2095.08 BOOL  ; RK_07 U8_Z 铝壳上料移载Y轴CW极限输入信号
2095.09 BOOL  ; RK_07 U8_Z 铝壳上料移载Y轴CCW极限输入信号
2095.10 BOOL  ; RK_07 U8_Z 铝壳上料移载Y轴原点接近输入信号
2095.11 BOOL  ; RK_07 U8_Z 铝壳上料移载Y轴原点输入信号
2095.12 BOOL  ; RK_07 U8_Z 铝壳上料移载Y轴中断输入信号
2095.13 BOOL  ; RK_07 U8_Z 铝壳上料移载Y轴紧急停止输入信号
2095.14 BOOL  ; RK_07 U8_Z 铝壳上料移载Y轴定位完成信号
2095.15 BOOL  ; $?St$Bk?_#[5047] / RK_07 U8_Z 铝壳上料移载Y轴偏差计数器复位输出 / 原点调整命令输出$?St$Bk?_#[5047]
2096 CHANNEL  ; RK_07 U8_Z 铝壳上料移载Y轴错误代码
2096.00 BOOL  ; RK_07 U8_Z 铝壳上料移载Y轴错误代码
2096.01 BOOL  ; RK_07 U8_Z 铝壳上料移载Y轴错误代码
2096.02 BOOL  ; RK_07 U8_Z 铝壳上料移载Y轴错误代码
2096.03 BOOL  ; RK_07 U8_Z 铝壳上料移载Y轴错误代码
2096.04 BOOL  ; RK_07 U8_Z 铝壳上料移载Y轴错误代码
2096.05 BOOL  ; RK_07 U8_Z 铝壳上料移载Y轴错误代码
2096.06 BOOL  ; RK_07 U8_Z 铝壳上料移载Y轴错误代码
2096.07 BOOL  ; RK_07 U8_Z 铝壳上料移载Y轴错误代码
2096.08 BOOL  ; RK_07 U8_Z 铝壳上料移载Y轴错误代码
2096.09 BOOL  ; RK_07 U8_Z 铝壳上料移载Y轴错误代码
2096.10 BOOL  ; RK_07 U8_Z 铝壳上料移载Y轴错误代码
2096.11 BOOL  ; RK_07 U8_Z 铝壳上料移载Y轴错误代码
2096.12 BOOL  ; RK_07 U8_Z 铝壳上料移载Y轴错误代码
2096.13 BOOL  ; RK_07 U8_Z 铝壳上料移载Y轴错误代码
2096.14 BOOL  ; RK_07 U8_Z 铝壳上料移载Y轴错误代码
2096.15 BOOL  ; RK_07 U8_Z 铝壳上料移载Y轴错误代码
2097.00 BOOL  ; RK_10 U8_U 电池除尘上料X轴Not Use
2097.01 BOOL  ; RK_10 U8_U 电池除尘上料X轴Not Use
2097.02 BOOL  ; RK_10 U8_U 电池除尘上料X轴Not Use
2097.03 BOOL  ; RK_10 U8_U 电池除尘上料X轴Not Use
2097.04 BOOL  ; RK_10 U8_U 电池除尘上料X轴等待存储器操作标志位
2097.05 BOOL  ; RK_10 U8_U 电池除尘上料X轴定位结束标志位
2097.06 BOOL  ; RK_10 U8_U 电池除尘上料X轴无原点标志位
2097.07 BOOL  ; RK_10 U8_U 电池除尘上料X轴原点停止标志位
2097.08 BOOL  ; RK_10 U8_U 电池除尘上料X轴区域0监控标志位
2097.09 BOOL  ; RK_10 U8_U 电池除尘上料X轴区域1监控标志位
2097.10 BOOL  ; RK_10 U8_U 电池除尘上料X轴区域2监控标志位
2097.11 BOOL  ; RK_10 U8_U 电池除尘上料X轴示教完成标志位
2097.12 BOOL  ; RK_10 U8_U 电池除尘上料X轴错误标志位
2097.13 BOOL  ; RK_10 U8_U 电池除尘上料X轴忙标志位
2097.14 BOOL  ; RK_10 U8_U 电池除尘上料X轴数据传送标志
2097.15 BOOL  ; RK_10 U8_U 电池除尘上料X轴减速停止执行标志
2098.00 BOOL  ; RK_10 U8_U 电池除尘上料X轴Not Use
2098.01 BOOL  ; RK_10 U8_U 电池除尘上料X轴Not Use
2098.02 BOOL  ; RK_10 U8_U 电池除尘上料X轴Not Use
2098.03 BOOL  ; RK_10 U8_U 电池除尘上料X轴Not Use
2098.04 BOOL  ; RK_10 U8_U 电池除尘上料X轴Not Use
2098.05 BOOL  ; RK_10 U8_U 电池除尘上料X轴Not Use
2098.06 BOOL  ; RK_10 U8_U 电池除尘上料X轴Not Use
2098.07 BOOL  ; RK_10 U8_U 电池除尘上料X轴Not Use
2098.08 BOOL  ; RK_10 U8_U 电池除尘上料X轴CW极限输入信号
2098.09 BOOL  ; RK_10 U8_U 电池除尘上料X轴CCW极限输入信号
2098.10 BOOL  ; RK_10 U8_U 电池除尘上料X轴原点接近输入信号
2098.11 BOOL  ; RK_10 U8_U 电池除尘上料X轴原点输入信号
2098.12 BOOL  ; RK_10 U8_U 电池除尘上料X轴中断输入信号
2098.13 BOOL  ; RK_10 U8_U 电池除尘上料X轴紧急停止输入信号
2098.14 BOOL  ; RK_10 U8_U 电池除尘上料X轴定位完成信号
2098.15 BOOL  ; $?St$Bk?_#[5048] / RK_10 U8_U 电池除尘上料X轴偏差计数器复位输出 / 原点调整命令输出$?St$Bk?_#[5048]
2099 CHANNEL  ; RK_10 U8_U 电池除尘上料X轴错误代码
2099.00 BOOL  ; RK_10 U8_U 电池除尘上料X轴错误代码
2099.01 BOOL  ; RK_10 U8_U 电池除尘上料X轴错误代码
2099.02 BOOL  ; RK_10 U8_U 电池除尘上料X轴错误代码
2099.03 BOOL  ; RK_10 U8_U 电池除尘上料X轴错误代码
2099.04 BOOL  ; RK_10 U8_U 电池除尘上料X轴错误代码
2099.05 BOOL  ; RK_10 U8_U 电池除尘上料X轴错误代码
2099.06 BOOL  ; RK_10 U8_U 电池除尘上料X轴错误代码
2099.07 BOOL  ; RK_10 U8_U 电池除尘上料X轴错误代码
2099.08 BOOL  ; RK_10 U8_U 电池除尘上料X轴错误代码
2099.09 BOOL  ; RK_10 U8_U 电池除尘上料X轴错误代码
2099.10 BOOL  ; RK_10 U8_U 电池除尘上料X轴错误代码
2099.11 BOOL  ; RK_10 U8_U 电池除尘上料X轴错误代码
2099.12 BOOL  ; RK_10 U8_U 电池除尘上料X轴错误代码
2099.13 BOOL  ; RK_10 U8_U 电池除尘上料X轴错误代码
2099.14 BOOL  ; RK_10 U8_U 电池除尘上料X轴错误代码
2099.15 BOOL  ; RK_10 U8_U 电池除尘上料X轴错误代码
2101 CHANNEL  ; RK_05 #1入壳压力采样值
2102 CHANNEL  ; RK_05 #2入壳压力采样值
210.01 BOOL  ; PC系统通讯正常标志
210.02 BOOL  ; 整机机械手归零标志
210.03 BOOL  ; 安全门标志
221.00 BOOL  ; 整机复位（M）
221.01 BOOL  ; RK_01 电芯来料机构整机复位（M）
221.02 BOOL  ; RK_02 电芯进料机构整机复位（M）
221.03 BOOL  ; RK_03 电芯上料机构整机复位（M）
221.04 BOOL  ; RK_04 电芯除尘机构整机复位（M）
221.05 BOOL  ; RK_05 #1入壳机构整机复位（M）
221.06 BOOL  ; RK_05 #2入壳机构整机复位（M）
221.07 BOOL  ; RK_06 电池上下料机构整机复位（M）
221.08 BOOL  ; RK_07 铝壳进料机构整机复位（M）
221.09 BOOL  ; RK_07 铝壳上料移载机构整机复位（M）
221.10 BOOL  ; RK_07 #1铝壳上料升降机构整机复位（M）
221.11 BOOL  ; RK_07 #2铝壳上料升降机构整机复位（M）
221.12 BOOL  ; RK_07 铝壳托盘下料升降机构整机复位（M）
221.13 BOOL  ; RK_08 铝壳除尘机构整机复位（M）
221.14 BOOL  ; RK_09 #1Hipot检测机构整机复位（M）
221.15 BOOL  ; RK_09 #2Hipot检测机构整机复位（M）
222.00 BOOL  ; RK_10 电池除尘上料机构整机复位（M）
222.01 BOOL  ; RK_11 电池除尘机构整机复位（M）
222.02 BOOL  ; RK_12 预焊上下料机构整机复位（M）
222.03 BOOL  ; RK_13 #1移载机构整机复位（M）
222.04 BOOL  ; RK_13 #2移载机构整机复位（M）
222.05 BOOL  ; RK_14 #1压装机构整机复位（M）
222.06 BOOL  ; RK_14 #2压装机构整机复位（M）
222.07 BOOL  ; RK_15 轮廓检测机构整机复位（M）
222.08 BOOL  ; RK_16 焊接机构整机复位（M）
2.00 BOOL  ; RK_01 U0_X 电芯来料Y轴报警信号
2.01 BOOL  ; RK_01 U0_X 电芯来料Y轴准备好了信号
2.02 BOOL  ; RK_02 U0_Y 电芯进料X轴报警信号
2.03 BOOL  ; RK_02 U0_Y 电芯进料X轴准备好了信号
2.04 BOOL  ; RK_02 U0_Z 电芯进料Z轴报警信号
2.05 BOOL  ; RK_02 U0_Z 电芯进料Z轴准备好了信号
2.06 BOOL  ; RK_03 U0_U 电芯上料X轴报警信号
2.07 BOOL  ; RK_03 U0_U 电芯上料X轴准备好了信号
2.08 BOOL  ; RK_05 U2_X #1入壳Y轴报警信号
2.09 BOOL  ; RK_05 U2_X #1入壳Y轴准备好了信号
2.10 BOOL  ; RK_05 U2_Y #2入壳Y轴报警信号
2.11 BOOL  ; RK_05 U2_Y #2入壳Y轴准备好了信号
2.13 BOOL  ; RK_05 #1入壳定位陶瓷棒上#1夹紧气缸伸出位
2.14 BOOL  ; RK_05 #1入壳定位陶瓷棒上#2夹紧气缸伸出位
2.15 BOOL  ; RK_05 #1入壳定位陶瓷棒下#1夹紧气缸伸出位
3000.00 BOOL  ; 前工序安全位模拟
300.00 BOOL  ; RK_02 电芯进料机械手夹爪气缸夹紧[Pls]
300.01 BOOL  ; RK_02 电芯进料机械手夹爪气缸张开[Pls]
300.02 BOOL  ; RK_02 电芯进料机械手压紧气缸伸出[Pls]
300.03 BOOL  ; RK_02 电芯进料机械手压紧气缸缩回[Pls]
300.04 BOOL  ; RK_03 电芯上料机械手夹爪气缸夹紧[Pls]
300.05 BOOL  ; RK_03 电芯上料机械手夹爪气缸张开[Pls]
300.06 BOOL  ; RK_03 电芯上料机械手压紧气缸伸出[Pls]
300.07 BOOL  ; RK_03 电芯上料机械手压紧气缸缩回[Pls]
300.08 BOOL  ; RK_03 电芯上料升降气缸下降[Pls]
300.09 BOOL  ; RK_03 电芯上料升降气缸上升[Pls]
300.10 BOOL  ; RK_04 电芯除尘伸缩气缸缩回[Pls]
300.11 BOOL  ; RK_04 电芯除尘伸缩气缸伸出[Pls]
300.12 BOOL  ; RK_05 #1入壳滚轮夹紧气缸伸出[Pls]
300.13 BOOL  ; RK_05 #1入壳滚轮夹紧气缸缩回[Pls]
300.14 BOOL  ; RK_05 #1入壳铝壳定位平台伸缩气缸缩回[Pls]
300.15 BOOL  ; RK_05 #1入壳铝壳定位平台伸缩气缸伸出[Pls]
301.00 BOOL  ; RK_05 #1入壳铝壳定位平台升降气缸上升[Pls]
301.01 BOOL  ; RK_05 #1入壳铝壳定位平台升降气缸下降[Pls]
301.02 BOOL  ; RK_05 #1入壳铝壳定位伸缩气缸缩回[Pls]
301.03 BOOL  ; RK_05 #1入壳铝壳定位伸缩气缸伸出[Pls]
301.04 BOOL  ; RK_05 #1入壳铝壳定位夹爪气缸夹紧[Pls]
301.05 BOOL  ; RK_05 #1入壳铝壳定位夹爪气缸张开[Pls]
301.06 BOOL  ; RK_05 #2入壳滚轮夹紧气缸伸出[Pls]
301.07 BOOL  ; RK_05 #2入壳滚轮夹紧气缸缩回[Pls]
301.08 BOOL  ; RK_05 #2入壳铝壳定位平台伸缩气缸缩回[Pls]
301.09 BOOL  ; RK_05 #2入壳铝壳定位平台伸缩气缸伸出[Pls]
301.10 BOOL  ; RK_05 #2入壳铝壳定位平台升降气缸上升[Pls]
301.11 BOOL  ; RK_05 #2入壳铝壳定位平台升降气缸下降[Pls]
301.12 BOOL  ; RK_05 #2入壳铝壳定位伸缩气缸缩回[Pls]
301.13 BOOL  ; RK_05 #2入壳铝壳定位伸缩气缸伸出[Pls]
301.14 BOOL  ; RK_05 #2入壳铝壳定位夹爪气缸夹紧[Pls]
301.15 BOOL  ; RK_05 #2入壳铝壳定位夹爪气缸张开[Pls]
302.00 BOOL  ; RK_01 U0_X 电芯来料Y轴报警复位[Pls]
302.01 BOOL  ; RK_01 U0_X 电芯来料Y轴使能[Pls]
302.02 BOOL  ; RK_02 U0_Y 电芯进料X轴报警复位[Pls]
302.03 BOOL  ; RK_02 U0_Y 电芯进料X轴使能[Pls]
302.04 BOOL  ; RK_02 U0_Z 电芯进料Z轴报警复位[Pls]
302.05 BOOL  ; RK_02 U0_Z 电芯进料Z轴使能[Pls]
302.06 BOOL  ; RK_03 U0_U 电芯上料X轴报警复位[Pls]
302.07 BOOL  ; RK_03 U0_U 电芯上料X轴使能[Pls]
302.08 BOOL  ; RK_05 U2_X #1入壳Y轴报警复位[Pls]
302.09 BOOL  ; RK_05 U2_X #1入壳Y轴使能[Pls]
302.10 BOOL  ; RK_05 U2_Y #2入壳Y轴报警复位[Pls]
302.11 BOOL  ; RK_05 U2_Y #2入壳Y轴使能[Pls]
302.12 BOOL  ; RK_02 电芯进料Z轴刹车使能[Pls]
302.13 BOOL  ; RK_05 #1入壳定位陶瓷棒夹紧气缸伸出[Pls]
302.14 BOOL  ; RK_05 #1入壳定位陶瓷棒夹紧气缸缩回[Pls]
302.15 BOOL  ; RK_05 #2入壳定位陶瓷棒夹紧气缸伸出[Pls]
303.00 BOOL  ; RK_05 #2入壳定位陶瓷棒夹紧气缸缩回[Pls]
303.01 BOOL  ; RK_04 电芯除尘吹气阀开[Pls]
303.02 BOOL  ; RK_02 扫码NG拉带启动[Pls]
303.03 BOOL  ; RK_05 #1入壳吸盘立真空[Pls]
303.04 BOOL  ; RK_05 #2入壳吸盘立真空[Pls]
303.05 BOOL  ; RK_05 #1入壳吸盘伸缩气缸伸出[Pls]
303.06 BOOL  ; RK_05 #1入壳吸盘伸缩气缸缩回[Pls]
303.07 BOOL  ; RK_05 #2入壳吸盘伸缩气缸伸出[Pls]
303.08 BOOL  ; RK_05 #2入壳吸盘伸缩气缸缩回[Pls]
303.09 BOOL  ; 前端设备对接输出信号（公共）[Pls]
303.10 BOOL  ; 后端设备对接输出信号（公共）[Pls]
303.11 BOOL  ; RK_05 #1入壳电芯定位夹爪气缸伸出[Pls]
303.12 BOOL  ; RK_05 #1入壳电芯定位夹爪气缸缩回[Pls]
303.13 BOOL  ; RK_05 #2入壳电芯定位夹爪气缸伸出[Pls]
303.14 BOOL  ; RK_05 #2入壳电芯定位夹爪气缸缩回[Pls]
308.00 BOOL  ; RK_11 电池除尘旋转伸缩气缸缩回[Pls]
308.01 BOOL  ; RK_11 电池除尘旋转伸缩气缸伸出[Pls]
308.02 BOOL  ; RK_11 电池除尘伸缩气缸伸出[Pls]
308.03 BOOL  ; RK_11 电池除尘伸缩气缸缩回[Pls]
308.04 BOOL  ; RK_11 电池除尘夹爪气缸夹紧[Pls]
308.05 BOOL  ; RK_11 电池除尘夹爪气缸张开[Pls]
308.06 BOOL  ; RK_12 预焊上料机械手夹爪气缸夹紧[Pls]
308.07 BOOL  ; RK_12 预焊上料机械手夹爪气缸张开[Pls]
308.08 BOOL  ; RK_12 预焊下料机械手夹爪气缸夹紧[Pls]
308.09 BOOL  ; RK_12 预焊下料机械手夹爪气缸张开[Pls]
308.10 BOOL  ; RK_13 #1移载升降气缸上升[Pls]
308.11 BOOL  ; RK_13 #1移载升降气缸下降[Pls]
308.12 BOOL  ; RK_13 #1移载定位#1伸缩气缸缩回[Pls]
308.13 BOOL  ; RK_13 #1移载定位#1伸缩气缸伸出[Pls]
308.14 BOOL  ; RK_13 #1移载定位#2伸缩气缸缩回[Pls]
308.15 BOOL  ; RK_13 #1移载定位#2伸缩气缸伸出[Pls]
309.00 BOOL  ; RK_13 #1移载导向#1伸缩气缸伸出[Pls]
309.01 BOOL  ; RK_13 #1移载导向#1伸缩气缸缩回[Pls]
309.02 BOOL  ; RK_13 #1移载导向#2伸缩气缸伸出[Pls]
309.03 BOOL  ; RK_13 #1移载导向#2伸缩气缸缩回[Pls]
309.04 BOOL  ; RK_13 #1移载左右定位伸缩气缸伸出[Pls]
309.05 BOOL  ; RK_13 #1移载左右定位伸缩气缸缩回[Pls]
309.06 BOOL  ; RK_13 #2移载升降气缸上升[Pls]
309.07 BOOL  ; RK_13 #2移载升降气缸下降[Pls]
309.08 BOOL  ; RK_13 #2移载定位#1伸缩气缸缩回[Pls]
309.09 BOOL  ; RK_13 #2移载定位#1伸缩气缸伸出[Pls]
309.10 BOOL  ; RK_13 #2移载定位#2伸缩气缸缩回[Pls]
309.11 BOOL  ; RK_13 #2移载定位#2伸缩气缸伸出[Pls]
309.12 BOOL  ; RK_13 #2移载导向#1伸缩气缸伸出[Pls]
309.13 BOOL  ; RK_13 #2移载导向#1伸缩气缸缩回[Pls]
309.14 BOOL  ; RK_13 #2移载导向#2伸缩气缸伸出[Pls]
309.15 BOOL  ; RK_13 #2移载导向#2伸缩气缸缩回[Pls]
310.00 BOOL  ; RK_13 #2移载左右定位伸缩气缸伸出[Pls]
310.01 BOOL  ; RK_13 #2移载左右定位伸缩气缸缩回[Pls]
310.02 BOOL  ; RK_14 #1压装升降气缸下降[Pls]
310.03 BOOL  ; RK_14 #1压装升降气缸上升[Pls]
310.04 BOOL  ; RK_14 #1压装#1吸盘升降气缸下降[Pls]
310.05 BOOL  ; RK_14 #1压装#1吸盘升降气缸上升[Pls]
310.06 BOOL  ; RK_14 #1压装#2吸盘升降气缸下降[Pls]
310.07 BOOL  ; RK_14 #1压装#2吸盘升降气缸上升[Pls]
310.08 BOOL  ; RK_14 #2压装升降气缸下降[Pls]
310.09 BOOL  ; RK_14 #2压装升降气缸上升[Pls]
310.10 BOOL  ; RK_14 #2压装#1吸盘升降气缸下降[Pls]
310.11 BOOL  ; RK_14 #2压装#1吸盘升降气缸上升[Pls]
310.12 BOOL  ; RK_14 #2压装#2吸盘升降气缸下降[Pls]
310.13 BOOL  ; RK_14 #2压装#2吸盘升降气缸上升[Pls]
310.14 BOOL  ; RK_15 轮廓检测#1伸缩气缸伸出[Pls]
310.15 BOOL  ; RK_15 轮廓检测#1伸缩气缸缩回[Pls]
311.00 BOOL  ; RK_15 轮廓检测#2伸缩气缸伸出[Pls]
311.01 BOOL  ; RK_15 轮廓检测#2伸缩气缸缩回[Pls]
311.02 BOOL  ; RK_12 轮廓检测NG拨料气缸伸出[Pls]
311.03 BOOL  ; RK_12 轮廓检测NG拨料气缸缩回[Pls]
311.04 BOOL  ; RK_11 电池除尘吹气阀开[Pls]
311.05 BOOL  ; 0[Pls]
311.06 BOOL  ; 0[Pls]
311.07 BOOL  ; RK_16 激光焊接触发[Pls]
311.08 BOOL  ; RK_16 PLC急停输出到激光设备[Pls]
311.09 BOOL  ; RK_16 #1移载激光焊任务选择[Pls]
311.10 BOOL  ; RK_16 #2移载激光焊任务选择[Pls]
311.11 BOOL  ; RK_16 集尘器启动[Pls]
311.12 BOOL  ; 0[Pls]
311.13 BOOL  ; 0[Pls]
311.14 BOOL  ; RK_14 #1压装吸盘立真空[Pls]
311.15 BOOL  ; RK_14 #2压装吸盘立真空[Pls]
312.00 BOOL  ; RK_12 U4_X 预焊上下料X轴报警复位[Pls]
312.01 BOOL  ; RK_12 U4_X 预焊上下料X轴使能[Pls]
312.02 BOOL  ; RK_12 U4_Y 预焊上料Z轴报警复位[Pls]
312.03 BOOL  ; RK_12 U4_Y 预焊上料Z轴使能[Pls]
312.04 BOOL  ; RK_12 U4_Z 预焊下料Z轴报警复位[Pls]
312.05 BOOL  ; RK_12 U4_Z 预焊下料Z轴使能[Pls]
312.06 BOOL  ; RK_13 U4_U #1移载Y轴报警复位[Pls]
312.07 BOOL  ; RK_13 U4_U #1移载Y轴使能[Pls]
312.08 BOOL  ; RK_13 U6_X #2移载Y轴报警复位[Pls]
312.09 BOOL  ; RK_13 U6_X #2移载Y轴使能[Pls]
312.10 BOOL  ; RK_16 U6_Y 激光焊接X轴报警复位[Pls]
312.11 BOOL  ; RK_16 U6_Y 激光焊接X轴使能[Pls]
312.12 BOOL  ; RK_16 U6_Z 激光焊接Z轴报警复位[Pls]
312.13 BOOL  ; RK_16 U6_Z 激光焊接Z轴使能[Pls]
312.14 BOOL  ; RK_12 预焊上料Z轴刹车使能[Pls]
312.15 BOOL  ; RK_12 预焊下料Z轴刹车使能[Pls]
313.00 BOOL  ; RK_16 激光焊接Z轴刹车使能[Pls]
313.01 BOOL  ; 0[Pls]
313.02 BOOL  ; 0[Pls]
313.03 BOOL  ; 0[Pls]
313.04 BOOL  ; 0[Pls]
313.05 BOOL  ; RK_12 OK出料拉带启动[Pls]
313.06 BOOL  ; 0[Pls]
313.07 BOOL  ; 0[Pls]
313.08 BOOL  ; 0[Pls]
313.09 BOOL  ; RK_07 #1铝壳上料电机刹车使能[Pls]
313.10 BOOL  ; RK_07 #2铝壳上料电机刹车使能[Pls]
313.11 BOOL  ; RK_07 #3托盘下料电机刹车使能[Pls]
313.12 BOOL  ; 三色灯_红（公共）[Pls]
313.13 BOOL  ; 三色灯_绿（公共）[Pls]
313.14 BOOL  ; 三色灯_黄（公共）[Pls]
313.15 BOOL  ; 蜂鸣器（公共）[Pls]
314.00 BOOL  ; RK_06 铝壳上料升降气缸下降[Pls]
314.01 BOOL  ; RK_06 铝壳上料升降气缸上升[Pls]
314.02 BOOL  ; RK_06 电池下料升降气缸下降[Pls]
314.03 BOOL  ; RK_06 电池下料升降气缸上升[Pls]
314.04 BOOL  ; RK_06 铝壳上料夹爪气缸夹紧[Pls]
314.05 BOOL  ; RK_06 铝壳上料夹爪气缸张开[Pls]
314.06 BOOL  ; RK_06 电池下料夹爪气缸夹紧[Pls]
314.07 BOOL  ; RK_06 电池下料夹爪气缸张开[Pls]
314.08 BOOL  ; RK_07 #1铝壳上料车定位升降气缸上升[Pls]
314.09 BOOL  ; RK_07 #1铝壳上料车定位升降气缸下降[Pls]
314.10 BOOL  ; RK_07 #2铝壳上料车定位升降气缸上升[Pls]
314.11 BOOL  ; RK_07 #2铝壳上料车定位升降气缸下降[Pls]
314.12 BOOL  ; RK_07 #3托盘下料车定位升降气缸上升[Pls]
314.13 BOOL  ; RK_07 #3托盘下料车定位升降气缸下降[Pls]
314.14 BOOL  ; RK_07 铝壳进料机械手升降气缸下降[Pls]
314.15 BOOL  ; RK_07 铝壳进料机械手升降气缸上升[Pls]
315.00 BOOL  ; RK_08 铝壳除尘旋转伸缩气缸缩回[Pls]
315.01 BOOL  ; RK_08 铝壳除尘旋转伸缩气缸伸出[Pls]
315.02 BOOL  ; RK_08 铝壳除尘伸缩气缸伸出[Pls]
315.03 BOOL  ; RK_08 铝壳除尘伸缩气缸缩回[Pls]
315.04 BOOL  ; RK_08 铝壳除尘夹爪气缸夹紧[Pls]
315.05 BOOL  ; RK_08 铝壳除尘夹爪气缸张开[Pls]
315.06 BOOL  ; RK_09 #1Hipot测试旋转伸缩气缸伸出[Pls]
315.07 BOOL  ; RK_09 #1Hipot测试旋转伸缩气缸缩回[Pls]
315.08 BOOL  ; RK_09 #1Hipot测试平台伸缩气缸缩回[Pls]
315.09 BOOL  ; RK_09 #1Hipot测试平台伸缩气缸伸出[Pls]
315.10 BOOL  ; RK_09 #1Hipot测试伸缩气缸伸出[Pls]
315.11 BOOL  ; RK_09 #1Hipot测试伸缩气缸缩回[Pls]
315.12 BOOL  ; RK_09 #2Hipot测试旋转伸缩气缸伸出[Pls]
315.13 BOOL  ; RK_09 #2Hipot测试旋转伸缩气缸缩回[Pls]
315.14 BOOL  ; RK_09 #2Hipot测试平台伸缩气缸缩回[Pls]
315.15 BOOL  ; RK_09 #2Hipot测试平台伸缩气缸伸出[Pls]
316.00 BOOL  ; RK_09 #2Hipot测试伸缩气缸伸出[Pls]
316.01 BOOL  ; RK_09 #2Hipot测试伸缩气缸缩回[Pls]
316.02 BOOL  ; RK_10 电池除尘上料机械手升降气缸下降[Pls]
316.03 BOOL  ; RK_10 电池除尘上料机械手升降气缸上升[Pls]
316.04 BOOL  ; RK_10 电池除尘上料机械手夹爪气缸夹紧[Pls]
316.05 BOOL  ; RK_10 电池除尘上料机械手夹爪气缸张开[Pls]
316.06 BOOL  ; RK_06 U8_X 电池上下料X轴报警复位[Pls]
316.07 BOOL  ; RK_06 U8_X 电池上下料X轴使能[Pls]
316.08 BOOL  ; RK_07 U8_Y 铝壳进料X轴报警复位[Pls]
316.09 BOOL  ; RK_07 U8_Y 铝壳进料X轴使能[Pls]
316.10 BOOL  ; RK_07 U8_Z 铝壳上料移载Y轴报警复位[Pls]
316.11 BOOL  ; RK_07 U8_Z 铝壳上料移载Y轴使能[Pls]
316.12 BOOL  ; RK_10 U8_U 电池除尘上料X轴报警复位[Pls]
316.13 BOOL  ; RK_10 U8_U 电池除尘上料X轴使能[Pls]
316.14 BOOL  ; RK_09 Hipot测试仪远程使能（取消）[Pls]
316.15 BOOL  ; RK_07 #1铝壳上料启动指示[Pls]
317.00 BOOL  ; RK_07 #2铝壳上料启动指示[Pls]
317.01 BOOL  ; RK_07 #3托盘下料启动指示[Pls]
317.02 BOOL  ; RK_07 铝壳上料移载吸盘立真空[Pls]
317.03 BOOL  ; RK_07 铝壳进料吸盘立真空[Pls]
317.04 BOOL  ; RK_07 #1铝壳上料电机正转[Pls]
317.05 BOOL  ; RK_07 #1铝壳上料电机反转[Pls]
317.06 BOOL  ; RK_10 Hipot检测NG拉带启动[Pls]
317.07 BOOL  ; RK_08 铝壳除尘吹气阀开[Pls]
317.08 BOOL  ; 0[Pls]
317.09 BOOL  ; RK_07 #2铝壳上料电机正转[Pls]
317.10 BOOL  ; RK_07 #2铝壳上料电机反转[Pls]
317.11 BOOL  ; 启动指示_绿（公共）[Pls]
317.12 BOOL  ; 停止指示_红（公共）[Pls]
317.13 BOOL  ; 复位指示_黄（公共）[Pls]
317.14 BOOL  ; RK_07 #3托盘下料电机正转[Pls]
317.15 BOOL  ; RK_07 #3托盘下料电机反转[Pls]
321.04 BOOL  ; RK_11 电池除尘吹气阀关[Pls]
321.14 BOOL  ; RK_14 #1压装吸盘破真空[Pls]
321.15 BOOL  ; RK_14 #2压装吸盘破真空[Pls]
323.01 BOOL  ; RK_04 电芯除尘吹气阀关[Pls]
323.02 BOOL  ; RK_02 扫码NG拉带停止[Pls]
323.03 BOOL  ; RK_05 #1入壳吸盘破真空[Pls]
323.04 BOOL  ; RK_05 #2入壳吸盘破真空[Pls]
323.05 BOOL  ; RK_12 OK出料拉带停止[Pls]
327.02 BOOL  ; RK_07 铝壳上料移载吸盘破真空[Pls]
327.03 BOOL  ; RK_07 铝壳进料吸盘破真空[Pls]
327.04 BOOL  ; RK_07 #1铝壳上料电机停止[Pls]
327.06 BOOL  ; RK_10 Hipot检测NG拉带停止[Pls]
327.07 BOOL  ; RK_08 铝壳除尘吹气阀关[Pls]
327.09 BOOL  ; RK_07 #2铝壳上料电机停止[Pls]
327.14 BOOL  ; RK_07 #3托盘下料电机停止[Pls]
350.00 BOOL  ; RK_01 U0_X 电芯来料Y轴待料位[Pls]
350.01 BOOL  ; RK_01 U0_X 电芯来料Y轴上料位[Pls]
350.02 BOOL  ; RK_01 U0_X 电芯来料Y轴扫码位[Pls]
350.03 BOOL  ; RK_01 U0_X 电芯来料Y轴下料位[Pls]
350.04 BOOL  ; 备用[Pls]
350.05 BOOL  ; 备用[Pls]
350.06 BOOL  ; 备用[Pls]
350.07 BOOL  ; 备用[Pls]
350.08 BOOL  ; 备用[Pls]
350.09 BOOL  ; 备用[Pls]
350.10 BOOL  ; RK_01 U0_X 电芯来料Y轴回原点[Pls]
350.11 BOOL  ; RK_01 U0_X 电芯来料Y轴JOG+[Pls]
350.12 BOOL  ; RK_01 U0_X 电芯来料Y轴JOG-[Pls]
350.13 BOOL  ; RK_01 U0_X 电芯来料Y轴JOG高速[Pls]
350.14 BOOL  ; RK_01 U0_X 电芯来料Y轴JOG低速[Pls]
350.15 BOOL  ; 备用[Pls]
351.00 BOOL  ; RK_02 U0_Y 电芯进料X轴待料位[Pls]
351.01 BOOL  ; RK_02 U0_Y 电芯进料X轴取料位[Pls]
351.02 BOOL  ; RK_02 U0_Y 电芯进料X轴扫码OK放料位[Pls]
351.03 BOOL  ; RK_02 U0_Y 电芯进料X轴扫码NG放料位[Pls]
351.04 BOOL  ; 备用[Pls]
351.05 BOOL  ; 备用[Pls]
351.06 BOOL  ; 备用[Pls]
351.07 BOOL  ; 备用[Pls]
351.08 BOOL  ; 备用[Pls]
351.09 BOOL  ; 备用[Pls]
351.10 BOOL  ; RK_02 U0_Y 电芯进料X轴回原点[Pls]
351.11 BOOL  ; RK_02 U0_Y 电芯进料X轴JOG+[Pls]
351.12 BOOL  ; RK_02 U0_Y 电芯进料X轴JOG-[Pls]
351.13 BOOL  ; RK_02 U0_Y 电芯进料X轴JOG高速[Pls]
351.14 BOOL  ; RK_02 U0_Y 电芯进料X轴JOG低速[Pls]
351.15 BOOL  ; 备用[Pls]
352.00 BOOL  ; RK_02 U0_Z 电芯进料Z轴待料位（扫码）[Pls]
352.01 BOOL  ; RK_02 U0_Z 电芯进料Z轴取料位[Pls]
352.02 BOOL  ; RK_02 U0_Z 电芯进料Z轴扫码OK放料位[Pls]
352.03 BOOL  ; RK_02 U0_Z 电芯进料Z轴扫码NG放料位[Pls]
352.04 BOOL  ; RK_02 U0_Z 电芯进料Z轴扫码位[Pls]
352.05 BOOL  ; 备用[Pls]
352.06 BOOL  ; 备用[Pls]
352.07 BOOL  ; 备用[Pls]
352.08 BOOL  ; 备用[Pls]
352.09 BOOL  ; 备用[Pls]
352.10 BOOL  ; RK_02 U0_Z 电芯进料Z轴回原点[Pls]
352.11 BOOL  ; RK_02 U0_Z 电芯进料Z轴JOG+[Pls]
352.12 BOOL  ; RK_02 U0_Z 电芯进料Z轴JOG-[Pls]
352.13 BOOL  ; RK_02 U0_Z 电芯进料Z轴JOG高速[Pls]
352.14 BOOL  ; RK_02 U0_Z 电芯进料Z轴JOG低速[Pls]
352.15 BOOL  ; 备用[Pls]
353.00 BOOL  ; RK_03 U0_U 电芯上料X轴待料位[Pls]
353.01 BOOL  ; RK_03 U0_U 电芯上料X轴取料位[Pls]
353.02 BOOL  ; RK_03 U0_U 电芯上料X轴#1入壳放料位[Pls]
353.03 BOOL  ; RK_03 U0_U 电芯上料X轴#2入壳放料位[Pls]
353.04 BOOL  ; 备用[Pls]
353.05 BOOL  ; 备用[Pls]
353.06 BOOL  ; 备用[Pls]
353.07 BOOL  ; 备用[Pls]
353.08 BOOL  ; 备用[Pls]
353.09 BOOL  ; 备用[Pls]
353.10 BOOL  ; RK_03 U0_U 电芯上料X轴回原点[Pls]
353.11 BOOL  ; RK_03 U0_U 电芯上料X轴JOG+[Pls]
353.12 BOOL  ; RK_03 U0_U 电芯上料X轴JOG-[Pls]
353.13 BOOL  ; RK_03 U0_U 电芯上料X轴JOG高速[Pls]
353.14 BOOL  ; RK_03 U0_U 电芯上料X轴JOG低速[Pls]
353.15 BOOL  ; 备用[Pls]
354.00 BOOL  ; RK_05 U2_X #1入壳Y轴待料位[Pls]
354.01 BOOL  ; RK_05 U2_X #1入壳Y轴滚轮压紧位[Pls]
354.02 BOOL  ; RK_05 U2_X #1入壳Y轴滚轮松开位[Pls]
354.03 BOOL  ; RK_05 U2_X #1入壳Y轴入壳位[Pls]
354.04 BOOL  ; RK_05 U2_X #1入壳Y轴电芯定位夹爪松开位[Pls]
354.05 BOOL  ; 备用[Pls]
354.06 BOOL  ; 备用[Pls]
354.07 BOOL  ; 备用[Pls]
354.08 BOOL  ; 备用[Pls]
354.09 BOOL  ; 备用[Pls]
354.10 BOOL  ; RK_05 U2_X #1入壳Y轴回原点[Pls]
354.11 BOOL  ; RK_05 U2_X #1入壳Y轴JOG+[Pls]
354.12 BOOL  ; RK_05 U2_X #1入壳Y轴JOG-[Pls]
354.13 BOOL  ; RK_05 U2_X #1入壳Y轴JOG高速[Pls]
354.14 BOOL  ; RK_05 U2_X #1入壳Y轴JOG低速[Pls]
354.15 BOOL  ; 备用[Pls]
355.00 BOOL  ; RK_05 U2_Y #2入壳Y轴待料位[Pls]
355.01 BOOL  ; RK_05 U2_Y #2入壳Y轴滚轮压紧位[Pls]
355.02 BOOL  ; RK_05 U2_Y #2入壳Y轴滚轮松开位[Pls]
355.03 BOOL  ; RK_05 U2_Y #2入壳Y轴入壳位[Pls]
355.04 BOOL  ; RK_05 U2_Y #2入壳Y轴电芯定位夹爪松开位[Pls]
355.05 BOOL  ; 备用[Pls]
355.06 BOOL  ; 备用[Pls]
355.07 BOOL  ; 备用[Pls]
355.08 BOOL  ; 备用[Pls]
355.09 BOOL  ; 备用[Pls]
355.10 BOOL  ; RK_05 U2_Y #2入壳Y轴回原点[Pls]
355.11 BOOL  ; RK_05 U2_Y #2入壳Y轴JOG+[Pls]
355.12 BOOL  ; RK_05 U2_Y #2入壳Y轴JOG-[Pls]
355.13 BOOL  ; RK_05 U2_Y #2入壳Y轴JOG高速[Pls]
355.14 BOOL  ; RK_05 U2_Y #2入壳Y轴JOG低速[Pls]
355.15 BOOL  ; 备用[Pls]
356.00 BOOL  ; RK_12 U4_X 预焊上下料X轴待料位[Pls]
356.01 BOOL  ; RK_12 U4_X 预焊上下料X轴除尘取料位[Pls]
356.02 BOOL  ; RK_12 U4_X 预焊上下料X轴#1移载放料位[Pls]
356.03 BOOL  ; RK_12 U4_X 预焊上下料X轴#2移载放料位[Pls]
356.04 BOOL  ; RK_12 U4_X 预焊上下料X轴#1移载取料位[Pls]
356.05 BOOL  ; RK_12 U4_X 预焊上下料X轴#2移载取料位[Pls]
356.06 BOOL  ; RK_12 U4_X 预焊上下料X轴OK放料位[Pls]
356.07 BOOL  ; RK_12 U4_X 预焊上下料X轴#1NG放料位[Pls]
356.08 BOOL  ; RK_12 U4_X 预焊上下料X轴#2NG放料位[Pls]
356.09 BOOL  ; 备用[Pls]
356.10 BOOL  ; RK_12 U4_X 预焊上下料X轴回原点[Pls]
356.11 BOOL  ; RK_12 U4_X 预焊上下料X轴JOG+[Pls]
356.12 BOOL  ; RK_12 U4_X 预焊上下料X轴JOG-[Pls]
356.13 BOOL  ; RK_12 U4_X 预焊上下料X轴JOG高速[Pls]
356.14 BOOL  ; RK_12 U4_X 预焊上下料X轴JOG低速[Pls]
356.15 BOOL  ; 备用[Pls]
357.00 BOOL  ; RK_12 U4_Y 预焊上料Z轴待料位[Pls]
357.01 BOOL  ; RK_12 U4_Y 预焊上料Z轴除尘取料位[Pls]
357.02 BOOL  ; RK_12 U4_Y 预焊上料Z轴#1移载放料位[Pls]
357.03 BOOL  ; RK_12 U4_Y 预焊上料Z轴#2移载放料位[Pls]
357.04 BOOL  ; 备用[Pls]
357.05 BOOL  ; 备用[Pls]
357.06 BOOL  ; 备用[Pls]
357.07 BOOL  ; 备用[Pls]
357.08 BOOL  ; 备用[Pls]
357.09 BOOL  ; 备用[Pls]
357.10 BOOL  ; RK_12 U4_Y 预焊上料Z轴回原点[Pls]
357.11 BOOL  ; RK_12 U4_Y 预焊上料Z轴JOG+[Pls]
357.12 BOOL  ; RK_12 U4_Y 预焊上料Z轴JOG-[Pls]
357.13 BOOL  ; RK_12 U4_Y 预焊上料Z轴JOG高速[Pls]
357.14 BOOL  ; RK_12 U4_Y 预焊上料Z轴JOG低速[Pls]
357.15 BOOL  ; 备用[Pls]
358.00 BOOL  ; RK_12 U4_Z 预焊下料Z轴待料位[Pls]
358.01 BOOL  ; RK_12 U4_Z 预焊下料Z轴#1移载取料位[Pls]
358.02 BOOL  ; RK_12 U4_Z 预焊下料Z轴#2移载取料位[Pls]
358.03 BOOL  ; RK_12 U4_Z 预焊下料Z轴OK放料位[Pls]
358.04 BOOL  ; RK_12 U4_Z 预焊下料Z轴#1NG放料位[Pls]
358.05 BOOL  ; RK_12 U4_Z 预焊下料Z轴#2NG放料位[Pls]
358.06 BOOL  ; 备用[Pls]
358.07 BOOL  ; 备用[Pls]
358.08 BOOL  ; 备用[Pls]
358.09 BOOL  ; 备用[Pls]
358.10 BOOL  ; RK_12 U4_Z 预焊下料Z轴回原点[Pls]
358.11 BOOL  ; RK_12 U4_Z 预焊下料Z轴JOG+[Pls]
358.12 BOOL  ; RK_12 U4_Z 预焊下料Z轴JOG-[Pls]
358.13 BOOL  ; RK_12 U4_Z 预焊下料Z轴JOG高速[Pls]
358.14 BOOL  ; RK_12 U4_Z 预焊下料Z轴JOG低速[Pls]
358.15 BOOL  ; 备用[Pls]
359.00 BOOL  ; RK_13 U4_U #1移载Y轴待料位[Pls]
359.01 BOOL  ; RK_13 U4_U #1移载Y轴取放料位[Pls]
359.02 BOOL  ; RK_13 U4_U #1移载Y轴压装位[Pls]
359.03 BOOL  ; RK_13 U4_U #1移载Y轴#1轮廓检测位[Pls]
359.04 BOOL  ; RK_13 U4_U #1移载Y轴#2轮廓检测位[Pls]
359.05 BOOL  ; RK_13 U4_U #1移载Y轴激光焊接位[Pls]
359.06 BOOL  ; 备用[Pls]
359.07 BOOL  ; 备用[Pls]
359.08 BOOL  ; 备用[Pls]
359.09 BOOL  ; 备用[Pls]
359.10 BOOL  ; RK_13 U4_U #1移载Y轴回原点[Pls]
359.11 BOOL  ; RK_13 U4_U #1移载Y轴JOG+[Pls]
359.12 BOOL  ; RK_13 U4_U #1移载Y轴JOG-[Pls]
359.13 BOOL  ; RK_13 U4_U #1移载Y轴JOG高速[Pls]
359.14 BOOL  ; RK_13 U4_U #1移载Y轴JOG低速[Pls]
359.15 BOOL  ; 备用[Pls]
360.00 BOOL  ; RK_13 U6_X #2移载Y轴待料位[Pls]
360.01 BOOL  ; RK_13 U6_X #2移载Y轴取放料位[Pls]
360.02 BOOL  ; RK_13 U6_X #2移载Y轴压装位[Pls]
360.03 BOOL  ; RK_13 U6_X #2移载Y轴#1轮廓检测位[Pls]
360.04 BOOL  ; RK_13 U6_X #2移载Y轴#2轮廓检测位[Pls]
360.05 BOOL  ; RK_13 U6_X #2移载Y轴激光焊接位[Pls]
360.06 BOOL  ; 备用[Pls]
360.07 BOOL  ; 备用[Pls]
360.08 BOOL  ; 备用[Pls]
360.09 BOOL  ; 备用[Pls]
360.10 BOOL  ; RK_13 U6_X #2移载Y轴回原点[Pls]
360.11 BOOL  ; RK_13 U6_X #2移载Y轴JOG+[Pls]
360.12 BOOL  ; RK_13 U6_X #2移载Y轴JOG-[Pls]
360.13 BOOL  ; RK_13 U6_X #2移载Y轴JOG高速[Pls]
360.14 BOOL  ; RK_13 U6_X #2移载Y轴JOG低速[Pls]
360.15 BOOL  ; 备用[Pls]
361.00 BOOL  ; RK_16 U6_Y 激光焊接X轴待机位[Pls]
361.01 BOOL  ; RK_16 U6_Y 激光焊接X轴#1移载焊接位[Pls]
361.02 BOOL  ; RK_16 U6_Y 激光焊接X轴#2移载焊接位[Pls]
361.03 BOOL  ; 备用[Pls]
361.04 BOOL  ; 备用[Pls]
361.05 BOOL  ; 备用[Pls]
361.06 BOOL  ; 备用[Pls]
361.07 BOOL  ; 备用[Pls]
361.08 BOOL  ; 备用[Pls]
361.09 BOOL  ; 备用[Pls]
361.10 BOOL  ; RK_16 U6_Y 激光焊接X轴回原点[Pls]
361.11 BOOL  ; RK_16 U6_Y 激光焊接X轴JOG+[Pls]
361.12 BOOL  ; RK_16 U6_Y 激光焊接X轴JOG-[Pls]
361.13 BOOL  ; RK_16 U6_Y 激光焊接X轴JOG高速[Pls]
361.14 BOOL  ; RK_16 U6_Y 激光焊接X轴JOG低速[Pls]
361.15 BOOL  ; 备用[Pls]
362.00 BOOL  ; RK_16 U6_Z 激光焊接Z轴待机位[Pls]
362.01 BOOL  ; RK_16 U6_Z 激光焊接Z轴#1移载焊接位[Pls]
362.02 BOOL  ; RK_16 U6_Z 激光焊接Z轴#2移载焊接位[Pls]
362.03 BOOL  ; 备用[Pls]
362.04 BOOL  ; 备用[Pls]
362.05 BOOL  ; 备用[Pls]
362.06 BOOL  ; 备用[Pls]
362.07 BOOL  ; 备用[Pls]
362.08 BOOL  ; 备用[Pls]
362.09 BOOL  ; 备用[Pls]
362.10 BOOL  ; RK_16 U6_Z 激光焊接Z轴回原点[Pls]
362.11 BOOL  ; RK_16 U6_Z 激光焊接Z轴JOG+[Pls]
362.12 BOOL  ; RK_16 U6_Z 激光焊接Z轴JOG-[Pls]
362.13 BOOL  ; RK_16 U6_Z 激光焊接Z轴JOG高速[Pls]
362.14 BOOL  ; RK_16 U6_Z 激光焊接Z轴JOG低速[Pls]
362.15 BOOL  ; 备用[Pls]
363.00 BOOL  ; RK_06 U8_X 电池上下料X轴待机位[Pls]
363.01 BOOL  ; RK_06 U8_X 电池上下料X轴铝壳除尘取料位[Pls]
363.02 BOOL  ; RK_06 U8_X 电池上下料X轴#1入壳放料位[Pls]
363.03 BOOL  ; RK_06 U8_X 电池上下料X轴#2入壳放料位[Pls]
363.04 BOOL  ; RK_06 U8_X 电池上下料X轴#1入壳取料位[Pls]
363.05 BOOL  ; RK_06 U8_X 电池上下料X轴#2入壳取料位[Pls]
363.06 BOOL  ; RK_06 U8_X 电池上下料X轴#1Hipot检测放料位[Pls]
363.07 BOOL  ; RK_06 U8_X 电池上下料X轴#2Hipot检测放料位[Pls]
363.08 BOOL  ; 备用[Pls]
363.09 BOOL  ; 备用[Pls]
363.10 BOOL  ; RK_06 U8_X 电池上下料X轴回原点[Pls]
363.11 BOOL  ; RK_06 U8_X 电池上下料X轴JOG+[Pls]
363.12 BOOL  ; RK_06 U8_X 电池上下料X轴JOG-[Pls]
363.13 BOOL  ; RK_06 U8_X 电池上下料X轴JOG高速[Pls]
363.14 BOOL  ; RK_06 U8_X 电池上下料X轴JOG低速[Pls]
363.15 BOOL  ; 备用[Pls]
364.00 BOOL  ; RK_07 U8_Y 铝壳进料X轴等待位[Pls]
364.01 BOOL  ; RK_07 U8_Y 铝壳进料X轴取料位[Pls]
364.02 BOOL  ; RK_07 U8_Y 铝壳进料X轴放料位[Pls]
364.03 BOOL  ; 备用[Pls]
364.04 BOOL  ; 备用[Pls]
364.05 BOOL  ; 备用[Pls]
364.06 BOOL  ; 备用[Pls]
364.07 BOOL  ; 备用[Pls]
364.08 BOOL  ; 备用[Pls]
364.09 BOOL  ; 备用[Pls]
364.10 BOOL  ; RK_07 U8_Y 铝壳进料X轴回原点[Pls]
364.11 BOOL  ; RK_07 U8_Y 铝壳进料X轴JOG+[Pls]
364.12 BOOL  ; RK_07 U8_Y 铝壳进料X轴JOG-[Pls]
364.13 BOOL  ; RK_07 U8_Y 铝壳进料X轴JOG高速[Pls]
364.14 BOOL  ; RK_07 U8_Y 铝壳进料X轴JOG低速[Pls]
364.15 BOOL  ; 备用[Pls]
365.00 BOOL  ; RK_07 U8_Z 铝壳上料移载Y轴待料位[Pls]
365.01 BOOL  ; RK_07 U8_Z 铝壳上料移载Y轴#1铝壳上料位[Pls]
365.02 BOOL  ; RK_07 U8_Z 铝壳上料移载Y轴#2铝壳上料位[Pls]
365.03 BOOL  ; RK_07 U8_Z 铝壳上料移载Y轴#3铝壳托盘下料位[Pls]
365.04 BOOL  ; RK_07 U8_Z 铝壳上料移载Y轴铝壳取料位[Pls]
365.05 BOOL  ; 备用[Pls]
365.06 BOOL  ; 备用[Pls]
365.07 BOOL  ; 备用[Pls]
365.08 BOOL  ; 备用[Pls]
365.09 BOOL  ; 备用[Pls]
365.10 BOOL  ; RK_07 U8_Z 铝壳上料移载Y轴回原点[Pls]
365.11 BOOL  ; RK_07 U8_Z 铝壳上料移载Y轴JOG+[Pls]
365.12 BOOL  ; RK_07 U8_Z 铝壳上料移载Y轴JOG-[Pls]
365.13 BOOL  ; RK_07 U8_Z 铝壳上料移载Y轴JOG高速[Pls]
365.14 BOOL  ; RK_07 U8_Z 铝壳上料移载Y轴JOG低速[Pls]
365.15 BOOL  ; 备用[Pls]
366.00 BOOL  ; RK_10 U8_U 电池除尘上料X轴待料位[Pls]
366.01 BOOL  ; RK_10 U8_U 电池除尘上料X轴#1Hipot检测取料位[Pls]
366.02 BOOL  ; RK_10 U8_U 电池除尘上料X轴#2Hipot检测取料位[Pls]
366.03 BOOL  ; RK_10 U8_U 电池除尘上料X轴Hipot OK放料位[Pls]
366.04 BOOL  ; RK_10 U8_U 电池除尘上料X轴Hipot NG放料位[Pls]
366.05 BOOL  ; 备用[Pls]
366.06 BOOL  ; 备用[Pls]
366.07 BOOL  ; 备用[Pls]
366.08 BOOL  ; 备用[Pls]
366.09 BOOL  ; 备用[Pls]
366.10 BOOL  ; RK_10 U8_U 电池除尘上料X轴回原点[Pls]
366.11 BOOL  ; RK_10 U8_U 电池除尘上料X轴JOG+[Pls]
366.12 BOOL  ; RK_10 U8_U 电池除尘上料X轴JOG-[Pls]
366.13 BOOL  ; RK_10 U8_U 电池除尘上料X轴JOG高速[Pls]
366.14 BOOL  ; RK_10 U8_U 电池除尘上料X轴JOG低速[Pls]
366.15 BOOL  ; 备用[Pls]
3.00 BOOL  ; RK_05 #1入壳定位陶瓷棒下#2夹紧气缸伸出位
3.01 BOOL  ; RK_05 #1入壳定位陶瓷棒上#1夹紧气缸缩回位
3.02 BOOL  ; RK_05 #1入壳定位陶瓷棒上#2夹紧气缸缩回位
3.03 BOOL  ; RK_05 #1入壳定位陶瓷棒下#1夹紧气缸缩回位
3.04 BOOL  ; RK_05 #1入壳定位陶瓷棒下#2夹紧气缸缩回位
3.05 BOOL  ; RK_05 #1入壳吸盘上#1伸缩气缸缩回位
3.06 BOOL  ; RK_05 #1入壳吸盘上#2伸缩气缸缩回位
3.07 BOOL  ; RK_05 #1入壳吸盘上#3伸缩气缸缩回位
3.08 BOOL  ; RK_05 #1入壳吸盘下#1伸缩气缸缩回位
3.09 BOOL  ; RK_05 #1入壳吸盘下#2伸缩气缸缩回位
3.10 BOOL  ; RK_05 #1入壳吸盘下#3伸缩气缸缩回位
3.11 BOOL  ; RK_05 #1入壳电芯#1定位夹爪气缸松开位
3.12 BOOL  ; RK_05 #1入壳电芯#2定位夹爪气缸松开位
3.13 BOOL  ; RK_05 #1入壳电芯#1定位夹爪气缸夹紧位
3.14 BOOL  ; RK_05 #1入壳电芯#2定位夹爪气缸夹紧位
3.15 BOOL  ; RK_05 #2入壳定位陶瓷棒上#1夹紧气缸伸出位
400.00 BOOL  ; RK_02 电芯进料机械手夹爪气缸夹紧[M]
400.01 BOOL  ; RK_02 电芯进料机械手夹爪气缸张开[M]
400.02 BOOL  ; RK_02 电芯进料机械手压紧气缸伸出[M]
400.03 BOOL  ; RK_02 电芯进料机械手压紧气缸缩回[M]
400.04 BOOL  ; RK_03 电芯上料机械手夹爪气缸夹紧[M]
400.05 BOOL  ; RK_03 电芯上料机械手夹爪气缸张开[M]
400.06 BOOL  ; RK_03 电芯上料机械手压紧气缸伸出[M]
400.07 BOOL  ; RK_03 电芯上料机械手压紧气缸缩回[M]
400.08 BOOL  ; RK_03 电芯上料升降气缸下降[M]
400.09 BOOL  ; RK_03 电芯上料升降气缸上升[M]
400.10 BOOL  ; RK_04 电芯除尘伸缩气缸缩回[M]
400.11 BOOL  ; RK_04 电芯除尘伸缩气缸伸出[M]
400.12 BOOL  ; RK_05 #1入壳滚轮夹紧气缸伸出[M]
400.13 BOOL  ; RK_05 #1入壳滚轮夹紧气缸缩回[M]
400.14 BOOL  ; RK_05 #1入壳铝壳定位平台伸缩气缸缩回[M]
400.15 BOOL  ; RK_05 #1入壳铝壳定位平台伸缩气缸伸出[M]
401.00 BOOL  ; RK_05 #1入壳铝壳定位平台升降气缸上升[M]
401.01 BOOL  ; RK_05 #1入壳铝壳定位平台升降气缸下降[M]
401.02 BOOL  ; RK_05 #1入壳铝壳定位伸缩气缸缩回[M]
401.03 BOOL  ; RK_05 #1入壳铝壳定位伸缩气缸伸出[M]
401.04 BOOL  ; RK_05 #1入壳铝壳定位夹爪气缸夹紧[M]
401.05 BOOL  ; RK_05 #1入壳铝壳定位夹爪气缸张开[M]
401.06 BOOL  ; RK_05 #2入壳滚轮夹紧气缸伸出[M]
401.07 BOOL  ; RK_05 #2入壳滚轮夹紧气缸缩回[M]
401.08 BOOL  ; RK_05 #2入壳铝壳定位平台伸缩气缸缩回[M]
401.09 BOOL  ; RK_05 #2入壳铝壳定位平台伸缩气缸伸出[M]
401.10 BOOL  ; RK_05 #2入壳铝壳定位平台升降气缸上升[M]
401.11 BOOL  ; RK_05 #2入壳铝壳定位平台升降气缸下降[M]
401.12 BOOL  ; RK_05 #2入壳铝壳定位伸缩气缸缩回[M]
401.13 BOOL  ; RK_05 #2入壳铝壳定位伸缩气缸伸出[M]
401.14 BOOL  ; RK_05 #2入壳铝壳定位夹爪气缸夹紧[M]
401.15 BOOL  ; RK_05 #2入壳铝壳定位夹爪气缸张开[M]
402.00 BOOL  ; RK_01 U0_X 电芯来料Y轴报警复位[M]
402.01 BOOL  ; RK_01 U0_X 电芯来料Y轴使能[M]
402.02 BOOL  ; RK_02 U0_Y 电芯进料X轴报警复位[M]
402.03 BOOL  ; RK_02 U0_Y 电芯进料X轴使能[M]
402.04 BOOL  ; RK_02 U0_Z 电芯进料Z轴报警复位[M]
402.05 BOOL  ; RK_02 U0_Z 电芯进料Z轴使能[M]
402.06 BOOL  ; RK_03 U0_U 电芯上料X轴报警复位[M]
402.07 BOOL  ; RK_03 U0_U 电芯上料X轴使能[M]
402.08 BOOL  ; RK_05 U2_X #1入壳Y轴报警复位[M]
402.09 BOOL  ; RK_05 U2_X #1入壳Y轴使能[M]
402.10 BOOL  ; RK_05 U2_Y #2入壳Y轴报警复位[M]
402.11 BOOL  ; RK_05 U2_Y #2入壳Y轴使能[M]
402.12 BOOL  ; RK_02 电芯进料Z轴刹车使能[M]
402.13 BOOL  ; RK_05 #1入壳定位陶瓷棒夹紧气缸伸出[M]
402.14 BOOL  ; RK_05 #1入壳定位陶瓷棒夹紧气缸缩回[M]
402.15 BOOL  ; RK_05 #2入壳定位陶瓷棒夹紧气缸伸出[M]
403.00 BOOL  ; RK_05 #2入壳定位陶瓷棒夹紧气缸缩回[M]
403.01 BOOL  ; RK_04 电芯除尘吹气阀开[M]
403.02 BOOL  ; RK_02 扫码NG拉带启动[M]
403.03 BOOL  ; RK_05 #1入壳吸盘立真空[M]
403.04 BOOL  ; RK_05 #2入壳吸盘立真空[M]
403.05 BOOL  ; RK_05 #1入壳吸盘伸缩气缸伸出[M]
403.06 BOOL  ; RK_05 #1入壳吸盘伸缩气缸缩回[M]
403.07 BOOL  ; RK_05 #2入壳吸盘伸缩气缸伸出[M]
403.08 BOOL  ; RK_05 #2入壳吸盘伸缩气缸缩回[M]
403.09 BOOL  ; 前端设备对接输出信号（公共）[M]
403.10 BOOL  ; 后端设备对接输出信号（公共）[M]
403.11 BOOL  ; RK_05 #1入壳电芯定位夹爪气缸伸出[M]
403.12 BOOL  ; RK_05 #1入壳电芯定位夹爪气缸缩回[M]
403.13 BOOL  ; RK_05 #2入壳电芯定位夹爪气缸伸出[M]
403.14 BOOL  ; RK_05 #2入壳电芯定位夹爪气缸缩回[M]
408.00 BOOL  ; RK_11 电池除尘旋转伸缩气缸缩回[M]
408.01 BOOL  ; RK_11 电池除尘旋转伸缩气缸伸出[M]
408.02 BOOL  ; RK_11 电池除尘伸缩气缸伸出[M]
408.03 BOOL  ; RK_11 电池除尘伸缩气缸缩回[M]
408.04 BOOL  ; RK_11 电池除尘夹爪气缸夹紧[M]
408.05 BOOL  ; RK_11 电池除尘夹爪气缸张开[M]
408.06 BOOL  ; RK_12 预焊上料机械手夹爪气缸夹紧[M]
408.07 BOOL  ; RK_12 预焊上料机械手夹爪气缸张开[M]
408.08 BOOL  ; RK_12 预焊下料机械手夹爪气缸夹紧[M]
408.09 BOOL  ; RK_12 预焊下料机械手夹爪气缸张开[M]
408.10 BOOL  ; RK_13 #1移载升降气缸上升[M]
408.11 BOOL  ; RK_13 #1移载升降气缸下降[M]
408.12 BOOL  ; RK_13 #1移载定位#1伸缩气缸缩回[M]
408.13 BOOL  ; RK_13 #1移载定位#1伸缩气缸伸出[M]
408.14 BOOL  ; RK_13 #1移载定位#2伸缩气缸缩回[M]
408.15 BOOL  ; RK_13 #1移载定位#2伸缩气缸伸出[M]
409.00 BOOL  ; RK_13 #1移载导向#1伸缩气缸伸出[M]
409.01 BOOL  ; RK_13 #1移载导向#1伸缩气缸缩回[M]
409.02 BOOL  ; RK_13 #1移载导向#2伸缩气缸伸出[M]
409.03 BOOL  ; RK_13 #1移载导向#2伸缩气缸缩回[M]
409.04 BOOL  ; RK_13 #1移载左右定位伸缩气缸伸出[M]
409.05 BOOL  ; RK_13 #1移载左右定位伸缩气缸缩回[M]
409.06 BOOL  ; RK_13 #2移载升降气缸上升[M]
409.07 BOOL  ; RK_13 #2移载升降气缸下降[M]
409.08 BOOL  ; RK_13 #2移载定位#1伸缩气缸缩回[M]
409.09 BOOL  ; RK_13 #2移载定位#1伸缩气缸伸出[M]
409.10 BOOL  ; RK_13 #2移载定位#2伸缩气缸缩回[M]
409.11 BOOL  ; RK_13 #2移载定位#2伸缩气缸伸出[M]
409.12 BOOL  ; RK_13 #2移载导向#1伸缩气缸伸出[M]
409.13 BOOL  ; RK_13 #2移载导向#1伸缩气缸缩回[M]
409.14 BOOL  ; RK_13 #2移载导向#2伸缩气缸伸出[M]
409.15 BOOL  ; RK_13 #2移载导向#2伸缩气缸缩回[M]
410.00 BOOL  ; RK_13 #2移载左右定位伸缩气缸伸出[M]
410.01 BOOL  ; RK_13 #2移载左右定位伸缩气缸缩回[M]
410.02 BOOL  ; RK_14 #1压装升降气缸下降[M]
410.03 BOOL  ; RK_14 #1压装升降气缸上升[M]
410.04 BOOL  ; RK_14 #1压装#1吸盘升降气缸下降[M]
410.05 BOOL  ; RK_14 #1压装#1吸盘升降气缸上升[M]
410.06 BOOL  ; RK_14 #1压装#2吸盘升降气缸下降[M]
410.07 BOOL  ; RK_14 #1压装#2吸盘升降气缸上升[M]
410.08 BOOL  ; RK_14 #2压装升降气缸下降[M]
410.09 BOOL  ; RK_14 #2压装升降气缸上升[M]
410.10 BOOL  ; RK_14 #2压装#1吸盘升降气缸下降[M]
410.11 BOOL  ; RK_14 #2压装#1吸盘升降气缸上升[M]
410.12 BOOL  ; RK_14 #2压装#2吸盘升降气缸下降[M]
410.13 BOOL  ; RK_14 #2压装#2吸盘升降气缸上升[M]
410.14 BOOL  ; RK_15 轮廓检测#1伸缩气缸伸出[M]
410.15 BOOL  ; RK_15 轮廓检测#1伸缩气缸缩回[M]
411.00 BOOL  ; RK_15 轮廓检测#2伸缩气缸伸出[M]
411.01 BOOL  ; RK_15 轮廓检测#2伸缩气缸缩回[M]
411.02 BOOL  ; RK_12 轮廓检测NG拨料气缸伸出[M]
411.03 BOOL  ; RK_12 轮廓检测NG拨料气缸缩回[M]
411.04 BOOL  ; RK_11 电池除尘吹气阀开[M]
411.05 BOOL  ; 0[M]
411.06 BOOL  ; 0[M]
411.07 BOOL  ; RK_16 激光焊接触发[M]
411.08 BOOL  ; RK_16 PLC急停输出到激光设备[M]
411.09 BOOL  ; RK_16 #1移载激光焊任务选择[M]
411.10 BOOL  ; RK_16 #2移载激光焊任务选择[M]
411.11 BOOL  ; RK_16 集尘器启动[M]
411.12 BOOL  ; 0[M]
411.13 BOOL  ; 0[M]
411.14 BOOL  ; RK_14 #1压装吸盘立真空[M]
411.15 BOOL  ; RK_14 #2压装吸盘立真空[M]
412.00 BOOL  ; RK_12 U4_X 预焊上下料X轴报警复位[M]
412.01 BOOL  ; RK_12 U4_X 预焊上下料X轴使能[M]
412.02 BOOL  ; RK_12 U4_Y 预焊上料Z轴报警复位[M]
412.03 BOOL  ; RK_12 U4_Y 预焊上料Z轴使能[M]
412.04 BOOL  ; RK_12 U4_Z 预焊下料Z轴报警复位[M]
412.05 BOOL  ; RK_12 U4_Z 预焊下料Z轴使能[M]
412.06 BOOL  ; RK_13 U4_U #1移载Y轴报警复位[M]
412.07 BOOL  ; RK_13 U4_U #1移载Y轴使能[M]
412.08 BOOL  ; RK_13 U6_X #2移载Y轴报警复位[M]
412.09 BOOL  ; RK_13 U6_X #2移载Y轴使能[M]
412.10 BOOL  ; RK_16 U6_Y 激光焊接X轴报警复位[M]
412.11 BOOL  ; RK_16 U6_Y 激光焊接X轴使能[M]
412.12 BOOL  ; RK_16 U6_Z 激光焊接Z轴报警复位[M]
412.13 BOOL  ; RK_16 U6_Z 激光焊接Z轴使能[M]
412.14 BOOL  ; RK_12 预焊上料Z轴刹车使能[M]
412.15 BOOL  ; RK_12 预焊下料Z轴刹车使能[M]
413.00 BOOL  ; RK_16 激光焊接Z轴刹车使能[M]
413.01 BOOL  ; 0[M]
413.02 BOOL  ; 0[M]
413.03 BOOL  ; 0[M]
413.04 BOOL  ; 0[M]
413.05 BOOL  ; RK_12 OK出料拉带启动[M]
413.06 BOOL  ; 0[M]
413.07 BOOL  ; 0[M]
413.08 BOOL  ; 0[M]
413.09 BOOL  ; RK_07 #1铝壳上料电机刹车使能[M]
413.10 BOOL  ; RK_07 #2铝壳上料电机刹车使能[M]
413.11 BOOL  ; RK_07 #3托盘下料电机刹车使能[M]
413.12 BOOL  ; 三色灯_红（公共）[M]
413.13 BOOL  ; 三色灯_绿（公共）[M]
413.14 BOOL  ; 三色灯_黄（公共）[M]
413.15 BOOL  ; 蜂鸣器（公共）[M]
414.00 BOOL  ; RK_06 铝壳上料升降气缸下降[M]
414.01 BOOL  ; RK_06 铝壳上料升降气缸上升[M]
414.02 BOOL  ; RK_06 电池下料升降气缸下降[M]
414.03 BOOL  ; RK_06 电池下料升降气缸上升[M]
414.04 BOOL  ; RK_06 铝壳上料夹爪气缸夹紧[M]
414.05 BOOL  ; RK_06 铝壳上料夹爪气缸张开[M]
414.06 BOOL  ; RK_06 电池下料夹爪气缸夹紧[M]
414.07 BOOL  ; RK_06 电池下料夹爪气缸张开[M]
414.08 BOOL  ; RK_07 #1铝壳上料车定位升降气缸上升[M]
414.09 BOOL  ; RK_07 #1铝壳上料车定位升降气缸下降[M]
414.10 BOOL  ; RK_07 #2铝壳上料车定位升降气缸上升[M]
414.11 BOOL  ; RK_07 #2铝壳上料车定位升降气缸下降[M]
414.12 BOOL  ; RK_07 #3托盘下料车定位升降气缸上升[M]
414.13 BOOL  ; RK_07 #3托盘下料车定位升降气缸下降[M]
414.14 BOOL  ; RK_07 铝壳进料机械手升降气缸下降[M]
414.15 BOOL  ; RK_07 铝壳进料机械手升降气缸上升[M]
415.00 BOOL  ; RK_08 铝壳除尘旋转伸缩气缸缩回[M]
415.01 BOOL  ; RK_08 铝壳除尘旋转伸缩气缸伸出[M]
415.02 BOOL  ; RK_08 铝壳除尘伸缩气缸伸出[M]
415.03 BOOL  ; RK_08 铝壳除尘伸缩气缸缩回[M]
415.04 BOOL  ; RK_08 铝壳除尘夹爪气缸夹紧[M]
415.05 BOOL  ; RK_08 铝壳除尘夹爪气缸张开[M]
415.06 BOOL  ; RK_09 #1Hipot测试旋转伸缩气缸伸出[M]
415.07 BOOL  ; RK_09 #1Hipot测试旋转伸缩气缸缩回[M]
415.08 BOOL  ; RK_09 #1Hipot测试平台伸缩气缸缩回[M]
415.09 BOOL  ; RK_09 #1Hipot测试平台伸缩气缸伸出[M]
415.10 BOOL  ; RK_09 #1Hipot测试伸缩气缸伸出[M]
415.11 BOOL  ; RK_09 #1Hipot测试伸缩气缸缩回[M]
415.12 BOOL  ; RK_09 #2Hipot测试旋转伸缩气缸伸出[M]
415.13 BOOL  ; RK_09 #2Hipot测试旋转伸缩气缸缩回[M]
415.14 BOOL  ; RK_09 #2Hipot测试平台伸缩气缸缩回[M]
415.15 BOOL  ; RK_09 #2Hipot测试平台伸缩气缸伸出[M]
416.00 BOOL  ; RK_09 #2Hipot测试伸缩气缸伸出[M]
416.01 BOOL  ; RK_09 #2Hipot测试伸缩气缸缩回[M]
416.02 BOOL  ; RK_10 电池除尘上料机械手升降气缸下降[M]
416.03 BOOL  ; RK_10 电池除尘上料机械手升降气缸上升[M]
416.04 BOOL  ; RK_10 电池除尘上料机械手夹爪气缸夹紧[M]
416.05 BOOL  ; RK_10 电池除尘上料机械手夹爪气缸张开[M]
416.06 BOOL  ; RK_06 U8_X 电池上下料X轴报警复位[M]
416.07 BOOL  ; RK_06 U8_X 电池上下料X轴使能[M]
416.08 BOOL  ; RK_07 U8_Y 铝壳进料X轴报警复位[M]
416.09 BOOL  ; RK_07 U8_Y 铝壳进料X轴使能[M]
416.10 BOOL  ; RK_07 U8_Z 铝壳上料移载Y轴报警复位[M]
416.11 BOOL  ; RK_07 U8_Z 铝壳上料移载Y轴使能[M]
416.12 BOOL  ; RK_10 U8_U 电池除尘上料X轴报警复位[M]
416.13 BOOL  ; RK_10 U8_U 电池除尘上料X轴使能[M]
416.14 BOOL  ; RK_09 Hipot测试仪远程使能（取消）[M]
416.15 BOOL  ; RK_07 #1铝壳上料启动指示[M]
417.00 BOOL  ; RK_07 #2铝壳上料启动指示[M]
417.01 BOOL  ; RK_07 #3托盘下料启动指示[M]
417.02 BOOL  ; RK_07 铝壳上料移载吸盘立真空[M]
417.03 BOOL  ; RK_07 铝壳进料吸盘立真空[M]
417.04 BOOL  ; RK_07 #1铝壳上料电机正转[M]
417.05 BOOL  ; RK_07 #1铝壳上料电机反转[M]
417.06 BOOL  ; RK_10 Hipot检测NG拉带启动[M]
417.07 BOOL  ; RK_08 铝壳除尘吹气阀开[M]
417.08 BOOL  ; 0[M]
417.09 BOOL  ; RK_07 #2铝壳上料电机正转[M]
417.10 BOOL  ; RK_07 #2铝壳上料电机反转[M]
417.11 BOOL  ; 启动指示_绿（公共）[M]
417.12 BOOL  ; 停止指示_红（公共）[M]
417.13 BOOL  ; 复位指示_黄（公共）[M]
417.14 BOOL  ; RK_07 #3托盘下料电机正转[M]
417.15 BOOL  ; RK_07 #3托盘下料电机反转[M]
421.04 BOOL  ; RK_11 电池除尘吹气阀关[M]
421.14 BOOL  ; RK_14 #1压装吸盘破真空[M]
421.15 BOOL  ; RK_14 #2压装吸盘破真空[M]
423.01 BOOL  ; RK_04 电芯除尘吹气阀关[M]
423.02 BOOL  ; RK_02 扫码NG拉带停止[M]
423.03 BOOL  ; RK_05 #1入壳吸盘破真空[M]
423.04 BOOL  ; RK_05 #2入壳吸盘破真空[M]
423.05 BOOL  ; RK_12 OK出料拉带停止[M]
427.02 BOOL  ; RK_07 铝壳上料移载吸盘破真空[M]
427.03 BOOL  ; RK_07 铝壳进料吸盘破真空[M]
427.04 BOOL  ; RK_07 #1铝壳上料电机停止[M]
427.06 BOOL  ; RK_10 Hipot检测NG拉带停止[M]
427.07 BOOL  ; RK_08 铝壳除尘吹气阀关[M]
427.09 BOOL  ; RK_07 #2铝壳上料电机停止[M]
427.14 BOOL  ; RK_07 #3托盘下料电机停止[M]
449.00 BOOL  ; RK_02 电芯进料机构扫码测试[M]
449.01 BOOL  ; Hipot测试[M]
449.02 BOOL  ; Hipot检测仪参数查询[M]
449.03 BOOL  ; Hipot检测仪参数写入[M]
449.04 BOOL  ; #1移载轮廓测量参数写入[M]
449.05 BOOL  ; #2移载轮廓测量参数写入[M]
449.06 BOOL  ; #1移载#1/4点测量程序切换[M]
449.07 BOOL  ; #1移载#2/3点测量程序切换[M]
449.08 BOOL  ; #2移载#1/4点测量程序切换[M]
449.09 BOOL  ; #2移载#2/3点测量程序切换[M]
449.10 BOOL  ; #1点轮廓测量[M]
449.11 BOOL  ; #2点轮廓测量[M]
449.12 BOOL  ; #3点轮廓测量[M]
449.13 BOOL  ; #4点轮廓测量[M]
449.15 BOOL  ; Hipot检测放电延时参数写入[M]
450.00 BOOL  ; RK_01 U0_X 电芯来料Y轴待料位[M]
450.01 BOOL  ; RK_01 U0_X 电芯来料Y轴上料位[M]
450.02 BOOL  ; RK_01 U0_X 电芯来料Y轴扫码位[M]
450.03 BOOL  ; RK_01 U0_X 电芯来料Y轴下料位[M]
450.04 BOOL  ; 备用[M]
450.05 BOOL  ; 备用[M]
450.06 BOOL  ; 备用[M]
450.07 BOOL  ; 备用[M]
450.08 BOOL  ; 备用[M]
450.09 BOOL  ; 备用[M]
450.10 BOOL  ; RK_01 U0_X 电芯来料Y轴回原点[M]
450.11 BOOL  ; RK_01 U0_X 电芯来料Y轴JOG+[M]
450.12 BOOL  ; RK_01 U0_X 电芯来料Y轴JOG-[M]
450.13 BOOL  ; RK_01 U0_X 电芯来料Y轴JOG高速[M]
450.14 BOOL  ; RK_01 U0_X 电芯来料Y轴JOG低速[M]
450.15 BOOL  ; 备用[M]
451.00 BOOL  ; RK_02 U0_Y 电芯进料X轴待料位[M]
451.01 BOOL  ; RK_02 U0_Y 电芯进料X轴取料位[M]
451.02 BOOL  ; RK_02 U0_Y 电芯进料X轴扫码OK放料位[M]
451.03 BOOL  ; RK_02 U0_Y 电芯进料X轴扫码NG放料位[M]
451.04 BOOL  ; 备用[M]
451.05 BOOL  ; 备用[M]
451.06 BOOL  ; 备用[M]
451.07 BOOL  ; 备用[M]
451.08 BOOL  ; 备用[M]
451.09 BOOL  ; 备用[M]
451.10 BOOL  ; RK_02 U0_Y 电芯进料X轴回原点[M]
451.11 BOOL  ; RK_02 U0_Y 电芯进料X轴JOG+[M]
451.12 BOOL  ; RK_02 U0_Y 电芯进料X轴JOG-[M]
451.13 BOOL  ; RK_02 U0_Y 电芯进料X轴JOG高速[M]
451.14 BOOL  ; RK_02 U0_Y 电芯进料X轴JOG低速[M]
451.15 BOOL  ; 备用[M]
452.00 BOOL  ; RK_02 U0_Z 电芯进料Z轴待料位（扫码）[M]
452.01 BOOL  ; RK_02 U0_Z 电芯进料Z轴取料位[M]
452.02 BOOL  ; RK_02 U0_Z 电芯进料Z轴扫码OK放料位[M]
452.03 BOOL  ; RK_02 U0_Z 电芯进料Z轴扫码NG放料位[M]
452.04 BOOL  ; RK_02 U0_Z 电芯进料Z轴扫码位[M]
452.05 BOOL  ; 备用[M]
452.06 BOOL  ; 备用[M]
452.07 BOOL  ; 备用[M]
452.08 BOOL  ; 备用[M]
452.09 BOOL  ; 备用[M]
452.10 BOOL  ; RK_02 U0_Z 电芯进料Z轴回原点[M]
452.11 BOOL  ; RK_02 U0_Z 电芯进料Z轴JOG+[M]
452.12 BOOL  ; RK_02 U0_Z 电芯进料Z轴JOG-[M]
452.13 BOOL  ; RK_02 U0_Z 电芯进料Z轴JOG高速[M]
452.14 BOOL  ; RK_02 U0_Z 电芯进料Z轴JOG低速[M]
452.15 BOOL  ; 备用[M]
453.00 BOOL  ; RK_03 U0_U 电芯上料X轴待料位[M]
453.01 BOOL  ; RK_03 U0_U 电芯上料X轴取料位[M]
453.02 BOOL  ; RK_03 U0_U 电芯上料X轴#1入壳放料位[M]
453.03 BOOL  ; RK_03 U0_U 电芯上料X轴#2入壳放料位[M]
453.04 BOOL  ; 备用[M]
453.05 BOOL  ; 备用[M]
453.06 BOOL  ; 备用[M]
453.07 BOOL  ; 备用[M]
453.08 BOOL  ; 备用[M]
453.09 BOOL  ; 备用[M]
453.10 BOOL  ; RK_03 U0_U 电芯上料X轴回原点[M]
453.11 BOOL  ; RK_03 U0_U 电芯上料X轴JOG+[M]
453.12 BOOL  ; RK_03 U0_U 电芯上料X轴JOG-[M]
453.13 BOOL  ; RK_03 U0_U 电芯上料X轴JOG高速[M]
453.14 BOOL  ; RK_03 U0_U 电芯上料X轴JOG低速[M]
453.15 BOOL  ; 备用[M]
454.00 BOOL  ; RK_05 U2_X #1入壳Y轴待料位[M]
454.01 BOOL  ; RK_05 U2_X #1入壳Y轴滚轮压紧位[M]
454.02 BOOL  ; RK_05 U2_X #1入壳Y轴滚轮松开位[M]
454.03 BOOL  ; RK_05 U2_X #1入壳Y轴入壳位[M]
454.04 BOOL  ; RK_05 U2_X #1入壳Y轴电芯定位夹爪松开位[M]
454.05 BOOL  ; 备用[M]
454.06 BOOL  ; 备用[M]
454.07 BOOL  ; 备用[M]
454.08 BOOL  ; 备用[M]
454.09 BOOL  ; 备用[M]
454.10 BOOL  ; RK_05 U2_X #1入壳Y轴回原点[M]
454.11 BOOL  ; RK_05 U2_X #1入壳Y轴JOG+[M]
454.12 BOOL  ; RK_05 U2_X #1入壳Y轴JOG-[M]
454.13 BOOL  ; RK_05 U2_X #1入壳Y轴JOG高速[M]
454.14 BOOL  ; RK_05 U2_X #1入壳Y轴JOG低速[M]
454.15 BOOL  ; 备用[M]
455.00 BOOL  ; RK_05 U2_Y #2入壳Y轴待料位[M]
455.01 BOOL  ; RK_05 U2_Y #2入壳Y轴滚轮压紧位[M]
455.02 BOOL  ; RK_05 U2_Y #2入壳Y轴滚轮松开位[M]
455.03 BOOL  ; RK_05 U2_Y #2入壳Y轴入壳位[M]
455.04 BOOL  ; RK_05 U2_Y #2入壳Y轴电芯定位夹爪松开位[M]
455.05 BOOL  ; 备用[M]
455.06 BOOL  ; 备用[M]
455.07 BOOL  ; 备用[M]
455.08 BOOL  ; 备用[M]
455.09 BOOL  ; 备用[M]
455.10 BOOL  ; RK_05 U2_Y #2入壳Y轴回原点[M]
455.11 BOOL  ; RK_05 U2_Y #2入壳Y轴JOG+[M]
455.12 BOOL  ; RK_05 U2_Y #2入壳Y轴JOG-[M]
455.13 BOOL  ; RK_05 U2_Y #2入壳Y轴JOG高速[M]
455.14 BOOL  ; RK_05 U2_Y #2入壳Y轴JOG低速[M]
455.15 BOOL  ; 备用[M]
456.00 BOOL  ; RK_12 U4_X 预焊上下料X轴待料位[M]
456.01 BOOL  ; RK_12 U4_X 预焊上下料X轴除尘取料位[M]
456.02 BOOL  ; RK_12 U4_X 预焊上下料X轴#1移载放料位[M]
456.03 BOOL  ; RK_12 U4_X 预焊上下料X轴#2移载放料位[M]
456.04 BOOL  ; RK_12 U4_X 预焊上下料X轴#1移载取料位[M]
456.05 BOOL  ; RK_12 U4_X 预焊上下料X轴#2移载取料位[M]
456.06 BOOL  ; RK_12 U4_X 预焊上下料X轴OK放料位[M]
456.07 BOOL  ; RK_12 U4_X 预焊上下料X轴#1NG放料位[M]
456.08 BOOL  ; RK_12 U4_X 预焊上下料X轴#2NG放料位[M]
456.09 BOOL  ; 备用[M]
456.10 BOOL  ; RK_12 U4_X 预焊上下料X轴回原点[M]
456.11 BOOL  ; RK_12 U4_X 预焊上下料X轴JOG+[M]
456.12 BOOL  ; RK_12 U4_X 预焊上下料X轴JOG-[M]
456.13 BOOL  ; RK_12 U4_X 预焊上下料X轴JOG高速[M]
456.14 BOOL  ; RK_12 U4_X 预焊上下料X轴JOG低速[M]
456.15 BOOL  ; 备用[M]
457.00 BOOL  ; RK_12 U4_Y 预焊上料Z轴待料位[M]
457.01 BOOL  ; RK_12 U4_Y 预焊上料Z轴除尘取料位[M]
457.02 BOOL  ; RK_12 U4_Y 预焊上料Z轴#1移载放料位[M]
457.03 BOOL  ; RK_12 U4_Y 预焊上料Z轴#2移载放料位[M]
457.04 BOOL  ; 备用[M]
457.05 BOOL  ; 备用[M]
457.06 BOOL  ; 备用[M]
457.07 BOOL  ; 备用[M]
457.08 BOOL  ; 备用[M]
457.09 BOOL  ; 备用[M]
457.10 BOOL  ; RK_12 U4_Y 预焊上料Z轴回原点[M]
457.11 BOOL  ; RK_12 U4_Y 预焊上料Z轴JOG+[M]
457.12 BOOL  ; RK_12 U4_Y 预焊上料Z轴JOG-[M]
457.13 BOOL  ; RK_12 U4_Y 预焊上料Z轴JOG高速[M]
457.14 BOOL  ; RK_12 U4_Y 预焊上料Z轴JOG低速[M]
457.15 BOOL  ; 备用[M]
458.00 BOOL  ; RK_12 U4_Z 预焊下料Z轴待料位[M]
458.01 BOOL  ; RK_12 U4_Z 预焊下料Z轴#1移载取料位[M]
458.02 BOOL  ; RK_12 U4_Z 预焊下料Z轴#2移载取料位[M]
458.03 BOOL  ; RK_12 U4_Z 预焊下料Z轴OK放料位[M]
458.04 BOOL  ; RK_12 U4_Z 预焊下料Z轴#1NG放料位[M]
458.05 BOOL  ; RK_12 U4_Z 预焊下料Z轴#2NG放料位[M]
458.06 BOOL  ; 备用[M]
458.07 BOOL  ; 备用[M]
458.08 BOOL  ; 备用[M]
458.09 BOOL  ; 备用[M]
458.10 BOOL  ; RK_12 U4_Z 预焊下料Z轴回原点[M]
458.11 BOOL  ; RK_12 U4_Z 预焊下料Z轴JOG+[M]
458.12 BOOL  ; RK_12 U4_Z 预焊下料Z轴JOG-[M]
458.13 BOOL  ; RK_12 U4_Z 预焊下料Z轴JOG高速[M]
458.14 BOOL  ; RK_12 U4_Z 预焊下料Z轴JOG低速[M]
458.15 BOOL  ; 备用[M]
459.00 BOOL  ; RK_13 U4_U #1移载Y轴待料位[M]
459.01 BOOL  ; RK_13 U4_U #1移载Y轴取放料位[M]
459.02 BOOL  ; RK_13 U4_U #1移载Y轴压装位[M]
459.03 BOOL  ; RK_13 U4_U #1移载Y轴#1轮廓检测位[M]
459.04 BOOL  ; RK_13 U4_U #1移载Y轴#2轮廓检测位[M]
459.05 BOOL  ; RK_13 U4_U #1移载Y轴激光焊接位[M]
459.06 BOOL  ; 备用[M]
459.07 BOOL  ; 备用[M]
459.08 BOOL  ; 备用[M]
459.09 BOOL  ; 备用[M]
459.10 BOOL  ; RK_13 U4_U #1移载Y轴回原点[M]
459.11 BOOL  ; RK_13 U4_U #1移载Y轴JOG+[M]
459.12 BOOL  ; RK_13 U4_U #1移载Y轴JOG-[M]
459.13 BOOL  ; RK_13 U4_U #1移载Y轴JOG高速[M]
459.14 BOOL  ; RK_13 U4_U #1移载Y轴JOG低速[M]
459.15 BOOL  ; 备用[M]
460.00 BOOL  ; RK_13 U6_X #2移载Y轴待料位[M]
460.01 BOOL  ; RK_13 U6_X #2移载Y轴取放料位[M]
460.02 BOOL  ; RK_13 U6_X #2移载Y轴压装位[M]
460.03 BOOL  ; $?St$Bk?_#[5049] / RK_13 U6_X #2移载Y轴#1轮廓检测位[M] / $?St$Bk?_#[5049]
460.04 BOOL  ; RK_13 U6_X #2移载Y轴#2轮廓检测位[M]
460.05 BOOL  ; RK_13 U6_X #2移载Y轴激光焊接位[M]
460.06 BOOL  ; 备用[M]
460.07 BOOL  ; 备用[M]
460.08 BOOL  ; 备用[M]
460.09 BOOL  ; 备用[M]
460.10 BOOL  ; RK_13 U6_X #2移载Y轴回原点[M]
460.11 BOOL  ; RK_13 U6_X #2移载Y轴JOG+[M]
460.12 BOOL  ; RK_13 U6_X #2移载Y轴JOG-[M]
460.13 BOOL  ; RK_13 U6_X #2移载Y轴JOG高速[M]
460.14 BOOL  ; RK_13 U6_X #2移载Y轴JOG低速[M]
460.15 BOOL  ; 备用[M]
461.00 BOOL  ; RK_16 U6_Y 激光焊接X轴待机位[M]
461.01 BOOL  ; RK_16 U6_Y 激光焊接X轴#1移载焊接位[M]
461.02 BOOL  ; RK_16 U6_Y 激光焊接X轴#2移载焊接位[M]
461.03 BOOL  ; 备用[M]
461.04 BOOL  ; 备用[M]
461.05 BOOL  ; 备用[M]
461.06 BOOL  ; 备用[M]
461.07 BOOL  ; 备用[M]
461.08 BOOL  ; 备用[M]
461.09 BOOL  ; 备用[M]
461.10 BOOL  ; RK_16 U6_Y 激光焊接X轴回原点[M]
461.11 BOOL  ; RK_16 U6_Y 激光焊接X轴JOG+[M]
461.12 BOOL  ; RK_16 U6_Y 激光焊接X轴JOG-[M]
461.13 BOOL  ; RK_16 U6_Y 激光焊接X轴JOG高速[M]
461.14 BOOL  ; RK_16 U6_Y 激光焊接X轴JOG低速[M]
461.15 BOOL  ; 备用[M]
462.00 BOOL  ; RK_16 U6_Z 激光焊接Z轴待机位[M]
462.01 BOOL  ; RK_16 U6_Z 激光焊接Z轴#1移载焊接位[M]
462.02 BOOL  ; RK_16 U6_Z 激光焊接Z轴#2移载焊接位[M]
462.03 BOOL  ; 备用[M]
462.04 BOOL  ; 备用[M]
462.05 BOOL  ; 备用[M]
462.06 BOOL  ; 备用[M]
462.07 BOOL  ; 备用[M]
462.08 BOOL  ; 备用[M]
462.09 BOOL  ; 备用[M]
462.10 BOOL  ; RK_16 U6_Z 激光焊接Z轴回原点[M]
462.11 BOOL  ; RK_16 U6_Z 激光焊接Z轴JOG+[M]
462.12 BOOL  ; RK_16 U6_Z 激光焊接Z轴JOG-[M]
462.13 BOOL  ; RK_16 U6_Z 激光焊接Z轴JOG高速[M]
462.14 BOOL  ; RK_16 U6_Z 激光焊接Z轴JOG低速[M]
462.15 BOOL  ; 备用[M]
463.00 BOOL  ; RK_06 U8_X 电池上下料X轴待机位[M]
463.01 BOOL  ; RK_06 U8_X 电池上下料X轴铝壳除尘取料位[M]
463.02 BOOL  ; RK_06 U8_X 电池上下料X轴#1入壳放料位[M]
463.03 BOOL  ; RK_06 U8_X 电池上下料X轴#2入壳放料位[M]
463.04 BOOL  ; RK_06 U8_X 电池上下料X轴#1入壳取料位[M]
463.05 BOOL  ; RK_06 U8_X 电池上下料X轴#2入壳取料位[M]
463.06 BOOL  ; RK_06 U8_X 电池上下料X轴#1Hipot检测放料位[M]
463.07 BOOL  ; RK_06 U8_X 电池上下料X轴#2Hipot检测放料位[M]
463.08 BOOL  ; 备用[M]
463.09 BOOL  ; 备用[M]
463.10 BOOL  ; RK_06 U8_X 电池上下料X轴回原点[M]
463.11 BOOL  ; RK_06 U8_X 电池上下料X轴JOG+[M]
463.12 BOOL  ; RK_06 U8_X 电池上下料X轴JOG-[M]
463.13 BOOL  ; RK_06 U8_X 电池上下料X轴JOG高速[M]
463.14 BOOL  ; RK_06 U8_X 电池上下料X轴JOG低速[M]
463.15 BOOL  ; 备用[M]
464.00 BOOL  ; RK_07 U8_Y 铝壳进料X轴等待位[M]
464.01 BOOL  ; RK_07 U8_Y 铝壳进料X轴取料位[M]
464.02 BOOL  ; RK_07 U8_Y 铝壳进料X轴放料位[M]
464.03 BOOL  ; 备用[M]
464.04 BOOL  ; 备用[M]
464.05 BOOL  ; 备用[M]
464.06 BOOL  ; 备用[M]
464.07 BOOL  ; 备用[M]
464.08 BOOL  ; 备用[M]
464.09 BOOL  ; 备用[M]
464.10 BOOL  ; RK_07 U8_Y 铝壳进料X轴回原点[M]
464.11 BOOL  ; RK_07 U8_Y 铝壳进料X轴JOG+[M]
464.12 BOOL  ; RK_07 U8_Y 铝壳进料X轴JOG-[M]
464.13 BOOL  ; RK_07 U8_Y 铝壳进料X轴JOG高速[M]
464.14 BOOL  ; RK_07 U8_Y 铝壳进料X轴JOG低速[M]
464.15 BOOL  ; 备用[M]
465.00 BOOL  ; RK_07 U8_Z 铝壳上料移载Y轴待料位[M]
465.01 BOOL  ; RK_07 U8_Z 铝壳上料移载Y轴#1铝壳上料位[M]
465.02 BOOL  ; RK_07 U8_Z 铝壳上料移载Y轴#2铝壳上料位[M]
465.03 BOOL  ; RK_07 U8_Z 铝壳上料移载Y轴#3铝壳托盘下料位[M]
465.04 BOOL  ; RK_07 U8_Z 铝壳上料移载Y轴铝壳取料位[M]
465.05 BOOL  ; 备用[M]
465.06 BOOL  ; 备用[M]
465.07 BOOL  ; 备用[M]
465.08 BOOL  ; 备用[M]
465.09 BOOL  ; 备用[M]
465.10 BOOL  ; RK_07 U8_Z 铝壳上料移载Y轴回原点[M]
465.11 BOOL  ; RK_07 U8_Z 铝壳上料移载Y轴JOG+[M]
465.12 BOOL  ; RK_07 U8_Z 铝壳上料移载Y轴JOG-[M]
465.13 BOOL  ; RK_07 U8_Z 铝壳上料移载Y轴JOG高速[M]
465.14 BOOL  ; RK_07 U8_Z 铝壳上料移载Y轴JOG低速[M]
465.15 BOOL  ; 备用[M]
466.00 BOOL  ; RK_10 U8_U 电池除尘上料X轴待料位[M]
466.01 BOOL  ; RK_10 U8_U 电池除尘上料X轴#1Hipot检测取料位[M]
466.02 BOOL  ; RK_10 U8_U 电池除尘上料X轴#2Hipot检测取料位[M]
466.03 BOOL  ; RK_10 U8_U 电池除尘上料X轴Hipot OK放料位[M]
466.04 BOOL  ; RK_10 U8_U 电池除尘上料X轴Hipot NG放料位[M]
466.05 BOOL  ; 备用[M]
466.06 BOOL  ; 备用[M]
466.07 BOOL  ; 备用[M]
466.08 BOOL  ; 备用[M]
466.09 BOOL  ; 备用[M]
466.10 BOOL  ; RK_10 U8_U 电池除尘上料X轴回原点[M]
466.11 BOOL  ; RK_10 U8_U 电池除尘上料X轴JOG+[M]
466.12 BOOL  ; RK_10 U8_U 电池除尘上料X轴JOG-[M]
466.13 BOOL  ; RK_10 U8_U 电池除尘上料X轴JOG高速[M]
466.14 BOOL  ; RK_10 U8_U 电池除尘上料X轴JOG低速[M]
466.15 BOOL  ; 备用[M]
4.00 BOOL  ; RK_05 #2入壳定位陶瓷棒上#2夹紧气缸伸出位
4.01 BOOL  ; RK_05 #2入壳定位陶瓷棒下#1夹紧气缸伸出位
4.02 BOOL  ; RK_05 #2入壳定位陶瓷棒下#2夹紧气缸伸出位
4.03 BOOL  ; RK_05 #2入壳定位陶瓷棒上#1夹紧气缸缩回位
4.04 BOOL  ; RK_05 #2入壳定位陶瓷棒上#2夹紧气缸缩回位
4.05 BOOL  ; RK_05 #2入壳定位陶瓷棒下#1夹紧气缸缩回位
4.06 BOOL  ; RK_05 #2入壳定位陶瓷棒下#2夹紧气缸缩回位
4.07 BOOL  ; RK_05 #2入壳吸盘上#1伸缩气缸缩回位
4.08 BOOL  ; RK_05 #2入壳吸盘上#2伸缩气缸缩回位
4.09 BOOL  ; RK_05 #2入壳吸盘上#3伸缩气缸缩回位
4.10 BOOL  ; RK_05 #2入壳吸盘下#1伸缩气缸缩回位
4.11 BOOL  ; RK_05 #2入壳吸盘下#2伸缩气缸缩回位
4.12 BOOL  ; RK_05 #2入壳吸盘下#3伸缩气缸缩回位
4.13 BOOL  ; RK_05 #2入壳电芯#1定位夹爪气缸松开位
4.14 BOOL  ; RK_05 #2入壳电芯#2定位夹爪气缸松开位
4.15 BOOL  ; RK_05 #2入壳电芯#1定位夹爪气缸夹紧位
500.00 BOOL  ; RK_02 电芯进料机械手夹爪气缸夹紧条件
500.01 BOOL  ; RK_02 电芯进料机械手夹爪气缸张开条件
500.02 BOOL  ; RK_02 电芯进料机械手压紧气缸伸出条件
500.03 BOOL  ; RK_02 电芯进料机械手压紧气缸缩回条件
500.04 BOOL  ; RK_03 电芯上料机械手夹爪气缸夹紧条件
500.05 BOOL  ; RK_03 电芯上料机械手夹爪气缸张开条件
500.06 BOOL  ; RK_03 电芯上料机械手压紧气缸伸出条件
500.07 BOOL  ; RK_03 电芯上料机械手压紧气缸缩回条件
500.08 BOOL  ; RK_03 电芯上料升降气缸下降条件
500.09 BOOL  ; RK_03 电芯上料升降气缸上升条件
500.10 BOOL  ; RK_04 电芯除尘伸缩气缸缩回条件
500.11 BOOL  ; RK_04 电芯除尘伸缩气缸伸出条件
500.12 BOOL  ; RK_05 #1入壳滚轮夹紧气缸伸出条件
500.13 BOOL  ; RK_05 #1入壳滚轮夹紧气缸缩回条件
500.14 BOOL  ; RK_05 #1入壳铝壳定位平台伸缩气缸缩回条件
500.15 BOOL  ; RK_05 #1入壳铝壳定位平台伸缩气缸伸出条件
501.00 BOOL  ; RK_05 #1入壳铝壳定位平台升降气缸上升条件
501.01 BOOL  ; RK_05 #1入壳铝壳定位平台升降气缸下降条件
501.02 BOOL  ; RK_05 #1入壳铝壳定位伸缩气缸缩回条件
501.03 BOOL  ; RK_05 #1入壳铝壳定位伸缩气缸伸出条件
501.04 BOOL  ; RK_05 #1入壳铝壳定位夹爪气缸夹紧条件
501.05 BOOL  ; RK_05 #1入壳铝壳定位夹爪气缸张开条件
501.06 BOOL  ; RK_05 #2入壳滚轮夹紧气缸伸出条件
501.07 BOOL  ; RK_05 #2入壳滚轮夹紧气缸缩回条件
501.08 BOOL  ; RK_05 #2入壳铝壳定位平台伸缩气缸缩回条件
501.09 BOOL  ; RK_05 #2入壳铝壳定位平台伸缩气缸伸出条件
501.10 BOOL  ; RK_05 #2入壳铝壳定位平台升降气缸上升条件
501.11 BOOL  ; RK_05 #2入壳铝壳定位平台升降气缸下降条件
501.12 BOOL  ; RK_05 #2入壳铝壳定位伸缩气缸缩回条件
501.13 BOOL  ; RK_05 #2入壳铝壳定位伸缩气缸伸出条件
501.14 BOOL  ; RK_05 #2入壳铝壳定位夹爪气缸夹紧条件
501.15 BOOL  ; RK_05 #2入壳铝壳定位夹爪气缸张开条件
502.00 BOOL  ; RK_01 U0_X 电芯来料Y轴报警复位条件
502.01 BOOL  ; RK_01 U0_X 电芯来料Y轴使能条件
502.02 BOOL  ; RK_02 U0_Y 电芯进料X轴报警复位条件
502.03 BOOL  ; RK_02 U0_Y 电芯进料X轴使能条件
502.04 BOOL  ; RK_02 U0_Z 电芯进料Z轴报警复位条件
502.05 BOOL  ; RK_02 U0_Z 电芯进料Z轴使能条件
502.06 BOOL  ; RK_03 U0_U 电芯上料X轴报警复位条件
502.07 BOOL  ; RK_03 U0_U 电芯上料X轴使能条件
502.08 BOOL  ; RK_05 U2_X #1入壳Y轴报警复位条件
502.09 BOOL  ; RK_05 U2_X #1入壳Y轴使能条件
502.10 BOOL  ; RK_05 U2_Y #2入壳Y轴报警复位条件
502.11 BOOL  ; RK_05 U2_Y #2入壳Y轴使能条件
502.12 BOOL  ; RK_02 电芯进料Z轴刹车使能条件
502.13 BOOL  ; RK_05 #1入壳定位陶瓷棒夹紧气缸伸出条件
502.14 BOOL  ; RK_05 #1入壳定位陶瓷棒夹紧气缸缩回条件
502.15 BOOL  ; RK_05 #2入壳定位陶瓷棒夹紧气缸伸出条件
503.00 BOOL  ; RK_05 #2入壳定位陶瓷棒夹紧气缸缩回条件
503.01 BOOL  ; RK_04 电芯除尘吹气阀开条件
503.02 BOOL  ; RK_02 扫码NG拉带启动条件
503.03 BOOL  ; RK_05 #1入壳吸盘立真空条件
503.04 BOOL  ; RK_05 #2入壳吸盘立真空条件
503.05 BOOL  ; RK_05 #1入壳吸盘伸缩气缸伸出条件
503.06 BOOL  ; RK_05 #1入壳吸盘伸缩气缸缩回条件
503.07 BOOL  ; RK_05 #2入壳吸盘伸缩气缸伸出条件
503.08 BOOL  ; RK_05 #2入壳吸盘伸缩气缸缩回条件
503.09 BOOL  ; 前端设备对接输出信号（公共）条件
503.10 BOOL  ; 后端设备对接输出信号（公共）条件
503.11 BOOL  ; RK_05 #1入壳电芯定位夹爪气缸伸出条件
503.12 BOOL  ; RK_05 #1入壳电芯定位夹爪气缸缩回条件
503.13 BOOL  ; RK_05 #2入壳电芯定位夹爪气缸伸出条件
503.14 BOOL  ; RK_05 #2入壳电芯定位夹爪气缸缩回条件
508.00 BOOL  ; RK_11 电池除尘旋转伸缩气缸缩回条件
508.01 BOOL  ; RK_11 电池除尘旋转伸缩气缸伸出条件
508.02 BOOL  ; RK_11 电池除尘伸缩气缸伸出条件
508.03 BOOL  ; RK_11 电池除尘伸缩气缸缩回条件
508.04 BOOL  ; RK_11 电池除尘夹爪气缸夹紧条件
508.05 BOOL  ; RK_11 电池除尘夹爪气缸张开条件
508.06 BOOL  ; RK_12 预焊上料机械手夹爪气缸夹紧条件
508.07 BOOL  ; RK_12 预焊上料机械手夹爪气缸张开条件
508.08 BOOL  ; RK_12 预焊下料机械手夹爪气缸夹紧条件
508.09 BOOL  ; RK_12 预焊下料机械手夹爪气缸张开条件
508.10 BOOL  ; RK_13 #1移载升降气缸上升条件
508.11 BOOL  ; RK_13 #1移载升降气缸下降条件
508.12 BOOL  ; RK_13 #1移载定位#1伸缩气缸缩回条件
508.13 BOOL  ; RK_13 #1移载定位#1伸缩气缸伸出条件
508.14 BOOL  ; RK_13 #1移载定位#2伸缩气缸缩回条件
508.15 BOOL  ; RK_13 #1移载定位#2伸缩气缸伸出条件
509.00 BOOL  ; RK_13 #1移载导向#1伸缩气缸伸出条件
509.01 BOOL  ; RK_13 #1移载导向#1伸缩气缸缩回条件
509.02 BOOL  ; RK_13 #1移载导向#2伸缩气缸伸出条件
509.03 BOOL  ; RK_13 #1移载导向#2伸缩气缸缩回条件
509.04 BOOL  ; RK_13 #1移载左右定位伸缩气缸伸出条件
509.05 BOOL  ; RK_13 #1移载左右定位伸缩气缸缩回条件
509.06 BOOL  ; RK_13 #2移载升降气缸上升条件
509.07 BOOL  ; RK_13 #2移载升降气缸下降条件
509.08 BOOL  ; RK_13 #2移载定位#1伸缩气缸缩回条件
509.09 BOOL  ; RK_13 #2移载定位#1伸缩气缸伸出条件
509.10 BOOL  ; RK_13 #2移载定位#2伸缩气缸缩回条件
509.11 BOOL  ; RK_13 #2移载定位#2伸缩气缸伸出条件
509.12 BOOL  ; RK_13 #2移载导向#1伸缩气缸伸出条件
509.13 BOOL  ; RK_13 #2移载导向#1伸缩气缸缩回条件
509.14 BOOL  ; RK_13 #2移载导向#2伸缩气缸伸出条件
509.15 BOOL  ; RK_13 #2移载导向#2伸缩气缸缩回条件
50.00 BOOL  ; RK_01 U0_X 电芯来料Y轴待料位
50.01 BOOL  ; RK_01 U0_X 电芯来料Y轴上料位
50.02 BOOL  ; RK_01 U0_X 电芯来料Y轴扫码位
50.03 BOOL  ; RK_01 U0_X 电芯来料Y轴下料位
50.04 BOOL  ; 备用
50.05 BOOL  ; 备用
50.06 BOOL  ; 备用
50.07 BOOL  ; 备用
50.08 BOOL  ; 备用
50.09 BOOL  ; 备用
510.00 BOOL  ; RK_13 #2移载左右定位伸缩气缸伸出条件
510.01 BOOL  ; RK_13 #2移载左右定位伸缩气缸缩回条件
510.02 BOOL  ; RK_14 #1压装升降气缸下降条件
510.03 BOOL  ; RK_14 #1压装升降气缸上升条件
510.04 BOOL  ; RK_14 #1压装#1吸盘升降气缸下降条件
510.05 BOOL  ; RK_14 #1压装#1吸盘升降气缸上升条件
510.06 BOOL  ; RK_14 #1压装#2吸盘升降气缸下降条件
510.07 BOOL  ; RK_14 #1压装#2吸盘升降气缸上升条件
510.08 BOOL  ; RK_14 #2压装升降气缸下降条件
510.09 BOOL  ; RK_14 #2压装升降气缸上升条件
510.10 BOOL  ; RK_14 #2压装#1吸盘升降气缸下降条件
510.11 BOOL  ; RK_14 #2压装#1吸盘升降气缸上升条件
510.12 BOOL  ; RK_14 #2压装#2吸盘升降气缸下降条件
510.13 BOOL  ; RK_14 #2压装#2吸盘升降气缸上升条件
510.14 BOOL  ; RK_15 轮廓检测#1伸缩气缸伸出条件
510.15 BOOL  ; RK_15 轮廓检测#1伸缩气缸缩回条件
511.00 BOOL  ; RK_15 轮廓检测#2伸缩气缸伸出条件
511.01 BOOL  ; RK_15 轮廓检测#2伸缩气缸缩回条件
511.02 BOOL  ; RK_12 轮廓检测NG拨料气缸伸出条件
511.03 BOOL  ; RK_12 轮廓检测NG拨料气缸缩回条件
511.04 BOOL  ; RK_11 电池除尘吹气阀开条件
511.05 BOOL  ; 0条件
511.06 BOOL  ; 0条件
511.07 BOOL  ; RK_16 激光焊接触发条件
511.08 BOOL  ; RK_16 PLC急停输出到激光设备条件
511.09 BOOL  ; RK_16 #1移载激光焊任务选择条件
511.10 BOOL  ; RK_16 #2移载激光焊任务选择条件
511.11 BOOL  ; RK_16 集尘器启动条件
511.12 BOOL  ; 0条件
511.13 BOOL  ; 0条件
511.14 BOOL  ; RK_14 #1压装吸盘立真空条件
511.15 BOOL  ; RK_14 #2压装吸盘立真空条件
512.00 BOOL  ; RK_12 U4_X 预焊上下料X轴报警复位条件
512.01 BOOL  ; RK_12 U4_X 预焊上下料X轴使能条件
512.02 BOOL  ; RK_12 U4_Y 预焊上料Z轴报警复位条件
512.03 BOOL  ; RK_12 U4_Y 预焊上料Z轴使能条件
512.04 BOOL  ; RK_12 U4_Z 预焊下料Z轴报警复位条件
512.05 BOOL  ; RK_12 U4_Z 预焊下料Z轴使能条件
512.06 BOOL  ; RK_13 U4_U #1移载Y轴报警复位条件
512.07 BOOL  ; RK_13 U4_U #1移载Y轴使能条件
512.08 BOOL  ; RK_13 U6_X #2移载Y轴报警复位条件
512.09 BOOL  ; RK_13 U6_X #2移载Y轴使能条件
512.10 BOOL  ; RK_16 U6_Y 激光焊接X轴报警复位条件
512.11 BOOL  ; RK_16 U6_Y 激光焊接X轴使能条件
512.12 BOOL  ; RK_16 U6_Z 激光焊接Z轴报警复位条件
512.13 BOOL  ; RK_16 U6_Z 激光焊接Z轴使能条件
512.14 BOOL  ; RK_12 预焊上料Z轴刹车使能条件
512.15 BOOL  ; RK_12 预焊下料Z轴刹车使能条件
513.00 BOOL  ; RK_16 激光焊接Z轴刹车使能条件
513.01 BOOL  ; 0条件
513.02 BOOL  ; 0条件
513.03 BOOL  ; 0条件
513.04 BOOL  ; 0条件
513.05 BOOL  ; RK_12 OK出料拉带启动条件
513.06 BOOL  ; 0条件
513.07 BOOL  ; 0条件
513.08 BOOL  ; 0条件
513.09 BOOL  ; RK_07 #1铝壳上料电机刹车使能条件
513.10 BOOL  ; RK_07 #2铝壳上料电机刹车使能条件
513.11 BOOL  ; RK_07 #3托盘下料电机刹车使能条件
513.12 BOOL  ; 三色灯_红（公共）条件
513.13 BOOL  ; 三色灯_绿（公共）条件
513.14 BOOL  ; 三色灯_黄（公共）条件
513.15 BOOL  ; 蜂鸣器（公共）条件
514.00 BOOL  ; RK_06 铝壳上料升降气缸下降条件
514.01 BOOL  ; RK_06 铝壳上料升降气缸上升条件
514.02 BOOL  ; RK_06 电池下料升降气缸下降条件
514.03 BOOL  ; RK_06 电池下料升降气缸上升条件
514.04 BOOL  ; RK_06 铝壳上料夹爪气缸夹紧条件
514.05 BOOL  ; RK_06 铝壳上料夹爪气缸张开条件
514.06 BOOL  ; RK_06 电池下料夹爪气缸夹紧条件
514.07 BOOL  ; RK_06 电池下料夹爪气缸张开条件
514.08 BOOL  ; RK_07 #1铝壳上料车定位升降气缸上升条件
514.09 BOOL  ; RK_07 #1铝壳上料车定位升降气缸下降条件
514.10 BOOL  ; RK_07 #2铝壳上料车定位升降气缸上升条件
514.11 BOOL  ; RK_07 #2铝壳上料车定位升降气缸下降条件
514.12 BOOL  ; RK_07 #3托盘下料车定位升降气缸上升条件
514.13 BOOL  ; RK_07 #3托盘下料车定位升降气缸下降条件
514.14 BOOL  ; RK_07 铝壳进料机械手升降气缸下降条件
514.15 BOOL  ; RK_07 铝壳进料机械手升降气缸上升条件
515.00 BOOL  ; RK_08 铝壳除尘旋转伸缩气缸缩回条件
515.01 BOOL  ; RK_08 铝壳除尘旋转伸缩气缸伸出条件
515.02 BOOL  ; RK_08 铝壳除尘伸缩气缸伸出条件
515.03 BOOL  ; RK_08 铝壳除尘伸缩气缸缩回条件
515.04 BOOL  ; RK_08 铝壳除尘夹爪气缸夹紧条件
515.05 BOOL  ; RK_08 铝壳除尘夹爪气缸张开条件
515.06 BOOL  ; RK_09 #1Hipot测试旋转伸缩气缸伸出条件
515.07 BOOL  ; RK_09 #1Hipot测试旋转伸缩气缸缩回条件
515.08 BOOL  ; RK_09 #1Hipot测试平台伸缩气缸缩回条件
515.09 BOOL  ; RK_09 #1Hipot测试平台伸缩气缸伸出条件
515.10 BOOL  ; RK_09 #1Hipot测试伸缩气缸伸出条件
515.11 BOOL  ; RK_09 #1Hipot测试伸缩气缸缩回条件
515.12 BOOL  ; RK_09 #2Hipot测试旋转伸缩气缸伸出条件
515.13 BOOL  ; RK_09 #2Hipot测试旋转伸缩气缸缩回条件
515.14 BOOL  ; RK_09 #2Hipot测试平台伸缩气缸缩回条件
515.15 BOOL  ; RK_09 #2Hipot测试平台伸缩气缸伸出条件
516.00 BOOL  ; RK_09 #2Hipot测试伸缩气缸伸出条件
516.01 BOOL  ; RK_09 #2Hipot测试伸缩气缸缩回条件
516.02 BOOL  ; RK_10 电池除尘上料机械手升降气缸下降条件
516.03 BOOL  ; RK_10 电池除尘上料机械手升降气缸上升条件
516.04 BOOL  ; RK_10 电池除尘上料机械手夹爪气缸夹紧条件
516.05 BOOL  ; RK_10 电池除尘上料机械手夹爪气缸张开条件
516.06 BOOL  ; RK_06 U8_X 电池上下料X轴报警复位条件
516.07 BOOL  ; RK_06 U8_X 电池上下料X轴使能条件
516.08 BOOL  ; RK_07 U8_Y 铝壳进料X轴报警复位条件
516.09 BOOL  ; RK_07 U8_Y 铝壳进料X轴使能条件
516.10 BOOL  ; RK_07 U8_Z 铝壳上料移载Y轴报警复位条件
516.11 BOOL  ; RK_07 U8_Z 铝壳上料移载Y轴使能条件
516.12 BOOL  ; RK_10 U8_U 电池除尘上料X轴报警复位条件
516.13 BOOL  ; RK_10 U8_U 电池除尘上料X轴使能条件
516.14 BOOL  ; RK_09 Hipot测试仪远程使能（取消）条件
516.15 BOOL  ; RK_07 #1铝壳上料启动指示条件
517.00 BOOL  ; RK_07 #2铝壳上料启动指示条件
517.01 BOOL  ; RK_07 #3托盘下料启动指示条件
517.02 BOOL  ; RK_07 铝壳上料移载吸盘立真空条件
517.03 BOOL  ; RK_07 铝壳进料吸盘立真空条件
517.04 BOOL  ; RK_07 #1铝壳上料电机正转条件
517.05 BOOL  ; RK_07 #1铝壳上料电机反转条件
517.06 BOOL  ; RK_10 Hipot检测NG拉带启动条件
517.07 BOOL  ; RK_08 铝壳除尘吹气阀开条件
517.08 BOOL  ; 0条件
517.09 BOOL  ; RK_07 #2铝壳上料电机正转条件
517.10 BOOL  ; RK_07 #2铝壳上料电机反转条件
517.11 BOOL  ; 启动指示_绿（公共）条件
517.12 BOOL  ; 停止指示_红（公共）条件
517.13 BOOL  ; 复位指示_黄（公共）条件
517.14 BOOL  ; RK_07 #3托盘下料电机正转条件
517.15 BOOL  ; RK_07 #3托盘下料电机反转条件
51.00 BOOL  ; RK_02 U0_Y 电芯进料X轴待料位
51.01 BOOL  ; RK_02 U0_Y 电芯进料X轴取料位
51.02 BOOL  ; RK_02 U0_Y 电芯进料X轴扫码OK放料位
51.03 BOOL  ; RK_02 U0_Y 电芯进料X轴扫码NG放料位
51.04 BOOL  ; 备用
51.05 BOOL  ; 备用
51.06 BOOL  ; 备用
51.07 BOOL  ; 备用
51.08 BOOL  ; 备用
51.09 BOOL  ; 备用
521.04 BOOL  ; RK_11 电池除尘吹气阀关条件
521.14 BOOL  ; RK_14 #1压装吸盘破真空条件
521.15 BOOL  ; RK_14 #2压装吸盘破真空条件
523.01 BOOL  ; RK_04 电芯除尘吹气阀关条件
523.02 BOOL  ; RK_02 扫码NG拉带停止条件
523.03 BOOL  ; RK_05 #1入壳吸盘破真空条件
523.04 BOOL  ; RK_05 #2入壳吸盘破真空条件
523.05 BOOL  ; RK_12 OK出料拉带停止条件
527.02 BOOL  ; RK_07 铝壳上料移载吸盘破真空条件
527.03 BOOL  ; RK_07 铝壳进料吸盘破真空条件
527.04 BOOL  ; RK_07 #1铝壳上料电机停止条件
527.06 BOOL  ; RK_10 Hipot检测NG拉带停止条件
527.07 BOOL  ; RK_08 铝壳除尘吹气阀关条件
527.09 BOOL  ; RK_07 #2铝壳上料电机停止条件
527.14 BOOL  ; RK_07 #3托盘下料电机停止条件
52.00 BOOL  ; RK_02 U0_Z 电芯进料Z轴待料位（扫码）
52.01 BOOL  ; RK_02 U0_Z 电芯进料Z轴取料位
52.02 BOOL  ; RK_02 U0_Z 电芯进料Z轴扫码OK放料位
52.03 BOOL  ; RK_02 U0_Z 电芯进料Z轴扫码NG放料位
52.04 BOOL  ; RK_02 U0_Z 电芯进料Z轴扫码位
52.05 BOOL  ; 备用
52.06 BOOL  ; 备用
52.07 BOOL  ; 备用
52.08 BOOL  ; 备用
52.09 BOOL  ; 备用
53.00 BOOL  ; RK_03 U0_U 电芯上料X轴待料位
53.01 BOOL  ; RK_03 U0_U 电芯上料X轴取料位
53.02 BOOL  ; RK_03 U0_U 电芯上料X轴#1入壳放料位
53.03 BOOL  ; RK_03 U0_U 电芯上料X轴#2入壳放料位
53.04 BOOL  ; 备用
53.05 BOOL  ; 备用
53.06 BOOL  ; 备用
53.07 BOOL  ; 备用
53.08 BOOL  ; 备用
53.09 BOOL  ; 备用
54.00 BOOL  ; RK_05 U2_X #1入壳Y轴待料位
54.01 BOOL  ; RK_05 U2_X #1入壳Y轴滚轮压紧位
54.02 BOOL  ; RK_05 U2_X #1入壳Y轴滚轮松开位
54.03 BOOL  ; RK_05 U2_X #1入壳Y轴入壳位
54.04 BOOL  ; RK_05 U2_X #1入壳Y轴电芯定位夹爪松开位
54.05 BOOL  ; 备用
54.06 BOOL  ; 备用
54.07 BOOL  ; 备用
54.08 BOOL  ; 备用
54.09 BOOL  ; 备用
550.00 BOOL  ; RK_01 U0_X 电芯来料Y轴待料位条件
550.01 BOOL  ; RK_01 U0_X 电芯来料Y轴上料位条件
550.02 BOOL  ; RK_01 U0_X 电芯来料Y轴扫码位条件
550.03 BOOL  ; RK_01 U0_X 电芯来料Y轴下料位条件
550.04 BOOL  ; 备用条件
550.05 BOOL  ; 备用条件
550.06 BOOL  ; 备用条件
550.07 BOOL  ; 备用条件
550.08 BOOL  ; 备用条件
550.09 BOOL  ; 备用条件
550.10 BOOL  ; RK_01 U0_X 电芯来料Y轴回原点条件
550.11 BOOL  ; RK_01 U0_X 电芯来料Y轴JOG+条件
550.12 BOOL  ; RK_01 U0_X 电芯来料Y轴JOG-条件
550.13 BOOL  ; RK_01 U0_X 电芯来料Y轴JOG高速条件
550.14 BOOL  ; RK_01 U0_X 电芯来料Y轴JOG低速条件
550.15 BOOL  ; 备用条件
551.00 BOOL  ; RK_02 U0_Y 电芯进料X轴待料位条件
551.01 BOOL  ; RK_02 U0_Y 电芯进料X轴取料位条件
551.02 BOOL  ; RK_02 U0_Y 电芯进料X轴扫码OK放料位条件
551.03 BOOL  ; RK_02 U0_Y 电芯进料X轴扫码NG放料位条件
551.04 BOOL  ; 备用条件
551.05 BOOL  ; 备用条件
551.06 BOOL  ; 备用条件
551.07 BOOL  ; 备用条件
551.08 BOOL  ; 备用条件
551.09 BOOL  ; 备用条件
551.10 BOOL  ; RK_02 U0_Y 电芯进料X轴回原点条件
551.11 BOOL  ; RK_02 U0_Y 电芯进料X轴JOG+条件
551.12 BOOL  ; RK_02 U0_Y 电芯进料X轴JOG-条件
551.13 BOOL  ; RK_02 U0_Y 电芯进料X轴JOG高速条件
551.14 BOOL  ; RK_02 U0_Y 电芯进料X轴JOG低速条件
551.15 BOOL  ; 备用条件
552.00 BOOL  ; RK_02 U0_Z 电芯进料Z轴待料位（扫码）条件
552.01 BOOL  ; RK_02 U0_Z 电芯进料Z轴取料位条件
552.02 BOOL  ; RK_02 U0_Z 电芯进料Z轴扫码OK放料位条件
552.03 BOOL  ; RK_02 U0_Z 电芯进料Z轴扫码NG放料位条件
552.04 BOOL  ; RK_02 U0_Z 电芯进料Z轴扫码位条件
552.05 BOOL  ; 备用条件
552.06 BOOL  ; 备用条件
552.07 BOOL  ; 备用条件
552.08 BOOL  ; 备用条件
552.09 BOOL  ; 备用条件
552.10 BOOL  ; RK_02 U0_Z 电芯进料Z轴回原点条件
552.11 BOOL  ; RK_02 U0_Z 电芯进料Z轴JOG+条件
552.12 BOOL  ; RK_02 U0_Z 电芯进料Z轴JOG-条件
552.13 BOOL  ; RK_02 U0_Z 电芯进料Z轴JOG高速条件
552.14 BOOL  ; RK_02 U0_Z 电芯进料Z轴JOG低速条件
552.15 BOOL  ; 备用条件
553.00 BOOL  ; RK_03 U0_U 电芯上料X轴待料位条件
553.01 BOOL  ; RK_03 U0_U 电芯上料X轴取料位条件
553.02 BOOL  ; RK_03 U0_U 电芯上料X轴#1入壳放料位条件
553.03 BOOL  ; RK_03 U0_U 电芯上料X轴#2入壳放料位条件
553.04 BOOL  ; 备用条件
553.05 BOOL  ; 备用条件
553.06 BOOL  ; 备用条件
553.07 BOOL  ; 备用条件
553.08 BOOL  ; 备用条件
553.09 BOOL  ; 备用条件
553.10 BOOL  ; RK_03 U0_U 电芯上料X轴回原点条件
553.11 BOOL  ; RK_03 U0_U 电芯上料X轴JOG+条件
553.12 BOOL  ; RK_03 U0_U 电芯上料X轴JOG-条件
553.13 BOOL  ; RK_03 U0_U 电芯上料X轴JOG高速条件
553.14 BOOL  ; RK_03 U0_U 电芯上料X轴JOG低速条件
553.15 BOOL  ; 备用条件
554.00 BOOL  ; RK_05 U2_X #1入壳Y轴待料位条件
554.01 BOOL  ; RK_05 U2_X #1入壳Y轴滚轮压紧位条件
554.02 BOOL  ; RK_05 U2_X #1入壳Y轴滚轮松开位条件
554.03 BOOL  ; RK_05 U2_X #1入壳Y轴入壳位条件
554.04 BOOL  ; RK_05 U2_X #1入壳Y轴电芯定位夹爪松开位条件
554.05 BOOL  ; 备用条件
554.06 BOOL  ; 备用条件
554.07 BOOL  ; 备用条件
554.08 BOOL  ; 备用条件
554.09 BOOL  ; 备用条件
554.10 BOOL  ; RK_05 U2_X #1入壳Y轴回原点条件
554.11 BOOL  ; RK_05 U2_X #1入壳Y轴JOG+条件
554.12 BOOL  ; RK_05 U2_X #1入壳Y轴JOG-条件
554.13 BOOL  ; RK_05 U2_X #1入壳Y轴JOG高速条件
554.14 BOOL  ; RK_05 U2_X #1入壳Y轴JOG低速条件
554.15 BOOL  ; 备用条件
555.00 BOOL  ; RK_05 U2_Y #2入壳Y轴待料位条件
555.01 BOOL  ; RK_05 U2_Y #2入壳Y轴滚轮压紧位条件
555.02 BOOL  ; RK_05 U2_Y #2入壳Y轴滚轮松开位条件
555.03 BOOL  ; RK_05 U2_Y #2入壳Y轴入壳位条件
555.04 BOOL  ; RK_05 U2_Y #2入壳Y轴电芯定位夹爪松开位条件
555.05 BOOL  ; 备用条件
555.06 BOOL  ; 备用条件
555.07 BOOL  ; 备用条件
555.08 BOOL  ; 备用条件
555.09 BOOL  ; 备用条件
555.10 BOOL  ; RK_05 U2_Y #2入壳Y轴回原点条件
555.11 BOOL  ; RK_05 U2_Y #2入壳Y轴JOG+条件
555.12 BOOL  ; RK_05 U2_Y #2入壳Y轴JOG-条件
555.13 BOOL  ; RK_05 U2_Y #2入壳Y轴JOG高速条件
555.14 BOOL  ; RK_05 U2_Y #2入壳Y轴JOG低速条件
555.15 BOOL  ; 备用条件
556.00 BOOL  ; RK_12 U4_X 预焊上下料X轴待料位条件
556.01 BOOL  ; RK_12 U4_X 预焊上下料X轴除尘取料位条件
556.02 BOOL  ; RK_12 U4_X 预焊上下料X轴#1移载放料位条件
556.03 BOOL  ; RK_12 U4_X 预焊上下料X轴#2移载放料位条件
556.04 BOOL  ; RK_12 U4_X 预焊上下料X轴#1移载取料位条件
556.05 BOOL  ; RK_12 U4_X 预焊上下料X轴#2移载取料位条件
556.06 BOOL  ; RK_12 U4_X 预焊上下料X轴OK放料位条件
556.07 BOOL  ; RK_12 U4_X 预焊上下料X轴#1NG放料位条件
556.08 BOOL  ; RK_12 U4_X 预焊上下料X轴#2NG放料位条件
556.09 BOOL  ; 备用条件
556.10 BOOL  ; RK_12 U4_X 预焊上下料X轴回原点条件
556.11 BOOL  ; RK_12 U4_X 预焊上下料X轴JOG+条件
556.12 BOOL  ; RK_12 U4_X 预焊上下料X轴JOG-条件
556.13 BOOL  ; RK_12 U4_X 预焊上下料X轴JOG高速条件
556.14 BOOL  ; RK_12 U4_X 预焊上下料X轴JOG低速条件
556.15 BOOL  ; 备用条件
557.00 BOOL  ; RK_12 U4_Y 预焊上料Z轴待料位条件
557.01 BOOL  ; RK_12 U4_Y 预焊上料Z轴除尘取料位条件
557.02 BOOL  ; RK_12 U4_Y 预焊上料Z轴#1移载放料位条件
557.03 BOOL  ; RK_12 U4_Y 预焊上料Z轴#2移载放料位条件
557.04 BOOL  ; 备用条件
557.05 BOOL  ; 备用条件
557.06 BOOL  ; 备用条件
557.07 BOOL  ; 备用条件
557.08 BOOL  ; 备用条件
557.09 BOOL  ; 备用条件
557.10 BOOL  ; RK_12 U4_Y 预焊上料Z轴回原点条件
557.11 BOOL  ; RK_12 U4_Y 预焊上料Z轴JOG+条件
557.12 BOOL  ; RK_12 U4_Y 预焊上料Z轴JOG-条件
557.13 BOOL  ; RK_12 U4_Y 预焊上料Z轴JOG高速条件
557.14 BOOL  ; RK_12 U4_Y 预焊上料Z轴JOG低速条件
557.15 BOOL  ; 备用条件
558.00 BOOL  ; RK_12 U4_Z 预焊下料Z轴待料位条件
558.01 BOOL  ; RK_12 U4_Z 预焊下料Z轴#1移载取料位条件
558.02 BOOL  ; RK_12 U4_Z 预焊下料Z轴#2移载取料位条件
558.03 BOOL  ; RK_12 U4_Z 预焊下料Z轴OK放料位条件
558.04 BOOL  ; RK_12 U4_Z 预焊下料Z轴#1NG放料位条件
558.05 BOOL  ; RK_12 U4_Z 预焊下料Z轴#2NG放料位条件
558.06 BOOL  ; 备用条件
558.07 BOOL  ; 备用条件
558.08 BOOL  ; 备用条件
558.09 BOOL  ; 备用条件
558.10 BOOL  ; RK_12 U4_Z 预焊下料Z轴回原点条件
558.11 BOOL  ; RK_12 U4_Z 预焊下料Z轴JOG+条件
558.12 BOOL  ; RK_12 U4_Z 预焊下料Z轴JOG-条件
558.13 BOOL  ; RK_12 U4_Z 预焊下料Z轴JOG高速条件
558.14 BOOL  ; RK_12 U4_Z 预焊下料Z轴JOG低速条件
558.15 BOOL  ; 备用条件
559.00 BOOL  ; RK_13 U4_U #1移载Y轴待料位条件
559.01 BOOL  ; RK_13 U4_U #1移载Y轴取放料位条件
559.02 BOOL  ; RK_13 U4_U #1移载Y轴压装位条件
559.03 BOOL  ; RK_13 U4_U #1移载Y轴#1轮廓检测位条件
559.04 BOOL  ; RK_13 U4_U #1移载Y轴#2轮廓检测位条件
559.05 BOOL  ; RK_13 U4_U #1移载Y轴激光焊接位条件
559.06 BOOL  ; 备用条件
559.07 BOOL  ; 备用条件
559.08 BOOL  ; 备用条件
559.09 BOOL  ; 备用条件
559.10 BOOL  ; RK_13 U4_U #1移载Y轴回原点条件
559.11 BOOL  ; RK_13 U4_U #1移载Y轴JOG+条件
559.12 BOOL  ; RK_13 U4_U #1移载Y轴JOG-条件
559.13 BOOL  ; RK_13 U4_U #1移载Y轴JOG高速条件
559.14 BOOL  ; RK_13 U4_U #1移载Y轴JOG低速条件
559.15 BOOL  ; 备用条件
55.00 BOOL  ; RK_05 U2_Y #2入壳Y轴待料位
55.01 BOOL  ; RK_05 U2_Y #2入壳Y轴滚轮压紧位
55.02 BOOL  ; RK_05 U2_Y #2入壳Y轴滚轮松开位
55.03 BOOL  ; RK_05 U2_Y #2入壳Y轴入壳位
55.04 BOOL  ; RK_05 U2_Y #2入壳Y轴电芯定位夹爪松开位
55.05 BOOL  ; 备用
55.06 BOOL  ; 备用
55.07 BOOL  ; 备用
55.08 BOOL  ; 备用
55.09 BOOL  ; 备用
560.00 BOOL  ; RK_13 U6_X #2移载Y轴待料位条件
560.01 BOOL  ; RK_13 U6_X #2移载Y轴取放料位条件
560.02 BOOL  ; RK_13 U6_X #2移载Y轴压装位条件
560.03 BOOL  ; RK_13 U6_X #2移载Y轴#1轮廓检测位条件
560.04 BOOL  ; RK_13 U6_X #2移载Y轴#2轮廓检测位条件
560.05 BOOL  ; RK_13 U6_X #2移载Y轴激光焊接位条件
560.06 BOOL  ; 备用条件
560.07 BOOL  ; 备用条件
560.08 BOOL  ; 备用条件
560.09 BOOL  ; 备用条件
560.10 BOOL  ; RK_13 U6_X #2移载Y轴回原点条件
560.11 BOOL  ; RK_13 U6_X #2移载Y轴JOG+条件
560.12 BOOL  ; RK_13 U6_X #2移载Y轴JOG-条件
560.13 BOOL  ; RK_13 U6_X #2移载Y轴JOG高速条件
560.14 BOOL  ; RK_13 U6_X #2移载Y轴JOG低速条件
560.15 BOOL  ; 备用条件
561.00 BOOL  ; RK_16 U6_Y 激光焊接X轴待机位条件
561.01 BOOL  ; RK_16 U6_Y 激光焊接X轴#1移载焊接位条件
561.02 BOOL  ; RK_16 U6_Y 激光焊接X轴#2移载焊接位条件
561.03 BOOL  ; 备用条件
561.04 BOOL  ; 备用条件
561.05 BOOL  ; 备用条件
561.06 BOOL  ; 备用条件
561.07 BOOL  ; 备用条件
561.08 BOOL  ; 备用条件
561.09 BOOL  ; 备用条件
561.10 BOOL  ; RK_16 U6_Y 激光焊接X轴回原点条件
561.11 BOOL  ; RK_16 U6_Y 激光焊接X轴JOG+条件
561.12 BOOL  ; RK_16 U6_Y 激光焊接X轴JOG-条件
561.13 BOOL  ; RK_16 U6_Y 激光焊接X轴JOG高速条件
561.14 BOOL  ; RK_16 U6_Y 激光焊接X轴JOG低速条件
561.15 BOOL  ; 备用条件
562.00 BOOL  ; RK_16 U6_Z 激光焊接Z轴待机位条件
562.01 BOOL  ; RK_16 U6_Z 激光焊接Z轴#1移载焊接位条件
562.02 BOOL  ; RK_16 U6_Z 激光焊接Z轴#2移载焊接位条件
562.03 BOOL  ; 备用条件
562.04 BOOL  ; 备用条件
562.05 BOOL  ; 备用条件
562.06 BOOL  ; 备用条件
562.07 BOOL  ; 备用条件
562.08 BOOL  ; 备用条件
562.09 BOOL  ; 备用条件
562.10 BOOL  ; RK_16 U6_Z 激光焊接Z轴回原点条件
562.11 BOOL  ; RK_16 U6_Z 激光焊接Z轴JOG+条件
562.12 BOOL  ; RK_16 U6_Z 激光焊接Z轴JOG-条件
562.13 BOOL  ; RK_16 U6_Z 激光焊接Z轴JOG高速条件
562.14 BOOL  ; RK_16 U6_Z 激光焊接Z轴JOG低速条件
562.15 BOOL  ; 备用条件
563.00 BOOL  ; RK_06 U8_X 电池上下料X轴待机位条件
563.01 BOOL  ; RK_06 U8_X 电池上下料X轴铝壳除尘取料位条件
563.02 BOOL  ; RK_06 U8_X 电池上下料X轴#1入壳放料位条件
563.03 BOOL  ; RK_06 U8_X 电池上下料X轴#2入壳放料位条件
563.04 BOOL  ; RK_06 U8_X 电池上下料X轴#1入壳取料位条件
563.05 BOOL  ; RK_06 U8_X 电池上下料X轴#2入壳取料位条件
563.06 BOOL  ; RK_06 U8_X 电池上下料X轴#1Hipot检测放料位条件
563.07 BOOL  ; RK_06 U8_X 电池上下料X轴#2Hipot检测放料位条件
563.08 BOOL  ; 备用条件
563.09 BOOL  ; 备用条件
563.10 BOOL  ; RK_06 U8_X 电池上下料X轴回原点条件
563.11 BOOL  ; RK_06 U8_X 电池上下料X轴JOG+条件
563.12 BOOL  ; RK_06 U8_X 电池上下料X轴JOG-条件
563.13 BOOL  ; RK_06 U8_X 电池上下料X轴JOG高速条件
563.14 BOOL  ; RK_06 U8_X 电池上下料X轴JOG低速条件
563.15 BOOL  ; 备用条件
564.00 BOOL  ; RK_07 U8_Y 铝壳进料X轴等待位条件
564.01 BOOL  ; RK_07 U8_Y 铝壳进料X轴取料位条件
564.02 BOOL  ; RK_07 U8_Y 铝壳进料X轴放料位条件
564.03 BOOL  ; 备用条件
564.04 BOOL  ; 备用条件
564.05 BOOL  ; 备用条件
564.06 BOOL  ; 备用条件
564.07 BOOL  ; 备用条件
564.08 BOOL  ; 备用条件
564.09 BOOL  ; 备用条件
564.10 BOOL  ; RK_07 U8_Y 铝壳进料X轴回原点条件
564.11 BOOL  ; RK_07 U8_Y 铝壳进料X轴JOG+条件
564.12 BOOL  ; RK_07 U8_Y 铝壳进料X轴JOG-条件
564.13 BOOL  ; RK_07 U8_Y 铝壳进料X轴JOG高速条件
564.14 BOOL  ; RK_07 U8_Y 铝壳进料X轴JOG低速条件
564.15 BOOL  ; 备用条件
565.00 BOOL  ; RK_07 U8_Z 铝壳上料移载Y轴待料位条件
565.01 BOOL  ; RK_07 U8_Z 铝壳上料移载Y轴#1铝壳上料位条件
565.02 BOOL  ; RK_07 U8_Z 铝壳上料移载Y轴#2铝壳上料位条件
565.03 BOOL  ; RK_07 U8_Z 铝壳上料移载Y轴#3铝壳托盘下料位条件
565.04 BOOL  ; RK_07 U8_Z 铝壳上料移载Y轴铝壳取料位条件
565.05 BOOL  ; 备用条件
565.06 BOOL  ; 备用条件
565.07 BOOL  ; 备用条件
565.08 BOOL  ; 备用条件
565.09 BOOL  ; 备用条件
565.10 BOOL  ; RK_07 U8_Z 铝壳上料移载Y轴回原点条件
565.11 BOOL  ; RK_07 U8_Z 铝壳上料移载Y轴JOG+条件
565.12 BOOL  ; RK_07 U8_Z 铝壳上料移载Y轴JOG-条件
565.13 BOOL  ; RK_07 U8_Z 铝壳上料移载Y轴JOG高速条件
565.14 BOOL  ; RK_07 U8_Z 铝壳上料移载Y轴JOG低速条件
565.15 BOOL  ; 备用条件
566.00 BOOL  ; RK_10 U8_U 电池除尘上料X轴待料位条件
566.01 BOOL  ; RK_10 U8_U 电池除尘上料X轴#1Hipot检测取料位条件
566.02 BOOL  ; RK_10 U8_U 电池除尘上料X轴#2Hipot检测取料位条件
566.03 BOOL  ; RK_10 U8_U 电池除尘上料X轴Hipot OK放料位条件
566.04 BOOL  ; RK_10 U8_U 电池除尘上料X轴Hipot NG放料位条件
566.05 BOOL  ; 备用条件
566.06 BOOL  ; 备用条件
566.07 BOOL  ; 备用条件
566.08 BOOL  ; 备用条件
566.09 BOOL  ; 备用条件
566.10 BOOL  ; RK_10 U8_U 电池除尘上料X轴回原点条件
566.11 BOOL  ; RK_10 U8_U 电池除尘上料X轴JOG+条件
566.12 BOOL  ; RK_10 U8_U 电池除尘上料X轴JOG-条件
566.13 BOOL  ; RK_10 U8_U 电池除尘上料X轴JOG高速条件
566.14 BOOL  ; RK_10 U8_U 电池除尘上料X轴JOG低速条件
566.15 BOOL  ; 备用条件
56.00 BOOL  ; RK_12 U4_X 预焊上下料X轴待料位
56.01 BOOL  ; RK_12 U4_X 预焊上下料X轴除尘取料位
56.02 BOOL  ; RK_12 U4_X 预焊上下料X轴#1移载放料位
56.03 BOOL  ; RK_12 U4_X 预焊上下料X轴#2移载放料位
56.04 BOOL  ; RK_12 U4_X 预焊上下料X轴#1移载取料位
56.05 BOOL  ; RK_12 U4_X 预焊上下料X轴#2移载取料位
56.06 BOOL  ; RK_12 U4_X 预焊上下料X轴OK放料位
56.07 BOOL  ; RK_12 U4_X 预焊上下料X轴#1NG放料位
56.08 BOOL  ; RK_12 U4_X 预焊上下料X轴#2NG放料位
56.09 BOOL  ; 备用
57.00 BOOL  ; RK_12 U4_Y 预焊上料Z轴待料位
57.01 BOOL  ; RK_12 U4_Y 预焊上料Z轴除尘取料位
57.02 BOOL  ; RK_12 U4_Y 预焊上料Z轴#1移载放料位
57.03 BOOL  ; RK_12 U4_Y 预焊上料Z轴#2移载放料位
57.04 BOOL  ; 备用
57.05 BOOL  ; 备用
57.06 BOOL  ; 备用
57.07 BOOL  ; 备用
57.08 BOOL  ; 备用
57.09 BOOL  ; 备用
58.00 BOOL  ; RK_12 U4_Z 预焊下料Z轴待料位
58.01 BOOL  ; RK_12 U4_Z 预焊下料Z轴#1移载取料位
58.02 BOOL  ; RK_12 U4_Z 预焊下料Z轴#2移载取料位
58.03 BOOL  ; RK_12 U4_Z 预焊下料Z轴OK放料位
58.04 BOOL  ; RK_12 U4_Z 预焊下料Z轴#1NG放料位
58.05 BOOL  ; RK_12 U4_Z 预焊下料Z轴#2NG放料位
58.06 BOOL  ; 备用
58.07 BOOL  ; 备用
58.08 BOOL  ; 备用
58.09 BOOL  ; 备用
59.00 BOOL  ; RK_13 U4_U #1移载Y轴待料位
59.01 BOOL  ; RK_13 U4_U #1移载Y轴取放料位
59.02 BOOL  ; RK_13 U4_U #1移载Y轴压装位
59.03 BOOL  ; RK_13 U4_U #1移载Y轴#1轮廓检测位
59.04 BOOL  ; RK_13 U4_U #1移载Y轴#2轮廓检测位
59.05 BOOL  ; RK_13 U4_U #1移载Y轴激光焊接位
59.06 BOOL  ; 备用
59.07 BOOL  ; 备用
59.08 BOOL  ; 备用
59.09 BOOL  ; 备用
5.00 BOOL  ; RK_05 #2入壳电芯#2定位夹爪气缸夹紧位
5.01 BOOL  ; RK_01 电芯来料有料感应
5.02 BOOL  ; RK_02 电芯进料机械手夹爪柔性报警
5.03 BOOL  ; RK_03 电芯上料机械手夹爪柔性报警
5.04 BOOL  ; RK_04 电芯除尘有料感应
5.05 BOOL  ; RK_02 扫码NG拉带有料感应#1
5.06 BOOL  ; RK_02 扫码NG拉带有料感应#2
5.07 BOOL  ; RK_02 扫码NG拉带料满感应
5.08 BOOL  ; RK_05 #1入壳电芯有料感应
5.09 BOOL  ; RK_05 #1入壳铝壳有料感应
5.10 BOOL  ; RK_05 #2入壳电芯有料感应
5.11 BOOL  ; RK_05 #2入壳铝壳有料感应
5.12 BOOL  ; RK_05 #1入壳吸盘真空
5.13 BOOL  ; RK_05 #2入壳吸盘真空
5.14 BOOL  ; 前端设备对接输入信号（公共）
5.15 BOOL  ; 后端设备对接输入信号（公共）
6000.00 BOOL  ; 扫码阻挡#1伸出手动按钮
6000.01 BOOL  ; 扫码阻挡#1缩回手动按钮
6000.02 BOOL  ; 扫码阻挡#2伸出手动按钮
6000.03 BOOL  ; 扫码阻挡#2缩回手动按钮
6000.15 BOOL  ; 出料气缸复位
6001.00 BOOL  ; 扫码阻挡#1伸出手动输出
6001.01 BOOL  ; 扫码阻挡#1缩回手动输出
6001.02 BOOL  ; 扫码阻挡#2伸出手动输出
6001.03 BOOL  ; 扫码阻挡#2缩回手动输出
6002 CHANNEL  ; *出料拉带新增自动段
6002.00 BOOL  ; 流程初始化状态检测
6002.01 BOOL  ; 扫码位物料等待
6002.02 BOOL  ; 扫码阻挡伸出
6002.03 BOOL  ; 等待扫码完成
6002.04 BOOL  ; 扫码位物料可流出判定
6002.05 BOOL  ; 扫码隔离缩回
6002.06 BOOL  ; 物料流出到位等待
6002.07 BOOL  ; 扫码隔离伸出&阻挡缩回
6002.08 BOOL  ; 扫码气缸循环结束
600.00 BOOL  ; RK_02 电芯进料机械手夹爪气缸夹紧[A]
600.01 BOOL  ; RK_02 电芯进料机械手夹爪气缸张开[A]
600.02 BOOL  ; RK_02 电芯进料机械手压紧气缸伸出[A]
600.03 BOOL  ; RK_02 电芯进料机械手压紧气缸缩回[A]
600.04 BOOL  ; RK_03 电芯上料机械手夹爪气缸夹紧[A]
600.05 BOOL  ; RK_03 电芯上料机械手夹爪气缸张开[A]
600.06 BOOL  ; RK_03 电芯上料机械手压紧气缸伸出[A]
600.07 BOOL  ; RK_03 电芯上料机械手压紧气缸缩回[A]
600.08 BOOL  ; RK_03 电芯上料升降气缸下降[A]
600.09 BOOL  ; RK_03 电芯上料升降气缸上升[A]
600.10 BOOL  ; RK_04 电芯除尘伸缩气缸缩回[A]
600.11 BOOL  ; RK_04 电芯除尘伸缩气缸伸出[A]
600.12 BOOL  ; RK_05 #1入壳滚轮夹紧气缸伸出[A]
600.13 BOOL  ; RK_05 #1入壳滚轮夹紧气缸缩回[A]
600.14 BOOL  ; RK_05 #1入壳铝壳定位平台伸缩气缸缩回[A]
600.15 BOOL  ; RK_05 #1入壳铝壳定位平台伸缩气缸伸出[A]
601.00 BOOL  ; RK_05 #1入壳铝壳定位平台升降气缸上升[A]
601.01 BOOL  ; RK_05 #1入壳铝壳定位平台升降气缸下降[A]
601.02 BOOL  ; RK_05 #1入壳铝壳定位伸缩气缸缩回[A]
601.03 BOOL  ; RK_05 #1入壳铝壳定位伸缩气缸伸出[A]
601.04 BOOL  ; RK_05 #1入壳铝壳定位夹爪气缸夹紧[A]
601.05 BOOL  ; RK_05 #1入壳铝壳定位夹爪气缸张开[A]
601.06 BOOL  ; RK_05 #2入壳滚轮夹紧气缸伸出[A]
601.07 BOOL  ; RK_05 #2入壳滚轮夹紧气缸缩回[A]
601.08 BOOL  ; RK_05 #2入壳铝壳定位平台伸缩气缸缩回[A]
601.09 BOOL  ; RK_05 #2入壳铝壳定位平台伸缩气缸伸出[A]
601.10 BOOL  ; RK_05 #2入壳铝壳定位平台升降气缸上升[A]
601.11 BOOL  ; RK_05 #2入壳铝壳定位平台升降气缸下降[A]
601.12 BOOL  ; RK_05 #2入壳铝壳定位伸缩气缸缩回[A]
601.13 BOOL  ; RK_05 #2入壳铝壳定位伸缩气缸伸出[A]
601.14 BOOL  ; RK_05 #2入壳铝壳定位夹爪气缸夹紧[A]
601.15 BOOL  ; RK_05 #2入壳铝壳定位夹爪气缸张开[A]
602.00 BOOL  ; RK_01 U0_X 电芯来料Y轴报警复位[A]
602.01 BOOL  ; RK_01 U0_X 电芯来料Y轴使能[A]
602.02 BOOL  ; RK_02 U0_Y 电芯进料X轴报警复位[A]
602.03 BOOL  ; RK_02 U0_Y 电芯进料X轴使能[A]
602.04 BOOL  ; RK_02 U0_Z 电芯进料Z轴报警复位[A]
602.05 BOOL  ; RK_02 U0_Z 电芯进料Z轴使能[A]
602.06 BOOL  ; RK_03 U0_U 电芯上料X轴报警复位[A]
602.07 BOOL  ; RK_03 U0_U 电芯上料X轴使能[A]
602.08 BOOL  ; RK_05 U2_X #1入壳Y轴报警复位[A]
602.09 BOOL  ; RK_05 U2_X #1入壳Y轴使能[A]
602.10 BOOL  ; RK_05 U2_Y #2入壳Y轴报警复位[A]
602.11 BOOL  ; RK_05 U2_Y #2入壳Y轴使能[A]
602.12 BOOL  ; RK_02 电芯进料Z轴刹车使能[A]
602.13 BOOL  ; RK_05 #1入壳定位陶瓷棒夹紧气缸伸出[A]
602.14 BOOL  ; RK_05 #1入壳定位陶瓷棒夹紧气缸缩回[A]
602.15 BOOL  ; RK_05 #2入壳定位陶瓷棒夹紧气缸伸出[A]
603.00 BOOL  ; RK_05 #2入壳定位陶瓷棒夹紧气缸缩回[A]
603.01 BOOL  ; RK_04 电芯除尘吹气阀开[A]
603.02 BOOL  ; RK_02 扫码NG拉带启动[A]
603.03 BOOL  ; RK_05 #1入壳吸盘立真空[A]
603.04 BOOL  ; RK_05 #2入壳吸盘立真空[A]
603.05 BOOL  ; RK_05 #1入壳吸盘伸缩气缸伸出[A]
603.06 BOOL  ; RK_05 #1入壳吸盘伸缩气缸缩回[A]
603.07 BOOL  ; RK_05 #2入壳吸盘伸缩气缸伸出[A]
603.08 BOOL  ; RK_05 #2入壳吸盘伸缩气缸缩回[A]
603.09 BOOL  ; 前端设备对接输出信号（公共）[A]
603.10 BOOL  ; 后端设备对接输出信号（公共）[A]
603.11 BOOL  ; RK_05 #1入壳电芯定位夹爪气缸伸出[A]
603.12 BOOL  ; RK_05 #1入壳电芯定位夹爪气缸缩回[A]
603.13 BOOL  ; RK_05 #2入壳电芯定位夹爪气缸伸出[A]
603.14 BOOL  ; RK_05 #2入壳电芯定位夹爪气缸缩回[A]
608.00 BOOL  ; RK_11 电池除尘旋转伸缩气缸缩回[A]
608.01 BOOL  ; RK_11 电池除尘旋转伸缩气缸伸出[A]
608.02 BOOL  ; RK_11 电池除尘伸缩气缸伸出[A]
608.03 BOOL  ; RK_11 电池除尘伸缩气缸缩回[A]
608.04 BOOL  ; RK_11 电池除尘夹爪气缸夹紧[A]
608.05 BOOL  ; RK_11 电池除尘夹爪气缸张开[A]
608.06 BOOL  ; RK_12 预焊上料机械手夹爪气缸夹紧[A]
608.07 BOOL  ; RK_12 预焊上料机械手夹爪气缸张开[A]
608.08 BOOL  ; RK_12 预焊下料机械手夹爪气缸夹紧[A]
608.09 BOOL  ; RK_12 预焊下料机械手夹爪气缸张开[A]
608.10 BOOL  ; RK_13 #1移载升降气缸上升[A]
608.11 BOOL  ; RK_13 #1移载升降气缸下降[A]
608.12 BOOL  ; RK_13 #1移载定位#1伸缩气缸缩回[A]
608.13 BOOL  ; RK_13 #1移载定位#1伸缩气缸伸出[A]
608.14 BOOL  ; RK_13 #1移载定位#2伸缩气缸缩回[A]
608.15 BOOL  ; RK_13 #1移载定位#2伸缩气缸伸出[A]
609.00 BOOL  ; RK_13 #1移载导向#1伸缩气缸伸出[A]
609.01 BOOL  ; RK_13 #1移载导向#1伸缩气缸缩回[A]
609.02 BOOL  ; RK_13 #1移载导向#2伸缩气缸伸出[A]
609.03 BOOL  ; RK_13 #1移载导向#2伸缩气缸缩回[A]
609.04 BOOL  ; RK_13 #1移载左右定位伸缩气缸伸出[A]
609.05 BOOL  ; RK_13 #1移载左右定位伸缩气缸缩回[A]
609.06 BOOL  ; RK_13 #2移载升降气缸上升[A]
609.07 BOOL  ; RK_13 #2移载升降气缸下降[A]
609.08 BOOL  ; RK_13 #2移载定位#1伸缩气缸缩回[A]
609.09 BOOL  ; RK_13 #2移载定位#1伸缩气缸伸出[A]
609.10 BOOL  ; RK_13 #2移载定位#2伸缩气缸缩回[A]
609.11 BOOL  ; RK_13 #2移载定位#2伸缩气缸伸出[A]
609.12 BOOL  ; RK_13 #2移载导向#1伸缩气缸伸出[A]
609.13 BOOL  ; RK_13 #2移载导向#1伸缩气缸缩回[A]
609.14 BOOL  ; RK_13 #2移载导向#2伸缩气缸伸出[A]
609.15 BOOL  ; RK_13 #2移载导向#2伸缩气缸缩回[A]
60.00 BOOL  ; RK_13 U6_X #2移载Y轴待料位
60.01 BOOL  ; RK_13 U6_X #2移载Y轴取放料位
60.02 BOOL  ; RK_13 U6_X #2移载Y轴压装位
60.03 BOOL  ; RK_13 U6_X #2移载Y轴#1轮廓检测位
60.04 BOOL  ; RK_13 U6_X #2移载Y轴#2轮廓检测位
60.05 BOOL  ; RK_13 U6_X #2移载Y轴激光焊接位
60.06 BOOL  ; 备用
60.07 BOOL  ; 备用
60.08 BOOL  ; 备用
60.09 BOOL  ; 备用
610.00 BOOL  ; RK_13 #2移载左右定位伸缩气缸伸出[A]
610.01 BOOL  ; RK_13 #2移载左右定位伸缩气缸缩回[A]
610.02 BOOL  ; RK_14 #1压装升降气缸下降[A]
610.03 BOOL  ; RK_14 #1压装升降气缸上升[A]
610.04 BOOL  ; RK_14 #1压装#1吸盘升降气缸下降[A]
610.05 BOOL  ; RK_14 #1压装#1吸盘升降气缸上升[A]
610.06 BOOL  ; RK_14 #1压装#2吸盘升降气缸下降[A]
610.07 BOOL  ; RK_14 #1压装#2吸盘升降气缸上升[A]
610.08 BOOL  ; RK_14 #2压装升降气缸下降[A]
610.09 BOOL  ; RK_14 #2压装升降气缸上升[A]
610.10 BOOL  ; RK_14 #2压装#1吸盘升降气缸下降[A]
610.11 BOOL  ; RK_14 #2压装#1吸盘升降气缸上升[A]
610.12 BOOL  ; RK_14 #2压装#2吸盘升降气缸下降[A]
610.13 BOOL  ; RK_14 #2压装#2吸盘升降气缸上升[A]
610.14 BOOL  ; RK_15 轮廓检测#1伸缩气缸伸出[A]
610.15 BOOL  ; RK_15 轮廓检测#1伸缩气缸缩回[A]
611.00 BOOL  ; RK_15 轮廓检测#2伸缩气缸伸出[A]
611.01 BOOL  ; RK_15 轮廓检测#2伸缩气缸缩回[A]
611.02 BOOL  ; RK_12 轮廓检测NG拨料气缸伸出[A]
611.03 BOOL  ; RK_12 轮廓检测NG拨料气缸缩回[A]
611.04 BOOL  ; RK_11 电池除尘吹气阀开[A]
611.05 BOOL  ; 0[A]
611.06 BOOL  ; 0[A]
611.07 BOOL  ; RK_16 激光焊接触发[A]
611.08 BOOL  ; RK_16 PLC急停输出到激光设备[A]
611.09 BOOL  ; RK_16 #1移载激光焊任务选择[A]
611.10 BOOL  ; RK_16 #2移载激光焊任务选择[A]
611.11 BOOL  ; RK_16 集尘器启动[A]
611.12 BOOL  ; 0[A]
611.13 BOOL  ; 0[A]
611.14 BOOL  ; RK_14 #1压装吸盘立真空[A]
611.15 BOOL  ; RK_14 #2压装吸盘立真空[A]
612.00 BOOL  ; RK_12 U4_X 预焊上下料X轴报警复位[A]
612.01 BOOL  ; RK_12 U4_X 预焊上下料X轴使能[A]
612.02 BOOL  ; RK_12 U4_Y 预焊上料Z轴报警复位[A]
612.03 BOOL  ; RK_12 U4_Y 预焊上料Z轴使能[A]
612.04 BOOL  ; RK_12 U4_Z 预焊下料Z轴报警复位[A]
612.05 BOOL  ; RK_12 U4_Z 预焊下料Z轴使能[A]
612.06 BOOL  ; RK_13 U4_U #1移载Y轴报警复位[A]
612.07 BOOL  ; RK_13 U4_U #1移载Y轴使能[A]
612.08 BOOL  ; RK_13 U6_X #2移载Y轴报警复位[A]
612.09 BOOL  ; RK_13 U6_X #2移载Y轴使能[A]
612.10 BOOL  ; RK_16 U6_Y 激光焊接X轴报警复位[A]
612.11 BOOL  ; RK_16 U6_Y 激光焊接X轴使能[A]
612.12 BOOL  ; RK_16 U6_Z 激光焊接Z轴报警复位[A]
612.13 BOOL  ; RK_16 U6_Z 激光焊接Z轴使能[A]
612.14 BOOL  ; RK_12 预焊上料Z轴刹车使能[A]
612.15 BOOL  ; RK_12 预焊下料Z轴刹车使能[A]
613.00 BOOL  ; RK_16 激光焊接Z轴刹车使能[A]
613.01 BOOL  ; 0[A]
613.02 BOOL  ; 0[A]
613.03 BOOL  ; 0[A]
613.04 BOOL  ; 0[A]
613.05 BOOL  ; RK_12 OK出料拉带启动[A]
613.06 BOOL  ; 0[A]
613.07 BOOL  ; 0[A]
613.08 BOOL  ; 0[A]
613.09 BOOL  ; RK_07 #1铝壳上料电机刹车使能[A]
613.10 BOOL  ; RK_07 #2铝壳上料电机刹车使能[A]
613.11 BOOL  ; RK_07 #3托盘下料电机刹车使能[A]
613.12 BOOL  ; 三色灯_红（公共）[A]
613.13 BOOL  ; 三色灯_绿（公共）[A]
613.14 BOOL  ; 三色灯_黄（公共）[A]
613.15 BOOL  ; 蜂鸣器（公共）[A]
614.00 BOOL  ; RK_06 铝壳上料升降气缸下降[A]
614.01 BOOL  ; RK_06 铝壳上料升降气缸上升[A]
614.02 BOOL  ; RK_06 电池下料升降气缸下降[A]
614.03 BOOL  ; RK_06 电池下料升降气缸上升[A]
614.04 BOOL  ; RK_06 铝壳上料夹爪气缸夹紧[A]
614.05 BOOL  ; RK_06 铝壳上料夹爪气缸张开[A]
614.06 BOOL  ; RK_06 电池下料夹爪气缸夹紧[A]
614.07 BOOL  ; RK_06 电池下料夹爪气缸张开[A]
614.08 BOOL  ; RK_07 #1铝壳上料车定位升降气缸上升[A]
614.09 BOOL  ; RK_07 #1铝壳上料车定位升降气缸下降[A]
614.10 BOOL  ; RK_07 #2铝壳上料车定位升降气缸上升[A]
614.11 BOOL  ; RK_07 #2铝壳上料车定位升降气缸下降[A]
614.12 BOOL  ; RK_07 #3托盘下料车定位升降气缸上升[A]
614.13 BOOL  ; RK_07 #3托盘下料车定位升降气缸下降[A]
614.14 BOOL  ; RK_07 铝壳进料机械手升降气缸下降[A]
614.15 BOOL  ; RK_07 铝壳进料机械手升降气缸上升[A]
615.00 BOOL  ; RK_08 铝壳除尘旋转伸缩气缸缩回[A]
615.01 BOOL  ; RK_08 铝壳除尘旋转伸缩气缸伸出[A]
615.02 BOOL  ; RK_08 铝壳除尘伸缩气缸伸出[A]
615.03 BOOL  ; RK_08 铝壳除尘伸缩气缸缩回[A]
615.04 BOOL  ; RK_08 铝壳除尘夹爪气缸夹紧[A]
615.05 BOOL  ; RK_08 铝壳除尘夹爪气缸张开[A]
615.06 BOOL  ; RK_09 #1Hipot测试旋转伸缩气缸伸出[A]
615.07 BOOL  ; RK_09 #1Hipot测试旋转伸缩气缸缩回[A]
615.08 BOOL  ; RK_09 #1Hipot测试平台伸缩气缸缩回[A]
615.09 BOOL  ; RK_09 #1Hipot测试平台伸缩气缸伸出[A]
615.10 BOOL  ; RK_09 #1Hipot测试伸缩气缸伸出[A]
615.11 BOOL  ; RK_09 #1Hipot测试伸缩气缸缩回[A]
615.12 BOOL  ; RK_09 #2Hipot测试旋转伸缩气缸伸出[A]
615.13 BOOL  ; RK_09 #2Hipot测试旋转伸缩气缸缩回[A]
615.14 BOOL  ; RK_09 #2Hipot测试平台伸缩气缸缩回[A]
615.15 BOOL  ; RK_09 #2Hipot测试平台伸缩气缸伸出[A]
616.00 BOOL  ; RK_09 #2Hipot测试伸缩气缸伸出[A]
616.01 BOOL  ; RK_09 #2Hipot测试伸缩气缸缩回[A]
616.02 BOOL  ; RK_10 电池除尘上料机械手升降气缸下降[A]
616.03 BOOL  ; RK_10 电池除尘上料机械手升降气缸上升[A]
616.04 BOOL  ; RK_10 电池除尘上料机械手夹爪气缸夹紧[A]
616.05 BOOL  ; RK_10 电池除尘上料机械手夹爪气缸张开[A]
616.06 BOOL  ; RK_06 U8_X 电池上下料X轴报警复位[A]
616.07 BOOL  ; RK_06 U8_X 电池上下料X轴使能[A]
616.08 BOOL  ; RK_07 U8_Y 铝壳进料X轴报警复位[A]
616.09 BOOL  ; RK_07 U8_Y 铝壳进料X轴使能[A]
616.10 BOOL  ; RK_07 U8_Z 铝壳上料移载Y轴报警复位[A]
616.11 BOOL  ; RK_07 U8_Z 铝壳上料移载Y轴使能[A]
616.12 BOOL  ; RK_10 U8_U 电池除尘上料X轴报警复位[A]
616.13 BOOL  ; RK_10 U8_U 电池除尘上料X轴使能[A]
616.14 BOOL  ; RK_09 Hipot测试仪远程使能（取消）[A]
616.15 BOOL  ; RK_07 #1铝壳上料启动指示[A]
617.00 BOOL  ; RK_07 #2铝壳上料启动指示[A]
617.01 BOOL  ; RK_07 #3托盘下料启动指示[A]
617.02 BOOL  ; RK_07 铝壳上料移载吸盘立真空[A]
617.03 BOOL  ; RK_07 铝壳进料吸盘立真空[A]
617.04 BOOL  ; RK_07 #1铝壳上料电机正转[A]
617.05 BOOL  ; RK_07 #1铝壳上料电机反传[A]
617.06 BOOL  ; RK_10 Hipot检测NG拉带启动[A]
617.07 BOOL  ; RK_08 铝壳除尘吹气阀开[A]
617.08 BOOL  ; 0[A]
617.09 BOOL  ; RK_07 #2铝壳上料电机正传[A]
617.10 BOOL  ; RK_07 #2铝壳上料电机反传[A]
617.11 BOOL  ; 启动指示_绿（公共）[A]
617.12 BOOL  ; 停止指示_红（公共）[A]
617.13 BOOL  ; 复位指示_黄（公共）[A]
617.14 BOOL  ; RK_07 #3托盘下料电机正转[A]
617.15 BOOL  ; RK_07 #3托盘下料电机反传[A]
61.00 BOOL  ; RK_16 U6_Y 激光焊接X轴待机位
61.01 BOOL  ; RK_16 U6_Y 激光焊接X轴#1移载焊接位
61.02 BOOL  ; RK_16 U6_Y 激光焊接X轴#2移载焊接位
61.03 BOOL  ; 备用
61.04 BOOL  ; 备用
61.05 BOOL  ; 备用
61.06 BOOL  ; 备用
61.07 BOOL  ; 备用
61.08 BOOL  ; 备用
61.09 BOOL  ; 备用
621.04 BOOL  ; RK_11 电池除尘吹气阀关[A]
621.14 BOOL  ; RK_14 #1压装吸盘破真空[A]
621.15 BOOL  ; RK_14 #2压装吸盘破真空[A]
623.01 BOOL  ; RK_04 电芯除尘吹气阀关[A]
623.02 BOOL  ; RK_02 扫码NG拉带停止[A]
623.03 BOOL  ; RK_05 #1入壳吸盘破真空[A]
623.04 BOOL  ; RK_05 #2入壳吸盘破真空[A]
623.05 BOOL  ; RK_12 OK出料拉带停止[A]
627.02 BOOL  ; RK_07 铝壳上料移载吸盘破真空[A]
627.03 BOOL  ; RK_07 铝壳进料吸盘破真空[A]
627.04 BOOL  ; RK_07 #1铝壳上料电机停止[A]
627.06 BOOL  ; RK_10 Hipot检测NG拉带停止[A]
627.07 BOOL  ; RK_08 铝壳除尘吹气阀关[A]
627.09 BOOL  ; RK_07 #2铝壳上料电机停止[A]
627.14 BOOL  ; RK_07 #3托盘下料电机停止[A]
62.00 BOOL  ; RK_16 U6_Z 激光焊接Z轴待机位
62.01 BOOL  ; RK_16 U6_Z 激光焊接Z轴#1移载焊接位
62.02 BOOL  ; RK_16 U6_Z 激光焊接Z轴#2移载焊接位
62.03 BOOL  ; 备用
62.04 BOOL  ; 备用
62.05 BOOL  ; 备用
62.06 BOOL  ; 备用
62.07 BOOL  ; 备用
62.08 BOOL  ; 备用
62.09 BOOL  ; 备用
63.00 BOOL  ; RK_06 U8_X 电池上下料X轴待机位
63.01 BOOL  ; RK_06 U8_X 电池上下料X轴铝壳除尘取料位
63.02 BOOL  ; RK_06 U8_X 电池上下料X轴#1入壳放料位
63.03 BOOL  ; RK_06 U8_X 电池上下料X轴#2入壳放料位
63.04 BOOL  ; RK_06 U8_X 电池上下料X轴#1入壳取料位
63.05 BOOL  ; RK_06 U8_X 电池上下料X轴#2入壳取料位
63.06 BOOL  ; RK_06 U8_X 电池上下料X轴#1Hipot检测放料位
63.07 BOOL  ; RK_06 U8_X 电池上下料X轴#2Hipot检测放料位
63.08 BOOL  ; 备用
63.09 BOOL  ; 备用
64.00 BOOL  ; RK_07 U8_Y 铝壳进料X轴等待位
64.01 BOOL  ; RK_07 U8_Y 铝壳进料X轴取料位
64.02 BOOL  ; RK_07 U8_Y 铝壳进料X轴放料位
64.03 BOOL  ; 备用
64.04 BOOL  ; 备用
64.05 BOOL  ; 备用
64.06 BOOL  ; 备用
64.07 BOOL  ; 备用
64.08 BOOL  ; 备用
64.09 BOOL  ; 备用
650.00 BOOL  ; RK_01 U0_X 电芯来料Y轴待料位[A]
650.01 BOOL  ; RK_01 U0_X 电芯来料Y轴上料位[A]
650.02 BOOL  ; RK_01 U0_X 电芯来料Y轴扫码位[A]
650.03 BOOL  ; RK_01 U0_X 电芯来料Y轴下料位[A]
650.04 BOOL  ; 备用[A]
650.05 BOOL  ; 备用[A]
650.06 BOOL  ; 备用[A]
650.07 BOOL  ; 备用[A]
650.08 BOOL  ; 备用[A]
650.09 BOOL  ; 备用[A]
650.10 BOOL  ; RK_01 U0_X 电芯来料Y轴回原点[A]
650.11 BOOL  ; RK_01 U0_X 电芯来料Y轴JOG+[A]
650.12 BOOL  ; RK_01 U0_X 电芯来料Y轴JOG-[A]
650.13 BOOL  ; RK_01 U0_X 电芯来料Y轴JOG高速[A]
650.14 BOOL  ; RK_01 U0_X 电芯来料Y轴JOG低速[A]
650.15 BOOL  ; 备用[A]
651.00 BOOL  ; RK_02 U0_Y 电芯进料X轴待料位[A]
651.01 BOOL  ; RK_02 U0_Y 电芯进料X轴取料位[A]
651.02 BOOL  ; RK_02 U0_Y 电芯进料X轴扫码OK放料位[A]
651.03 BOOL  ; RK_02 U0_Y 电芯进料X轴扫码NG放料位[A]
651.04 BOOL  ; 备用[A]
651.05 BOOL  ; 备用[A]
651.06 BOOL  ; 备用[A]
651.07 BOOL  ; 备用[A]
651.08 BOOL  ; 备用[A]
651.09 BOOL  ; 备用[A]
651.10 BOOL  ; RK_02 U0_Y 电芯进料X轴回原点[A]
651.11 BOOL  ; RK_02 U0_Y 电芯进料X轴JOG+[A]
651.12 BOOL  ; RK_02 U0_Y 电芯进料X轴JOG-[A]
651.13 BOOL  ; RK_02 U0_Y 电芯进料X轴JOG高速[A]
651.14 BOOL  ; RK_02 U0_Y 电芯进料X轴JOG低速[A]
651.15 BOOL  ; 备用[A]
652.00 BOOL  ; RK_02 U0_Z 电芯进料Z轴待料位（扫码）[A]
652.01 BOOL  ; RK_02 U0_Z 电芯进料Z轴取料位[A]
652.02 BOOL  ; RK_02 U0_Z 电芯进料Z轴扫码OK放料位[A]
652.03 BOOL  ; RK_02 U0_Z 电芯进料Z轴扫码NG放料位[A]
652.04 BOOL  ; RK_02 U0_Z 电芯进料Z轴扫码位[A]
652.05 BOOL  ; 备用[A]
652.06 BOOL  ; 备用[A]
652.07 BOOL  ; 备用[A]
652.08 BOOL  ; 备用[A]
652.09 BOOL  ; 备用[A]
652.10 BOOL  ; RK_02 U0_Z 电芯进料Z轴回原点[A]
652.11 BOOL  ; RK_02 U0_Z 电芯进料Z轴JOG+[A]
652.12 BOOL  ; RK_02 U0_Z 电芯进料Z轴JOG-[A]
652.13 BOOL  ; RK_02 U0_Z 电芯进料Z轴JOG高速[A]
652.14 BOOL  ; RK_02 U0_Z 电芯进料Z轴JOG低速[A]
652.15 BOOL  ; 备用[A]
653.00 BOOL  ; RK_03 U0_U 电芯上料X轴待料位[A]
653.01 BOOL  ; RK_03 U0_U 电芯上料X轴取料位[A]
653.02 BOOL  ; RK_03 U0_U 电芯上料X轴#1入壳放料位[A]
653.03 BOOL  ; RK_03 U0_U 电芯上料X轴#2入壳放料位[A]
653.04 BOOL  ; 备用[A]
653.05 BOOL  ; 备用[A]
653.06 BOOL  ; 备用[A]
653.07 BOOL  ; 备用[A]
653.08 BOOL  ; 备用[A]
653.09 BOOL  ; 备用[A]
653.10 BOOL  ; RK_03 U0_U 电芯上料X轴回原点[A]
653.11 BOOL  ; RK_03 U0_U 电芯上料X轴JOG+[A]
653.12 BOOL  ; RK_03 U0_U 电芯上料X轴JOG-[A]
653.13 BOOL  ; RK_03 U0_U 电芯上料X轴JOG高速[A]
653.14 BOOL  ; RK_03 U0_U 电芯上料X轴JOG低速[A]
653.15 BOOL  ; 备用[A]
654.00 BOOL  ; RK_05 U2_X #1入壳Y轴待料位[A]
654.01 BOOL  ; RK_05 U2_X #1入壳Y轴滚轮压紧位[A]
654.02 BOOL  ; RK_05 U2_X #1入壳Y轴滚轮松开位[A]
654.03 BOOL  ; RK_05 U2_X #1入壳Y轴入壳位[A]
654.04 BOOL  ; RK_05 U2_X #1入壳Y轴电芯定位夹爪松开位[A]
654.05 BOOL  ; 备用[A]
654.06 BOOL  ; 备用[A]
654.07 BOOL  ; 备用[A]
654.08 BOOL  ; 备用[A]
654.09 BOOL  ; 备用[A]
654.10 BOOL  ; RK_05 U2_X #1入壳Y轴回原点[A]
654.11 BOOL  ; RK_05 U2_X #1入壳Y轴JOG+[A]
654.12 BOOL  ; RK_05 U2_X #1入壳Y轴JOG-[A]
654.13 BOOL  ; RK_05 U2_X #1入壳Y轴JOG高速[A]
654.14 BOOL  ; RK_05 U2_X #1入壳Y轴JOG低速[A]
654.15 BOOL  ; 备用[A]
655.00 BOOL  ; RK_05 U2_Y #2入壳Y轴待料位[A]
655.01 BOOL  ; RK_05 U2_Y #2入壳Y轴滚轮压紧位[A]
655.02 BOOL  ; RK_05 U2_Y #2入壳Y轴滚轮松开位[A]
655.03 BOOL  ; RK_05 U2_Y #2入壳Y轴入壳位[A]
655.04 BOOL  ; RK_05 U2_Y #2入壳Y轴电芯定位夹爪松开位[A]
655.05 BOOL  ; 备用[A]
655.06 BOOL  ; 备用[A]
655.07 BOOL  ; 备用[A]
655.08 BOOL  ; 备用[A]
655.09 BOOL  ; 备用[A]
655.10 BOOL  ; RK_05 U2_Y #2入壳Y轴回原点[A]
655.11 BOOL  ; RK_05 U2_Y #2入壳Y轴JOG+[A]
655.12 BOOL  ; RK_05 U2_Y #2入壳Y轴JOG-[A]
655.13 BOOL  ; RK_05 U2_Y #2入壳Y轴JOG高速[A]
655.14 BOOL  ; RK_05 U2_Y #2入壳Y轴JOG低速[A]
655.15 BOOL  ; 备用[A]
656.00 BOOL  ; RK_12 U4_X 预焊上下料X轴待料位[A]
656.01 BOOL  ; RK_12 U4_X 预焊上下料X轴除尘取料位[A]
656.02 BOOL  ; RK_12 U4_X 预焊上下料X轴#1移载放料位[A]
656.03 BOOL  ; RK_12 U4_X 预焊上下料X轴#2移载放料位[A]
656.04 BOOL  ; RK_12 U4_X 预焊上下料X轴#1移载取料位[A]
656.05 BOOL  ; RK_12 U4_X 预焊上下料X轴#2移载取料位[A]
656.06 BOOL  ; RK_12 U4_X 预焊上下料X轴OK放料位[A]
656.07 BOOL  ; RK_12 U4_X 预焊上下料X轴#1NG放料位[A]
656.08 BOOL  ; RK_12 U4_X 预焊上下料X轴#2NG放料位[A]
656.09 BOOL  ; 备用[A]
656.10 BOOL  ; RK_12 U4_X 预焊上下料X轴回原点[A]
656.11 BOOL  ; RK_12 U4_X 预焊上下料X轴JOG+[A]
656.12 BOOL  ; RK_12 U4_X 预焊上下料X轴JOG-[A]
656.13 BOOL  ; RK_12 U4_X 预焊上下料X轴JOG高速[A]
656.14 BOOL  ; RK_12 U4_X 预焊上下料X轴JOG低速[A]
656.15 BOOL  ; 备用[A]
657.00 BOOL  ; RK_12 U4_Y 预焊上料Z轴待料位[A]
657.01 BOOL  ; RK_12 U4_Y 预焊上料Z轴除尘取料位[A]
657.02 BOOL  ; RK_12 U4_Y 预焊上料Z轴#1移载放料位[A]
657.03 BOOL  ; RK_12 U4_Y 预焊上料Z轴#2移载放料位[A]
657.04 BOOL  ; 备用[A]
657.05 BOOL  ; 备用[A]
657.06 BOOL  ; 备用[A]
657.07 BOOL  ; 备用[A]
657.08 BOOL  ; 备用[A]
657.09 BOOL  ; 备用[A]
657.10 BOOL  ; RK_12 U4_Y 预焊上料Z轴回原点[A]
657.11 BOOL  ; RK_12 U4_Y 预焊上料Z轴JOG+[A]
657.12 BOOL  ; RK_12 U4_Y 预焊上料Z轴JOG-[A]
657.13 BOOL  ; RK_12 U4_Y 预焊上料Z轴JOG高速[A]
657.14 BOOL  ; RK_12 U4_Y 预焊上料Z轴JOG低速[A]
657.15 BOOL  ; 备用[A]
658.00 BOOL  ; RK_12 U4_Z 预焊下料Z轴待料位[A]
658.01 BOOL  ; RK_12 U4_Z 预焊下料Z轴#1移载取料位[A]
658.02 BOOL  ; RK_12 U4_Z 预焊下料Z轴#2移载取料位[A]
658.03 BOOL  ; RK_12 U4_Z 预焊下料Z轴OK放料位[A]
658.04 BOOL  ; RK_12 U4_Z 预焊下料Z轴#1NG放料位[A]
658.05 BOOL  ; RK_12 U4_Z 预焊下料Z轴#2NG放料位[A]
658.06 BOOL  ; 备用[A]
658.07 BOOL  ; 备用[A]
658.08 BOOL  ; 备用[A]
658.09 BOOL  ; 备用[A]
658.10 BOOL  ; RK_12 U4_Z 预焊下料Z轴回原点[A]
658.11 BOOL  ; RK_12 U4_Z 预焊下料Z轴JOG+[A]
658.12 BOOL  ; RK_12 U4_Z 预焊下料Z轴JOG-[A]
658.13 BOOL  ; RK_12 U4_Z 预焊下料Z轴JOG高速[A]
658.14 BOOL  ; RK_12 U4_Z 预焊下料Z轴JOG低速[A]
658.15 BOOL  ; 备用[A]
659.00 BOOL  ; RK_13 U4_U #1移载Y轴待料位[A]
659.01 BOOL  ; RK_13 U4_U #1移载Y轴取放料位[A]
659.02 BOOL  ; RK_13 U4_U #1移载Y轴压装位[A]
659.03 BOOL  ; RK_13 U4_U #1移载Y轴#1轮廓检测位[A]
659.04 BOOL  ; RK_13 U4_U #1移载Y轴#2轮廓检测位[A]
659.05 BOOL  ; RK_13 U4_U #1移载Y轴激光焊接位[A]
659.06 BOOL  ; 备用[A]
659.07 BOOL  ; 备用[A]
659.08 BOOL  ; 备用[A]
659.09 BOOL  ; 备用[A]
659.10 BOOL  ; RK_13 U4_U #1移载Y轴回原点[A]
659.11 BOOL  ; RK_13 U4_U #1移载Y轴JOG+[A]
659.12 BOOL  ; RK_13 U4_U #1移载Y轴JOG-[A]
659.13 BOOL  ; RK_13 U4_U #1移载Y轴JOG高速[A]
659.14 BOOL  ; RK_13 U4_U #1移载Y轴JOG低速[A]
659.15 BOOL  ; 备用[A]
65.00 BOOL  ; RK_07 U8_Z 铝壳上料移载Y轴待料位
65.01 BOOL  ; RK_07 U8_Z 铝壳上料移载Y轴#1铝壳上料位
65.02 BOOL  ; RK_07 U8_Z 铝壳上料移载Y轴#2铝壳上料位
65.03 BOOL  ; RK_07 U8_Z 铝壳上料移载Y轴#3铝壳托盘下料位
65.04 BOOL  ; RK_07 U8_Z 铝壳上料移载Y轴铝壳取料位
65.05 BOOL  ; 备用
65.06 BOOL  ; 备用
65.07 BOOL  ; 备用
65.08 BOOL  ; 备用
65.09 BOOL  ; 备用
660.00 BOOL  ; RK_13 U6_X #2移载Y轴待料位[A]
660.01 BOOL  ; RK_13 U6_X #2移载Y轴取放料位[A]
660.02 BOOL  ; RK_13 U6_X #2移载Y轴压装位[A]
660.03 BOOL  ; RK_13 U6_X #2移载Y轴#1轮廓检测位[A]
660.04 BOOL  ; RK_13 U6_X #2移载Y轴#2轮廓检测位[A]
660.05 BOOL  ; RK_13 U6_X #2移载Y轴激光焊接位[A]
660.06 BOOL  ; 备用[A]
660.07 BOOL  ; 备用[A]
660.08 BOOL  ; 备用[A]
660.09 BOOL  ; 备用[A]
660.10 BOOL  ; RK_13 U6_X #2移载Y轴回原点[A]
660.11 BOOL  ; RK_13 U6_X #2移载Y轴JOG+[A]
660.12 BOOL  ; RK_13 U6_X #2移载Y轴JOG-[A]
660.13 BOOL  ; RK_13 U6_X #2移载Y轴JOG高速[A]
660.14 BOOL  ; RK_13 U6_X #2移载Y轴JOG低速[A]
660.15 BOOL  ; 备用[A]
661.00 BOOL  ; RK_16 U6_Y 激光焊接X轴待机位[A]
661.01 BOOL  ; RK_16 U6_Y 激光焊接X轴#1移载焊接位[A]
661.02 BOOL  ; RK_16 U6_Y 激光焊接X轴#2移载焊接位[A]
661.03 BOOL  ; 备用[A]
661.04 BOOL  ; 备用[A]
661.05 BOOL  ; 备用[A]
661.06 BOOL  ; 备用[A]
661.07 BOOL  ; 备用[A]
661.08 BOOL  ; 备用[A]
661.09 BOOL  ; 备用[A]
661.10 BOOL  ; RK_16 U6_Y 激光焊接X轴回原点[A]
661.11 BOOL  ; RK_16 U6_Y 激光焊接X轴JOG+[A]
661.12 BOOL  ; RK_16 U6_Y 激光焊接X轴JOG-[A]
661.13 BOOL  ; RK_16 U6_Y 激光焊接X轴JOG高速[A]
661.14 BOOL  ; RK_16 U6_Y 激光焊接X轴JOG低速[A]
661.15 BOOL  ; 备用[A]
662.00 BOOL  ; RK_16 U6_Z 激光焊接Z轴待机位[A]
662.01 BOOL  ; RK_16 U6_Z 激光焊接Z轴#1移载焊接位[A]
662.02 BOOL  ; RK_16 U6_Z 激光焊接Z轴#2移载焊接位[A]
662.03 BOOL  ; 备用[A]
662.04 BOOL  ; 备用[A]
662.05 BOOL  ; 备用[A]
662.06 BOOL  ; 备用[A]
662.07 BOOL  ; 备用[A]
662.08 BOOL  ; 备用[A]
662.09 BOOL  ; 备用[A]
662.10 BOOL  ; RK_16 U6_Z 激光焊接Z轴回原点[A]
662.11 BOOL  ; RK_16 U6_Z 激光焊接Z轴JOG+[A]
662.12 BOOL  ; RK_16 U6_Z 激光焊接Z轴JOG-[A]
662.13 BOOL  ; RK_16 U6_Z 激光焊接Z轴JOG高速[A]
662.14 BOOL  ; RK_16 U6_Z 激光焊接Z轴JOG低速[A]
662.15 BOOL  ; 备用[A]
663.00 BOOL  ; RK_06 U8_X 电池上下料X轴待机位[A]
663.01 BOOL  ; RK_06 U8_X 电池上下料X轴铝壳除尘取料位[A]
663.02 BOOL  ; RK_06 U8_X 电池上下料X轴#1入壳放料位[A]
663.03 BOOL  ; RK_06 U8_X 电池上下料X轴#2入壳放料位[A]
663.04 BOOL  ; RK_06 U8_X 电池上下料X轴#1入壳取料位[A]
663.05 BOOL  ; RK_06 U8_X 电池上下料X轴#2入壳取料位[A]
663.06 BOOL  ; RK_06 U8_X 电池上下料X轴#1Hipot检测放料位[A]
663.07 BOOL  ; RK_06 U8_X 电池上下料X轴#2Hipot检测放料位[A]
663.08 BOOL  ; 备用[A]
663.09 BOOL  ; 备用[A]
663.10 BOOL  ; RK_06 U8_X 电池上下料X轴回原点[A]
663.11 BOOL  ; RK_06 U8_X 电池上下料X轴JOG+[A]
663.12 BOOL  ; RK_06 U8_X 电池上下料X轴JOG-[A]
663.13 BOOL  ; RK_06 U8_X 电池上下料X轴JOG高速[A]
663.14 BOOL  ; RK_06 U8_X 电池上下料X轴JOG低速[A]
663.15 BOOL  ; 备用[A]
664.00 BOOL  ; RK_07 U8_Y 铝壳进料X轴等待位[A]
664.01 BOOL  ; RK_07 U8_Y 铝壳进料X轴取料位[A]
664.02 BOOL  ; RK_07 U8_Y 铝壳进料X轴放料位[A]
664.03 BOOL  ; 备用[A]
664.04 BOOL  ; 备用[A]
664.05 BOOL  ; 备用[A]
664.06 BOOL  ; 备用[A]
664.07 BOOL  ; 备用[A]
664.08 BOOL  ; 备用[A]
664.09 BOOL  ; 备用[A]
664.10 BOOL  ; RK_07 U8_Y 铝壳进料X轴回原点[A]
664.11 BOOL  ; RK_07 U8_Y 铝壳进料X轴JOG+[A]
664.12 BOOL  ; RK_07 U8_Y 铝壳进料X轴JOG-[A]
664.13 BOOL  ; RK_07 U8_Y 铝壳进料X轴JOG高速[A]
664.14 BOOL  ; RK_07 U8_Y 铝壳进料X轴JOG低速[A]
664.15 BOOL  ; 备用[A]
665.00 BOOL  ; RK_07 U8_Z 铝壳上料移载Y轴待料位[A]
665.01 BOOL  ; RK_07 U8_Z 铝壳上料移载Y轴#1铝壳上料位[A]
665.02 BOOL  ; RK_07 U8_Z 铝壳上料移载Y轴#2铝壳上料位[A]
665.03 BOOL  ; RK_07 U8_Z 铝壳上料移载Y轴#3铝壳托盘下料位[A]
665.04 BOOL  ; RK_07 U8_Z 铝壳上料移载Y轴铝壳取料位[A]
665.05 BOOL  ; 备用[A]
665.06 BOOL  ; 备用[A]
665.07 BOOL  ; 备用[A]
665.08 BOOL  ; 备用[A]
665.09 BOOL  ; 备用[A]
665.10 BOOL  ; RK_07 U8_Z 铝壳上料移载Y轴回原点[A]
665.11 BOOL  ; RK_07 U8_Z 铝壳上料移载Y轴JOG+[A]
665.12 BOOL  ; RK_07 U8_Z 铝壳上料移载Y轴JOG-[A]
665.13 BOOL  ; RK_07 U8_Z 铝壳上料移载Y轴JOG高速[A]
665.14 BOOL  ; RK_07 U8_Z 铝壳上料移载Y轴JOG低速[A]
665.15 BOOL  ; 备用[A]
666.00 BOOL  ; RK_10 U8_U 电池除尘上料X轴待料位[A]
666.01 BOOL  ; RK_10 U8_U 电池除尘上料X轴#1Hipot检测取料位[A]
666.02 BOOL  ; RK_10 U8_U 电池除尘上料X轴#2Hipot检测取料位[A]
666.03 BOOL  ; RK_10 U8_U 电池除尘上料X轴Hipot OK放料位[A]
666.04 BOOL  ; RK_10 U8_U 电池除尘上料X轴Hipot NG放料位[A]
666.05 BOOL  ; 备用[A]
666.06 BOOL  ; 备用[A]
666.07 BOOL  ; 备用[A]
666.08 BOOL  ; 备用[A]
666.09 BOOL  ; 备用[A]
666.10 BOOL  ; RK_10 U8_U 电池除尘上料X轴回原点[A]
666.11 BOOL  ; RK_10 U8_U 电池除尘上料X轴JOG+[A]
666.12 BOOL  ; RK_10 U8_U 电池除尘上料X轴JOG-[A]
666.13 BOOL  ; RK_10 U8_U 电池除尘上料X轴JOG高速[A]
666.14 BOOL  ; RK_10 U8_U 电池除尘上料X轴JOG低速[A]
666.15 BOOL  ; 备用[A]
66.00 BOOL  ; RK_10 U8_U 电池除尘上料X轴待料位
66.01 BOOL  ; RK_10 U8_U 电池除尘上料X轴#1Hipot检测取料位
66.02 BOOL  ; RK_10 U8_U 电池除尘上料X轴#2Hipot检测取料位
66.03 BOOL  ; RK_10 U8_U 电池除尘上料X轴Hipot OK放料位
66.04 BOOL  ; RK_10 U8_U 电池除尘上料X轴Hipot NG放料位
66.05 BOOL  ; 备用
66.06 BOOL  ; 备用
66.07 BOOL  ; 备用
66.08 BOOL  ; 备用
66.09 BOOL  ; 备用
6.00 BOOL  ; 小屏插入信号（公共）
6.01 BOOL  ; NC433模块DC5V电源信号（公共）
6.02 BOOL  ; DC24V伺服刹车电源信号（公共）
6.03 BOOL  ; 出料端急停（公共）
6.04 BOOL  ; 小移动屏急停（公共）
6.05 BOOL  ; A机架#1门磁（公共）
6.06 BOOL  ; A机架#2门磁（公共）
6.07 BOOL  ; A机架#3门磁（公共）
6.08 BOOL  ; A机架#4门磁（公共）
6.09 BOOL  ; A机架#5门磁（公共）
6.10 BOOL  ; A机架#6门磁（公共）
6.11 BOOL  ; A机架#7门磁（公共）
6.12 BOOL  ; A机架#8门磁（公共）
6.13 BOOL  ; A机架#9门磁（公共）
6.14 BOOL  ; RK_01 电芯来料上料位有料感应
700.00 BOOL  ; RK_02 电芯进料机械手夹爪气缸夹紧[SW]
700.01 BOOL  ; RK_02 电芯进料机械手夹爪气缸张开[SW]
700.02 BOOL  ; RK_02 电芯进料机械手压紧气缸伸出[SW]
700.03 BOOL  ; RK_02 电芯进料机械手压紧气缸缩回[SW]
700.04 BOOL  ; RK_03 电芯上料机械手夹爪气缸夹紧[SW]
700.05 BOOL  ; RK_03 电芯上料机械手夹爪气缸张开[SW]
700.06 BOOL  ; RK_03 电芯上料机械手压紧气缸伸出[SW]
700.07 BOOL  ; RK_03 电芯上料机械手压紧气缸缩回[SW]
700.08 BOOL  ; RK_03 电芯上料升降气缸下降[SW]
700.09 BOOL  ; RK_03 电芯上料升降气缸上升[SW]
700.10 BOOL  ; RK_04 电芯除尘伸缩气缸缩回[SW]
700.11 BOOL  ; RK_04 电芯除尘伸缩气缸伸出[SW]
700.12 BOOL  ; RK_05 #1入壳滚轮夹紧气缸伸出[SW]
700.13 BOOL  ; RK_05 #1入壳滚轮夹紧气缸缩回[SW]
700.14 BOOL  ; RK_05 #1入壳铝壳定位平台伸缩气缸缩回[SW]
700.15 BOOL  ; RK_05 #1入壳铝壳定位平台伸缩气缸伸出[SW]
701.00 BOOL  ; RK_05 #1入壳铝壳定位平台升降气缸上升[SW]
701.01 BOOL  ; RK_05 #1入壳铝壳定位平台升降气缸下降[SW]
701.02 BOOL  ; RK_05 #1入壳铝壳定位伸缩气缸缩回[SW]
701.03 BOOL  ; RK_05 #1入壳铝壳定位伸缩气缸伸出[SW]
701.04 BOOL  ; RK_05 #1入壳铝壳定位夹爪气缸夹紧[SW]
701.05 BOOL  ; RK_05 #1入壳铝壳定位夹爪气缸张开[SW]
701.06 BOOL  ; RK_05 #2入壳滚轮夹紧气缸伸出[SW]
701.07 BOOL  ; RK_05 #2入壳滚轮夹紧气缸缩回[SW]
701.08 BOOL  ; RK_05 #2入壳铝壳定位平台伸缩气缸缩回[SW]
701.09 BOOL  ; RK_05 #2入壳铝壳定位平台伸缩气缸伸出[SW]
701.10 BOOL  ; RK_05 #2入壳铝壳定位平台升降气缸上升[SW]
701.11 BOOL  ; RK_05 #2入壳铝壳定位平台升降气缸下降[SW]
701.12 BOOL  ; RK_05 #2入壳铝壳定位伸缩气缸缩回[SW]
701.13 BOOL  ; RK_05 #2入壳铝壳定位伸缩气缸伸出[SW]
701.14 BOOL  ; RK_05 #2入壳铝壳定位夹爪气缸夹紧[SW]
701.15 BOOL  ; RK_05 #2入壳铝壳定位夹爪气缸张开[SW]
702.00 BOOL  ; RK_01 U0_X 电芯来料Y轴报警复位[SW]
702.01 BOOL  ; RK_01 U0_X 电芯来料Y轴使能[SW]
702.02 BOOL  ; RK_02 U0_Y 电芯进料X轴报警复位[SW]
702.03 BOOL  ; RK_02 U0_Y 电芯进料X轴使能[SW]
702.04 BOOL  ; RK_02 U0_Z 电芯进料Z轴报警复位[SW]
702.05 BOOL  ; RK_02 U0_Z 电芯进料Z轴使能[SW]
702.06 BOOL  ; RK_03 U0_U 电芯上料X轴报警复位[SW]
702.07 BOOL  ; RK_03 U0_U 电芯上料X轴使能[SW]
702.08 BOOL  ; RK_05 U2_X #1入壳Y轴报警复位[SW]
702.09 BOOL  ; RK_05 U2_X #1入壳Y轴使能[SW]
702.10 BOOL  ; RK_05 U2_Y #2入壳Y轴报警复位[SW]
702.11 BOOL  ; RK_05 U2_Y #2入壳Y轴使能[SW]
702.12 BOOL  ; RK_02 电芯进料Z轴刹车使能[SW]
702.13 BOOL  ; RK_05 #1入壳定位陶瓷棒夹紧气缸伸出[SW]
702.14 BOOL  ; RK_05 #1入壳定位陶瓷棒夹紧气缸缩回[SW]
702.15 BOOL  ; RK_05 #2入壳定位陶瓷棒夹紧气缸伸出[SW]
703.00 BOOL  ; RK_05 #2入壳定位陶瓷棒夹紧气缸缩回[SW]
703.01 BOOL  ; RK_04 电芯除尘吹气阀开[SW]
703.02 BOOL  ; RK_02 扫码NG拉带启动[SW]
703.03 BOOL  ; RK_05 #1入壳吸盘立真空[SW]
703.04 BOOL  ; RK_05 #2入壳吸盘立真空[SW]
703.05 BOOL  ; RK_05 #1入壳吸盘伸缩气缸伸出[SW]
703.06 BOOL  ; RK_05 #1入壳吸盘伸缩气缸缩回[SW]
703.07 BOOL  ; RK_05 #2入壳吸盘伸缩气缸伸出[SW]
703.08 BOOL  ; RK_05 #2入壳吸盘伸缩气缸缩回[SW]
703.09 BOOL  ; 前端设备对接输出信号（公共）[SW]
703.10 BOOL  ; 后端设备对接输出信号（公共）[SW]
703.11 BOOL  ; RK_05 #1入壳电芯定位夹爪气缸伸出[SW]
703.12 BOOL  ; RK_05 #1入壳电芯定位夹爪气缸缩回[SW]
703.13 BOOL  ; RK_05 #2入壳电芯定位夹爪气缸伸出[SW]
703.14 BOOL  ; RK_05 #2入壳电芯定位夹爪气缸缩回[SW]
708.00 BOOL  ; RK_11 电池除尘旋转伸缩气缸缩回[SW]
708.01 BOOL  ; RK_11 电池除尘旋转伸缩气缸伸出[SW]
708.02 BOOL  ; RK_11 电池除尘伸缩气缸伸出[SW]
708.03 BOOL  ; RK_11 电池除尘伸缩气缸缩回[SW]
708.04 BOOL  ; RK_11 电池除尘夹爪气缸夹紧[SW]
708.05 BOOL  ; RK_11 电池除尘夹爪气缸张开[SW]
708.06 BOOL  ; RK_12 预焊上料机械手夹爪气缸夹紧[SW]
708.07 BOOL  ; RK_12 预焊上料机械手夹爪气缸张开[SW]
708.08 BOOL  ; RK_12 预焊下料机械手夹爪气缸夹紧[SW]
708.09 BOOL  ; RK_12 预焊下料机械手夹爪气缸张开[SW]
708.10 BOOL  ; RK_13 #1移载升降气缸上升[SW]
708.11 BOOL  ; RK_13 #1移载升降气缸下降[SW]
708.12 BOOL  ; RK_13 #1移载定位#1伸缩气缸缩回[SW]
708.13 BOOL  ; RK_13 #1移载定位#1伸缩气缸伸出[SW]
708.14 BOOL  ; RK_13 #1移载定位#2伸缩气缸缩回[SW]
708.15 BOOL  ; RK_13 #1移载定位#2伸缩气缸伸出[SW]
709.00 BOOL  ; RK_13 #1移载导向#1伸缩气缸伸出[SW]
709.01 BOOL  ; RK_13 #1移载导向#1伸缩气缸缩回[SW]
709.02 BOOL  ; RK_13 #1移载导向#2伸缩气缸伸出[SW]
709.03 BOOL  ; RK_13 #1移载导向#2伸缩气缸缩回[SW]
709.04 BOOL  ; RK_13 #1移载左右定位伸缩气缸伸出[SW]
709.05 BOOL  ; RK_13 #1移载左右定位伸缩气缸缩回[SW]
709.06 BOOL  ; RK_13 #2移载升降气缸上升[SW]
709.07 BOOL  ; RK_13 #2移载升降气缸下降[SW]
709.08 BOOL  ; RK_13 #2移载定位#1伸缩气缸缩回[SW]
709.09 BOOL  ; RK_13 #2移载定位#1伸缩气缸伸出[SW]
709.10 BOOL  ; RK_13 #2移载定位#2伸缩气缸缩回[SW]
709.11 BOOL  ; RK_13 #2移载定位#2伸缩气缸伸出[SW]
709.12 BOOL  ; RK_13 #2移载导向#1伸缩气缸伸出[SW]
709.13 BOOL  ; RK_13 #2移载导向#1伸缩气缸缩回[SW]
709.14 BOOL  ; RK_13 #2移载导向#2伸缩气缸伸出[SW]
709.15 BOOL  ; RK_13 #2移载导向#2伸缩气缸缩回[SW]
710.00 BOOL  ; RK_13 #2移载左右定位伸缩气缸伸出[SW]
710.01 BOOL  ; RK_13 #2移载左右定位伸缩气缸缩回[SW]
710.02 BOOL  ; RK_14 #1压装升降气缸下降[SW]
710.03 BOOL  ; RK_14 #1压装升降气缸上升[SW]
710.04 BOOL  ; RK_14 #1压装#1吸盘升降气缸下降[SW]
710.05 BOOL  ; RK_14 #1压装#1吸盘升降气缸上升[SW]
710.06 BOOL  ; RK_14 #1压装#2吸盘升降气缸下降[SW]
710.07 BOOL  ; RK_14 #1压装#2吸盘升降气缸上升[SW]
710.08 BOOL  ; RK_14 #2压装升降气缸下降[SW]
710.09 BOOL  ; RK_14 #2压装升降气缸上升[SW]
710.10 BOOL  ; RK_14 #2压装#1吸盘升降气缸下降[SW]
710.11 BOOL  ; RK_14 #2压装#1吸盘升降气缸上升[SW]
710.12 BOOL  ; RK_14 #2压装#2吸盘升降气缸下降[SW]
710.13 BOOL  ; RK_14 #2压装#2吸盘升降气缸上升[SW]
710.14 BOOL  ; RK_15 轮廓检测#1伸缩气缸伸出[SW]
710.15 BOOL  ; RK_15 轮廓检测#1伸缩气缸缩回[SW]
711.00 BOOL  ; RK_15 轮廓检测#2伸缩气缸伸出[SW]
711.01 BOOL  ; RK_15 轮廓检测#2伸缩气缸缩回[SW]
711.02 BOOL  ; RK_12 轮廓检测NG拨料气缸伸出[SW]
711.03 BOOL  ; RK_12 轮廓检测NG拨料气缸缩回[SW]
711.04 BOOL  ; RK_11 电池除尘吹气阀开[SW]
711.05 BOOL  ; 0[SW]
711.06 BOOL  ; 0[SW]
711.07 BOOL  ; RK_16 激光焊接触发[SW]
711.08 BOOL  ; RK_16 PLC急停输出到激光设备[SW]
711.09 BOOL  ; RK_16 #1移载激光焊任务选择[SW]
711.10 BOOL  ; RK_16 #2移载激光焊任务选择[SW]
711.11 BOOL  ; RK_16 集尘器启动[SW]
711.12 BOOL  ; 0[SW]
711.13 BOOL  ; 0[SW]
711.14 BOOL  ; RK_14 #1压装吸盘立真空[SW]
711.15 BOOL  ; RK_14 #2压装吸盘立真空[SW]
712.00 BOOL  ; RK_12 U4_X 预焊上下料X轴报警复位[SW]
712.01 BOOL  ; RK_12 U4_X 预焊上下料X轴使能[SW]
712.02 BOOL  ; RK_12 U4_Y 预焊上料Z轴报警复位[SW]
712.03 BOOL  ; RK_12 U4_Y 预焊上料Z轴使能[SW]
712.04 BOOL  ; RK_12 U4_Z 预焊下料Z轴报警复位[SW]
712.05 BOOL  ; RK_12 U4_Z 预焊下料Z轴使能[SW]
712.06 BOOL  ; RK_13 U4_U #1移载Y轴报警复位[SW]
712.07 BOOL  ; RK_13 U4_U #1移载Y轴使能[SW]
712.08 BOOL  ; RK_13 U6_X #2移载Y轴报警复位[SW]
712.09 BOOL  ; RK_13 U6_X #2移载Y轴使能[SW]
712.10 BOOL  ; RK_16 U6_Y 激光焊接X轴报警复位[SW]
712.11 BOOL  ; RK_16 U6_Y 激光焊接X轴使能[SW]
712.12 BOOL  ; RK_16 U6_Z 激光焊接Z轴报警复位[SW]
712.13 BOOL  ; RK_16 U6_Z 激光焊接Z轴使能[SW]
712.14 BOOL  ; RK_12 预焊上料Z轴刹车使能[SW]
712.15 BOOL  ; RK_12 预焊下料Z轴刹车使能[SW]
713.00 BOOL  ; RK_16 激光焊接Z轴刹车使能[SW]
713.01 BOOL  ; 0[SW]
713.02 BOOL  ; 0[SW]
713.03 BOOL  ; 0[SW]
713.04 BOOL  ; 0[SW]
713.05 BOOL  ; RK_07 OK出料拉带启动[SW]
713.06 BOOL  ; 0[SW]
713.07 BOOL  ; 0[SW]
713.08 BOOL  ; 0[SW]
713.09 BOOL  ; RK_07 #1铝壳上料电机刹车使能[SW]
713.10 BOOL  ; RK_07 #2铝壳上料电机刹车使能[SW]
713.11 BOOL  ; RK_07 #3托盘下料电机刹车使能[SW]
713.12 BOOL  ; 三色灯_红（公共）[SW]
713.13 BOOL  ; 三色灯_绿（公共）[SW]
713.14 BOOL  ; 三色灯_黄（公共）[SW]
713.15 BOOL  ; 蜂鸣器（公共）[SW]
714.00 BOOL  ; RK_06 铝壳上料升降气缸下降[SW]
714.01 BOOL  ; RK_06 铝壳上料升降气缸上升[SW]
714.02 BOOL  ; RK_06 电池下料升降气缸下降[SW]
714.03 BOOL  ; RK_06 电池下料升降气缸上升[SW]
714.04 BOOL  ; RK_06 铝壳上料夹爪气缸夹紧[SW]
714.05 BOOL  ; RK_06 铝壳上料夹爪气缸张开[SW]
714.06 BOOL  ; RK_06 电池下料夹爪气缸夹紧[SW]
714.07 BOOL  ; RK_06 电池下料夹爪气缸张开[SW]
714.08 BOOL  ; RK_07 #1铝壳上料车定位升降气缸上升[SW]
714.09 BOOL  ; RK_07 #1铝壳上料车定位升降气缸下降[SW]
714.10 BOOL  ; RK_07 #2铝壳上料车定位升降气缸上升[SW]
714.11 BOOL  ; RK_07 #2铝壳上料车定位升降气缸下降[SW]
714.12 BOOL  ; RK_07 #3托盘下料车定位升降气缸上升[SW]
714.13 BOOL  ; RK_07 #3托盘下料车定位升降气缸下降[SW]
714.14 BOOL  ; RK_07 铝壳进料机械手升降气缸下降[SW]
714.15 BOOL  ; RK_07 铝壳进料机械手升降气缸上升[SW]
715.00 BOOL  ; RK_08 铝壳除尘旋转伸缩气缸缩回[SW]
715.01 BOOL  ; RK_08 铝壳除尘旋转伸缩气缸伸出[SW]
715.02 BOOL  ; RK_08 铝壳除尘伸缩气缸伸出[SW]
715.03 BOOL  ; RK_08 铝壳除尘伸缩气缸缩回[SW]
715.04 BOOL  ; RK_08 铝壳除尘夹爪气缸夹紧[SW]
715.05 BOOL  ; RK_08 铝壳除尘夹爪气缸张开[SW]
715.06 BOOL  ; RK_09 #1Hipot测试旋转伸缩气缸伸出[SW]
715.07 BOOL  ; RK_09 #1Hipot测试旋转伸缩气缸缩回[SW]
715.08 BOOL  ; RK_09 #1Hipot测试平台伸缩气缸缩回[SW]
715.09 BOOL  ; RK_09 #1Hipot测试平台伸缩气缸伸出[SW]
715.10 BOOL  ; RK_09 #1Hipot测试伸缩气缸伸出[SW]
715.11 BOOL  ; RK_09 #1Hipot测试伸缩气缸缩回[SW]
715.12 BOOL  ; RK_09 #2Hipot测试旋转伸缩气缸伸出[SW]
715.13 BOOL  ; RK_09 #2Hipot测试旋转伸缩气缸缩回[SW]
715.14 BOOL  ; RK_09 #2Hipot测试平台伸缩气缸缩回[SW]
715.15 BOOL  ; RK_09 #2Hipot测试平台伸缩气缸伸出[SW]
716.00 BOOL  ; RK_09 #2Hipot测试伸缩气缸伸出[SW]
716.01 BOOL  ; RK_09 #2Hipot测试伸缩气缸缩回[SW]
716.02 BOOL  ; RK_10 电池除尘上料机械手升降气缸下降[SW]
716.03 BOOL  ; RK_10 电池除尘上料机械手升降气缸上升[SW]
716.04 BOOL  ; RK_10 电池除尘上料机械手夹爪气缸夹紧[SW]
716.05 BOOL  ; RK_10 电池除尘上料机械手夹爪气缸张开[SW]
716.06 BOOL  ; RK_06 U8_X 电池上下料X轴报警复位[SW]
716.07 BOOL  ; RK_06 U8_X 电池上下料X轴使能[SW]
716.08 BOOL  ; RK_07 U8_Y 铝壳进料X轴报警复位[SW]
716.09 BOOL  ; RK_07 U8_Y 铝壳进料X轴使能[SW]
716.10 BOOL  ; RK_07 U8_Z 铝壳上料移载Y轴报警复位[SW]
716.11 BOOL  ; RK_07 U8_Z 铝壳上料移载Y轴使能[SW]
716.12 BOOL  ; RK_10 U8_U 电池除尘上料X轴报警复位[SW]
716.13 BOOL  ; RK_10 U8_U 电池除尘上料X轴使能[SW]
716.14 BOOL  ; RK_09 Hipot测试仪远程使能（取消）[SW]
716.15 BOOL  ; RK_07 #1铝壳上料启动指示[SW]
717.00 BOOL  ; RK_07 #2铝壳上料启动指示[SW]
717.01 BOOL  ; RK_07 #3托盘下料启动指示[SW]
717.02 BOOL  ; RK_07 铝壳上料移载吸盘立真空[SW]
717.03 BOOL  ; RK_07 铝壳进料吸盘立真空[SW]
717.04 BOOL  ; RK_07 #1铝壳上料电机正转[SW]
717.05 BOOL  ; RK_07 #1铝壳上料电机反转[SW]
717.06 BOOL  ; RK_10 Hipot检测NG拉带启动[SW]
717.07 BOOL  ; RK_08 铝壳除尘吹气阀开[SW]
717.08 BOOL  ; 0[SW]
717.09 BOOL  ; RK_07 #2铝壳上料电机正转[SW]
717.10 BOOL  ; RK_07 #2铝壳上料电机反转[SW]
717.11 BOOL  ; 启动指示_绿（公共）[SW]
717.12 BOOL  ; 停止指示_红（公共）[SW]
717.13 BOOL  ; 复位指示_黄（公共）[SW]
717.14 BOOL  ; RK_07 #3托盘下料电机正转[SW]
717.15 BOOL  ; RK_07 #3托盘下料电机反转[SW]
721.04 BOOL  ; RK_11 电池除尘吹气阀关[SW]
721.09 BOOL  ; RK_16#1移载激光焊任务取消[SW]
721.10 BOOL  ; RK_16#2移载激光焊任务取消[SW]
721.14 BOOL  ; RK_14 #1压装吸盘破真空[SW]
721.15 BOOL  ; RK_14 #2压装吸盘破真空[SW]
723.01 BOOL  ; RK_04 电芯除尘吹气阀关[SW]
723.02 BOOL  ; RK_02 扫码NG拉带停止[SW]
723.03 BOOL  ; RK_05 #1入壳吸盘破真空[SW]
723.04 BOOL  ; RK_05 #2入壳吸盘破真空[SW]
723.05 BOOL  ; RK_12 OK出料拉带停止[SW]
727.02 BOOL  ; RK_07 铝壳上料移载吸盘破真空[SW]
727.03 BOOL  ; RK_07 铝壳进料吸盘破真空[SW]
727.04 BOOL  ; RK_07 #1铝壳上料电机停止[SW]
727.06 BOOL  ; RK_10 Hipot检测NG拉带停止[SW]
727.07 BOOL  ; RK_08 铝壳除尘吹气阀关[SW]
727.09 BOOL  ; RK_07 #2铝壳上料电机停止[SW]
727.14 BOOL  ; RK_07 #3托盘下料电机停止[SW]
750.00 BOOL  ; RK_01 U0_X 电芯来料Y轴待料位[SW]
750.01 BOOL  ; RK_01 U0_X 电芯来料Y轴上料位[SW]
750.02 BOOL  ; RK_01 U0_X 电芯来料Y轴扫码位[SW]
750.03 BOOL  ; RK_01 U0_X 电芯来料Y轴下料位[SW]
750.04 BOOL  ; 备用[SW]
750.05 BOOL  ; 备用[SW]
750.06 BOOL  ; 备用[SW]
750.07 BOOL  ; 备用[SW]
750.08 BOOL  ; 备用[SW]
750.09 BOOL  ; 备用[SW]
750.10 BOOL  ; RK_01 U0_X 电芯来料Y轴回原点[SW]
750.11 BOOL  ; RK_01 U0_X 电芯来料Y轴JOG+[SW]
750.12 BOOL  ; RK_01 U0_X 电芯来料Y轴JOG-[SW]
750.13 BOOL  ; RK_01 U0_X 电芯来料Y轴JOG高速[SW]
750.14 BOOL  ; RK_01 U0_X 电芯来料Y轴JOG低速[SW]
750.15 BOOL  ; 备用[SW]
751.00 BOOL  ; RK_02 U0_Y 电芯进料X轴待料位[SW]
751.01 BOOL  ; RK_02 U0_Y 电芯进料X轴取料位[SW]
751.02 BOOL  ; RK_02 U0_Y 电芯进料X轴扫码OK放料位[SW]
751.03 BOOL  ; RK_02 U0_Y 电芯进料X轴扫码NG放料位[SW]
751.04 BOOL  ; 备用[SW]
751.05 BOOL  ; 备用[SW]
751.06 BOOL  ; 备用[SW]
751.07 BOOL  ; 备用[SW]
751.08 BOOL  ; 备用[SW]
751.09 BOOL  ; 备用[SW]
751.10 BOOL  ; RK_02 U0_Y 电芯进料X轴回原点[SW]
751.11 BOOL  ; RK_02 U0_Y 电芯进料X轴JOG+[SW]
751.12 BOOL  ; RK_02 U0_Y 电芯进料X轴JOG-[SW]
751.13 BOOL  ; RK_02 U0_Y 电芯进料X轴JOG高速[SW]
751.14 BOOL  ; RK_02 U0_Y 电芯进料X轴JOG低速[SW]
751.15 BOOL  ; 备用[SW]
752.00 BOOL  ; RK_02 U0_Z 电芯进料Z轴待料位（扫码）[SW]
752.01 BOOL  ; RK_02 U0_Z 电芯进料Z轴取料位[SW]
752.02 BOOL  ; RK_02 U0_Z 电芯进料Z轴扫码OK放料位[SW]
752.03 BOOL  ; RK_02 U0_Z 电芯进料Z轴扫码NG放料位[SW]
752.04 BOOL  ; RK_02 U0_Z 电芯进料Z轴扫码位[SW]
752.05 BOOL  ; 备用[SW]
752.06 BOOL  ; 备用[SW]
752.07 BOOL  ; 备用[SW]
752.08 BOOL  ; 备用[SW]
752.09 BOOL  ; 备用[SW]
752.10 BOOL  ; RK_02 U0_Z 电芯进料Z轴回原点[SW]
752.11 BOOL  ; RK_02 U0_Z 电芯进料Z轴JOG+[SW]
752.12 BOOL  ; RK_02 U0_Z 电芯进料Z轴JOG-[SW]
752.13 BOOL  ; RK_02 U0_Z 电芯进料Z轴JOG高速[SW]
752.14 BOOL  ; RK_02 U0_Z 电芯进料Z轴JOG低速[SW]
752.15 BOOL  ; 备用[SW]
753.00 BOOL  ; RK_03 U0_U 电芯上料X轴待料位[SW]
753.01 BOOL  ; RK_03 U0_U 电芯上料X轴取料位[SW]
753.02 BOOL  ; RK_03 U0_U 电芯上料X轴#1入壳放料位[SW]
753.03 BOOL  ; RK_03 U0_U 电芯上料X轴#2入壳放料位[SW]
753.04 BOOL  ; 备用[SW]
753.05 BOOL  ; 备用[SW]
753.06 BOOL  ; 备用[SW]
753.07 BOOL  ; 备用[SW]
753.08 BOOL  ; 备用[SW]
753.09 BOOL  ; 备用[SW]
753.10 BOOL  ; RK_03 U0_U 电芯上料X轴回原点[SW]
753.11 BOOL  ; RK_03 U0_U 电芯上料X轴JOG+[SW]
753.12 BOOL  ; RK_03 U0_U 电芯上料X轴JOG-[SW]
753.13 BOOL  ; RK_03 U0_U 电芯上料X轴JOG高速[SW]
753.14 BOOL  ; RK_03 U0_U 电芯上料X轴JOG低速[SW]
753.15 BOOL  ; 备用[SW]
754.00 BOOL  ; RK_05 U2_X #1入壳Y轴待料位[SW]
754.01 BOOL  ; RK_05 U2_X #1入壳Y轴滚轮压紧位[SW]
754.02 BOOL  ; RK_05 U2_X #1入壳Y轴滚轮松开位[SW]
754.03 BOOL  ; RK_05 U2_X #1入壳Y轴入壳位[SW]
754.04 BOOL  ; RK_05 U2_X #1入壳Y轴电芯定位夹爪松开位[SW]
754.05 BOOL  ; 备用[SW]
754.06 BOOL  ; 备用[SW]
754.07 BOOL  ; 备用[SW]
754.08 BOOL  ; 备用[SW]
754.09 BOOL  ; 备用[SW]
754.10 BOOL  ; RK_05 U2_X #1入壳Y轴回原点[SW]
754.11 BOOL  ; RK_05 U2_X #1入壳Y轴JOG+[SW]
754.12 BOOL  ; RK_05 U2_X #1入壳Y轴JOG-[SW]
754.13 BOOL  ; RK_05 U2_X #1入壳Y轴JOG高速[SW]
754.14 BOOL  ; RK_05 U2_X #1入壳Y轴JOG低速[SW]
754.15 BOOL  ; 备用[SW]
755.00 BOOL  ; RK_05 U2_Y #2入壳Y轴待料位[SW]
755.01 BOOL  ; RK_05 U2_Y #2入壳Y轴滚轮压紧位[SW]
755.02 BOOL  ; RK_05 U2_Y #2入壳Y轴滚轮松开位[SW]
755.03 BOOL  ; RK_05 U2_Y #2入壳Y轴入壳位[SW]
755.04 BOOL  ; RK_05 U2_Y #2入壳Y轴电芯定位夹爪松开位[SW]
755.05 BOOL  ; 备用[SW]
755.06 BOOL  ; 备用[SW]
755.07 BOOL  ; 备用[SW]
755.08 BOOL  ; 备用[SW]
755.09 BOOL  ; 备用[SW]
755.10 BOOL  ; RK_05 U2_Y #2入壳Y轴回原点[SW]
755.11 BOOL  ; RK_05 U2_Y #2入壳Y轴JOG+[SW]
755.12 BOOL  ; RK_05 U2_Y #2入壳Y轴JOG-[SW]
755.13 BOOL  ; RK_05 U2_Y #2入壳Y轴JOG高速[SW]
755.14 BOOL  ; RK_05 U2_Y #2入壳Y轴JOG低速[SW]
755.15 BOOL  ; 备用[SW]
756.00 BOOL  ; RK_12 U4_X 预焊上下料X轴待料位[SW]
756.01 BOOL  ; RK_12 U4_X 预焊上下料X轴除尘取料位[SW]
756.02 BOOL  ; RK_12 U4_X 预焊上下料X轴#1移载放料位[SW]
756.03 BOOL  ; RK_12 U4_X 预焊上下料X轴#2移载放料位[SW]
756.04 BOOL  ; RK_12 U4_X 预焊上下料X轴#1移载取料位[SW]
756.05 BOOL  ; RK_12 U4_X 预焊上下料X轴#2移载取料位[SW]
756.06 BOOL  ; RK_12 U4_X 预焊上下料X轴OK放料位[SW]
756.07 BOOL  ; RK_12 U4_X 预焊上下料X轴#1NG放料位[SW]
756.08 BOOL  ; RK_12 U4_X 预焊上下料X轴#2NG放料位[SW]
756.09 BOOL  ; 备用[SW]
756.10 BOOL  ; RK_12 U4_X 预焊上下料X轴回原点[SW]
756.11 BOOL  ; RK_12 U4_X 预焊上下料X轴JOG+[SW]
756.12 BOOL  ; RK_12 U4_X 预焊上下料X轴JOG-[SW]
756.13 BOOL  ; RK_12 U4_X 预焊上下料X轴JOG高速[SW]
756.14 BOOL  ; RK_12 U4_X 预焊上下料X轴JOG低速[SW]
756.15 BOOL  ; 备用[SW]
757.00 BOOL  ; RK_12 U4_Y 预焊上料Z轴待料位[SW]
757.01 BOOL  ; RK_12 U4_Y 预焊上料Z轴除尘取料位[SW]
757.02 BOOL  ; RK_12 U4_Y 预焊上料Z轴#1移载放料位[SW]
757.03 BOOL  ; RK_12 U4_Y 预焊上料Z轴#2移载放料位[SW]
757.04 BOOL  ; 备用[SW]
757.05 BOOL  ; 备用[SW]
757.06 BOOL  ; 备用[SW]
757.07 BOOL  ; 备用[SW]
757.08 BOOL  ; 备用[SW]
757.09 BOOL  ; 备用[SW]
757.10 BOOL  ; RK_12 U4_Y 预焊上料Z轴回原点[SW]
757.11 BOOL  ; RK_12 U4_Y 预焊上料Z轴JOG+[SW]
757.12 BOOL  ; RK_12 U4_Y 预焊上料Z轴JOG-[SW]
757.13 BOOL  ; RK_12 U4_Y 预焊上料Z轴JOG高速[SW]
757.14 BOOL  ; RK_12 U4_Y 预焊上料Z轴JOG低速[SW]
757.15 BOOL  ; 备用[SW]
758.00 BOOL  ; RK_12 U4_Z 预焊下料Z轴待料位[SW]
758.01 BOOL  ; RK_12 U4_Z 预焊下料Z轴#1移载取料位[SW]
758.02 BOOL  ; RK_12 U4_Z 预焊下料Z轴#2移载取料位[SW]
758.03 BOOL  ; RK_12 U4_Z 预焊下料Z轴OK放料位[SW]
758.04 BOOL  ; RK_12 U4_Z 预焊下料Z轴#1NG放料位[SW]
758.05 BOOL  ; RK_12 U4_Z 预焊下料Z轴#2NG放料位[SW]
758.06 BOOL  ; 备用[SW]
758.07 BOOL  ; 备用[SW]
758.08 BOOL  ; 备用[SW]
758.09 BOOL  ; 备用[SW]
758.10 BOOL  ; RK_12 U4_Z 预焊下料Z轴回原点[SW]
758.11 BOOL  ; RK_12 U4_Z 预焊下料Z轴JOG+[SW]
758.12 BOOL  ; RK_12 U4_Z 预焊下料Z轴JOG-[SW]
758.13 BOOL  ; RK_12 U4_Z 预焊下料Z轴JOG高速[SW]
758.14 BOOL  ; RK_12 U4_Z 预焊下料Z轴JOG低速[SW]
758.15 BOOL  ; 备用[SW]
759.00 BOOL  ; RK_13 U4_U #1移载Y轴待料位[SW]
759.01 BOOL  ; RK_13 U4_U #1移载Y轴取放料位[SW]
759.02 BOOL  ; RK_13 U4_U #1移载Y轴压装位[SW]
759.03 BOOL  ; RK_13 U4_U #1移载Y轴#1轮廓检测位[SW]
759.04 BOOL  ; RK_13 U4_U #1移载Y轴#2轮廓检测位[SW]
759.05 BOOL  ; RK_13 U4_U #1移载Y轴激光焊接位[SW]
759.06 BOOL  ; 备用[SW]
759.07 BOOL  ; 备用[SW]
759.08 BOOL  ; 备用[SW]
759.09 BOOL  ; 备用[SW]
759.10 BOOL  ; RK_13 U4_U #1移载Y轴回原点[SW]
759.11 BOOL  ; RK_13 U4_U #1移载Y轴JOG+[SW]
759.12 BOOL  ; RK_13 U4_U #1移载Y轴JOG-[SW]
759.13 BOOL  ; RK_13 U4_U #1移载Y轴JOG高速[SW]
759.14 BOOL  ; RK_13 U4_U #1移载Y轴JOG低速[SW]
759.15 BOOL  ; 备用[SW]
760.00 BOOL  ; RK_13 U6_X #2移载Y轴待料位[SW]
760.01 BOOL  ; RK_13 U6_X #2移载Y轴取放料位[SW]
760.02 BOOL  ; RK_13 U6_X #2移载Y轴压装位[SW]
760.03 BOOL  ; RK_13 U6_X #2移载Y轴#1轮廓检测位[SW]
760.04 BOOL  ; RK_13 U6_X #2移载Y轴#2轮廓检测位[SW]
760.05 BOOL  ; RK_13 U6_X #2移载Y轴激光焊接位[SW]
760.06 BOOL  ; 备用[SW]
760.07 BOOL  ; 备用[SW]
760.08 BOOL  ; 备用[SW]
760.09 BOOL  ; 备用[SW]
760.10 BOOL  ; RK_13 U6_X #2移载Y轴回原点[SW]
760.11 BOOL  ; RK_13 U6_X #2移载Y轴JOG+[SW]
760.12 BOOL  ; RK_13 U6_X #2移载Y轴JOG-[SW]
760.13 BOOL  ; RK_13 U6_X #2移载Y轴JOG高速[SW]
760.14 BOOL  ; RK_13 U6_X #2移载Y轴JOG低速[SW]
760.15 BOOL  ; 备用[SW]
761.00 BOOL  ; RK_16 U6_Y 激光焊接X轴待机位[SW]
761.01 BOOL  ; RK_16 U6_Y 激光焊接X轴#1移载焊接位[SW]
761.02 BOOL  ; RK_16 U6_Y 激光焊接X轴#2移载焊接位[SW]
761.03 BOOL  ; 备用[SW]
761.04 BOOL  ; 备用[SW]
761.05 BOOL  ; 备用[SW]
761.06 BOOL  ; 备用[SW]
761.07 BOOL  ; 备用[SW]
761.08 BOOL  ; 备用[SW]
761.09 BOOL  ; 备用[SW]
761.10 BOOL  ; RK_16 U6_Y 激光焊接X轴回原点[SW]
761.11 BOOL  ; RK_16 U6_Y 激光焊接X轴JOG+[SW]
761.12 BOOL  ; RK_16 U6_Y 激光焊接X轴JOG-[SW]
761.13 BOOL  ; RK_16 U6_Y 激光焊接X轴JOG高速[SW]
761.14 BOOL  ; RK_16 U6_Y 激光焊接X轴JOG低速[SW]
761.15 BOOL  ; 备用[SW]
